REGION Network 4: OUT4
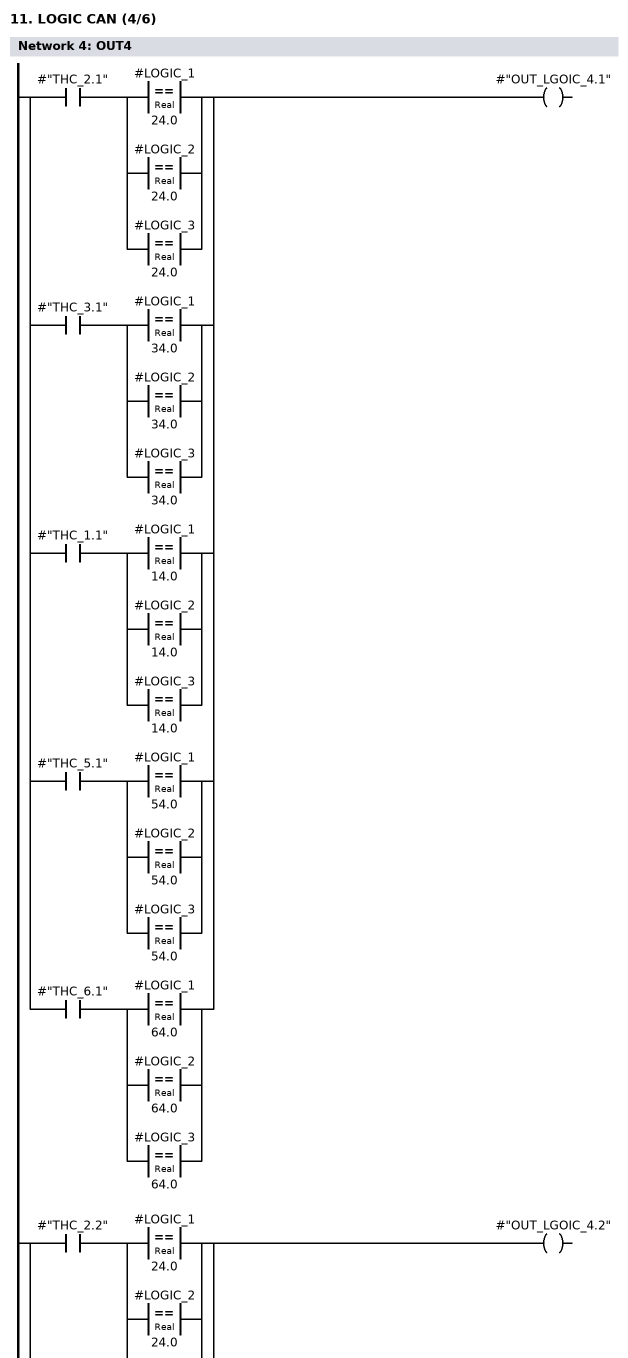
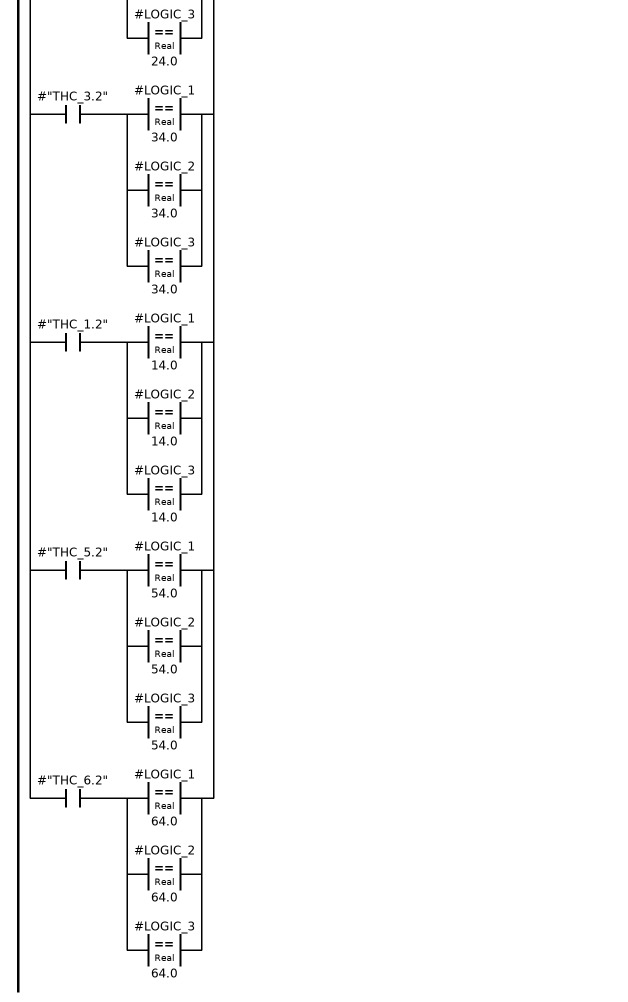
   RUNG wire#powerrail
      Contact( #"THC_2.1" )
      wire#w1
      { S7_Templates := "SrcType := Real" } EQ_Contact(in1 := #LOGIC_1, in2 := 24.0)
      wire#w2
      Coil( #"OUT_LGOIC_4.1" )
   END_RUNG
   RUNG wire#w1
      { S7_Templates := "SrcType := Real" } EQ_Contact(in1 := #LOGIC_2, in2 := 24.0)
   END_RUNG wire#w2
   RUNG wire#w1
      { S7_Templates := "SrcType := Real" } EQ_Contact(in1 := #LOGIC_3, in2 := 24.0)
   END_RUNG wire#w2
   RUNG wire#powerrail
      Contact( #"THC_3.1" )
      wire#w3
      { S7_Templates := "SrcType := Real" } EQ_Contact(in1 := #LOGIC_1, in2 := 34.0)
   END_RUNG wire#w2
   RUNG wire#w3
      { S7_Templates := "SrcType := Real" } EQ_Contact(in1 := #LOGIC_2, in2 := 34.0)
   END_RUNG wire#w2
   RUNG wire#w3
      { S7_Templates := "SrcType := Real" } EQ_Contact(in1 := #LOGIC_3, in2 := 34.0)
   END_RUNG wire#w2
   RUNG wire#powerrail
      Contact( #"THC_1.1" )
      wire#w4
      { S7_Templates := "SrcType := Real" } EQ_Contact(in1 := #LOGIC_1, in2 := 14.0)
   END_RUNG wire#w2
   RUNG wire#w4
      { S7_Templates := "SrcType := Real" } EQ_Contact(in1 := #LOGIC_2, in2 := 14.0)
   END_RUNG wire#w2
   RUNG wire#w4
      { S7_Templates := "SrcType := Real" } EQ_Contact(in1 := #LOGIC_3, in2 := 14.0)
   END_RUNG wire#w2
   RUNG wire#powerrail
      Contact( #"THC_5.1" )
      wire#w5
      { S7_Templates := "SrcType := Real" } EQ_Contact(in1 := #LOGIC_1, in2 := 54.0)
   END_RUNG wire#w2
   RUNG wire#w5
      { S7_Templates := "SrcType := Real" } EQ_Contact(in1 := #LOGIC_2, in2 := 54.0)
   END_RUNG wire#w2
   RUNG wire#w5
      { S7_Templates := "SrcType := Real" } EQ_Contact(in1 := #LOGIC_3, in2 := 54.0)
   END_RUNG wire#w2
   RUNG wire#powerrail
      Contact( #"THC_6.1" )
      wire#w6
      { S7_Templates := "SrcType := Real" } EQ_Contact(in1 := #LOGIC_1, in2 := 64.0)
   END_RUNG wire#w2
   RUNG wire#w6
      { S7_Templates := "SrcType := Real" } EQ_Contact(in1 := #LOGIC_2, in2 := 64.0)
   END_RUNG wire#w2
   RUNG wire#w6
      { S7_Templates := "SrcType := Real" } EQ_Contact(in1 := #LOGIC_3, in2 := 64.0)
   END_RUNG wire#w2
   RUNG wire#powerrail
      Contact( #"THC_2.2" )
      wire#w7
      { S7_Templates := "SrcType := Real" } EQ_Contact(in1 := #LOGIC_1, in2 := 24.0)
      wire#w8
      Coil( #"OUT_LGOIC_4.2" )
   END_RUNG
   RUNG wire#w7
      { S7_Templates := "SrcType := Real" } EQ_Contact(in1 := #LOGIC_2, in2 := 24.0)
   END_RUNG wire#w8
   RUNG wire#w7
      { S7_Templates := "SrcType := Real" } EQ_Contact(in1 := #LOGIC_3, in2 := 24.0)
   END_RUNG wire#w8
   RUNG wire#powerrail
      Contact( #"THC_3.2" )
      wire#w9
      { S7_Templates := "SrcType := Real" } EQ_Contact(in1 := #LOGIC_1, in2 := 34.0)
   END_RUNG wire#w8
   RUNG wire#w9
      { S7_Templates := "SrcType := Real" } EQ_Contact(in1 := #LOGIC_2, in2 := 34.0)
   END_RUNG wire#w8
   RUNG wire#w9
      { S7_Templates := "SrcType := Real" } EQ_Contact(in1 := #LOGIC_3, in2 := 34.0)
   END_RUNG wire#w8
   RUNG wire#powerrail
      Contact( #"THC_1.2" )
      wire#w10
      { S7_Templates := "SrcType := Real" } EQ_Contact(in1 := #LOGIC_1, in2 := 14.0)
   END_RUNG wire#w8
   RUNG wire#w10
      { S7_Templates := "SrcType := Real" } EQ_Contact(in1 := #LOGIC_2, in2 := 14.0)
   END_RUNG wire#w8
   RUNG wire#w10
      { S7_Templates := "SrcType := Real" } EQ_Contact(in1 := #LOGIC_3, in2 := 14.0)
   END_RUNG wire#w8
   RUNG wire#powerrail
      Contact( #"THC_5.2" )
      wire#w11
      { S7_Templates := "SrcType := Real" } EQ_Contact(in1 := #LOGIC_1, in2 := 54.0)
   END_RUNG wire#w8
   RUNG wire#w11
      { S7_Templates := "SrcType := Real" } EQ_Contact(in1 := #LOGIC_2, in2 := 54.0)
   END_RUNG wire#w8
   RUNG wire#w11
      { S7_Templates := "SrcType := Real" } EQ_Contact(in1 := #LOGIC_3, in2 := 54.0)
   END_RUNG wire#w8
   RUNG wire#powerrail
      Contact( #"THC_6.2" )
      wire#w12
      { S7_Templates := "SrcType := Real" } EQ_Contact(in1 := #LOGIC_1, in2 := 64.0)
   END_RUNG wire#w8
   RUNG wire#w12
      { S7_Templates := "SrcType := Real" } EQ_Contact(in1 := #LOGIC_2, in2 := 64.0)
   END_RUNG wire#w8
   RUNG wire#w12
      { S7_Templates := "SrcType := Real" } EQ_Contact(in1 := #LOGIC_3, in2 := 64.0)
   END_RUNG wire#w8
   // the same network as SCL:
   #"OUT_LGOIC_4.1" := (#"THC_2.1" AND ((#LOGIC_1 = 24.0) OR (#LOGIC_2 = 24.0) OR (#LOGIC_3 = 24.0))) OR (#"THC_3.1" AND ((#LOGIC_1 = 34.0) OR (#LOGIC_2 = 34.0) OR (#LOGIC_3 = 34.0))) OR (#"THC_1.1" AND ((#LOGIC_1 = 14.0) OR (#LOGIC_2 = 14.0) OR (#LOGIC_3 = 14.0))) OR (#"THC_5.1" AND ((#LOGIC_1 = 54.0) OR (#LOGIC_2 = 54.0) OR (#LOGIC_3 = 54.0))) OR (#"THC_6.1" AND ((#LOGIC_1 = 64.0) OR (#LOGIC_2 = 64.0) OR (#LOGIC_3 = 64.0)));
   #"OUT_LGOIC_4.2" := (#"THC_2.2" AND ((#LOGIC_1 = 24.0) OR (#LOGIC_2 = 24.0) OR (#LOGIC_3 = 24.0))) OR (#"THC_3.2" AND ((#LOGIC_1 = 34.0) OR (#LOGIC_2 = 34.0) OR (#LOGIC_3 = 34.0))) OR (#"THC_1.2" AND ((#LOGIC_1 = 14.0) OR (#LOGIC_2 = 14.0) OR (#LOGIC_3 = 14.0))) OR (#"THC_5.2" AND ((#LOGIC_1 = 54.0) OR (#LOGIC_2 = 54.0) OR (#LOGIC_3 = 54.0))) OR (#"THC_6.2" AND ((#LOGIC_1 = 64.0) OR (#LOGIC_2 = 64.0) OR (#LOGIC_3 = 64.0)));
END_REGION

REGION Network 5: OUT5
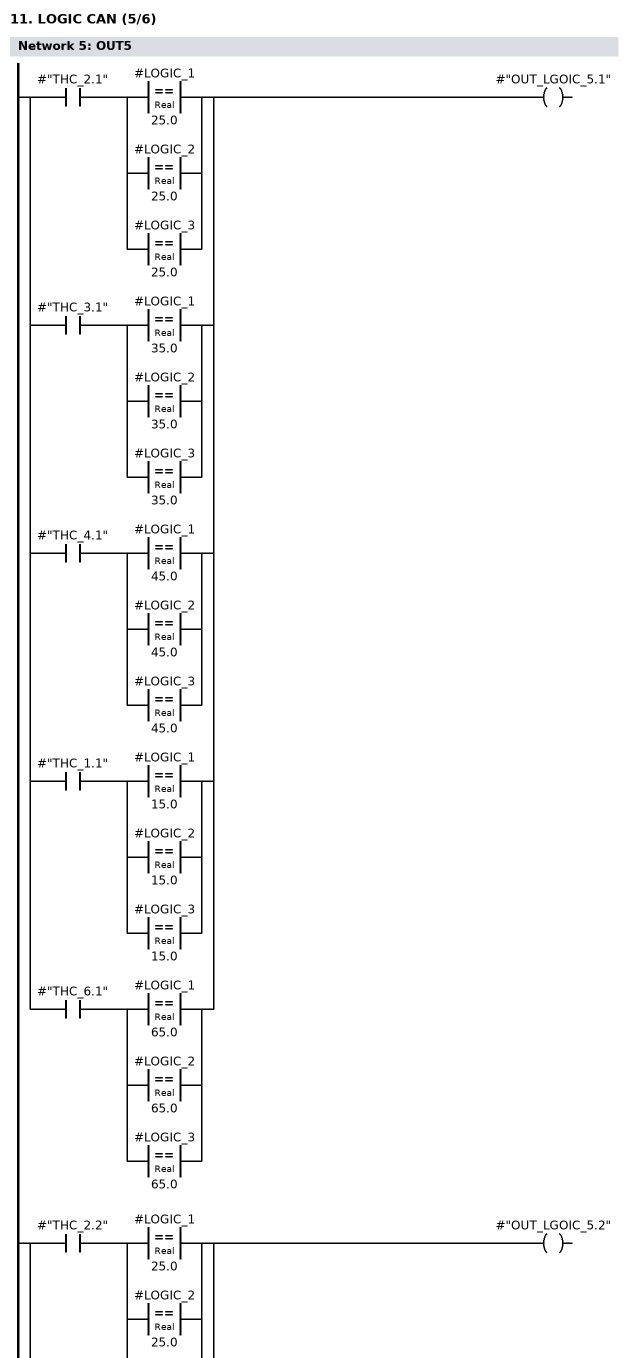
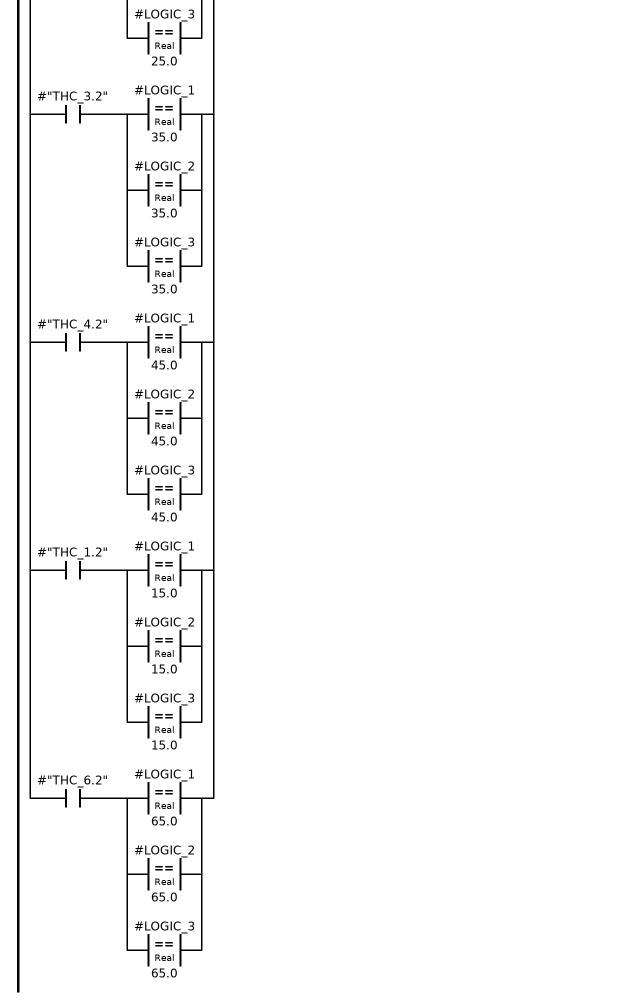
   RUNG wire#powerrail
      Contact( #"THC_2.1" )
      wire#w1
      { S7_Templates := "SrcType := Real" } EQ_Contact(in1 := #LOGIC_1, in2 := 25.0)
      wire#w2
      Coil( #"OUT_LGOIC_5.1" )
   END_RUNG
   RUNG wire#w1
      { S7_Templates := "SrcType := Real" } EQ_Contact(in1 := #LOGIC_2, in2 := 25.0)
   END_RUNG wire#w2
   RUNG wire#w1
      { S7_Templates := "SrcType := Real" } EQ_Contact(in1 := #LOGIC_3, in2 := 25.0)
   END_RUNG wire#w2
   RUNG wire#powerrail
      Contact( #"THC_3.1" )
      wire#w3
      { S7_Templates := "SrcType := Real" } EQ_Contact(in1 := #LOGIC_1, in2 := 35.0)
   END_RUNG wire#w2
   RUNG wire#w3
      { S7_Templates := "SrcType := Real" } EQ_Contact(in1 := #LOGIC_2, in2 := 35.0)
   END_RUNG wire#w2
   RUNG wire#w3
      { S7_Templates := "SrcType := Real" } EQ_Contact(in1 := #LOGIC_3, in2 := 35.0)
   END_RUNG wire#w2
   RUNG wire#powerrail
      Contact( #"THC_4.1" )
      wire#w4
      { S7_Templates := "SrcType := Real" } EQ_Contact(in1 := #LOGIC_1, in2 := 45.0)
   END_RUNG wire#w2
   RUNG wire#w4
      { S7_Templates := "SrcType := Real" } EQ_Contact(in1 := #LOGIC_2, in2 := 45.0)
   END_RUNG wire#w2
   RUNG wire#w4
      { S7_Templates := "SrcType := Real" } EQ_Contact(in1 := #LOGIC_3, in2 := 45.0)
   END_RUNG wire#w2
   RUNG wire#powerrail
      Contact( #"THC_1.1" )
      wire#w5
      { S7_Templates := "SrcType := Real" } EQ_Contact(in1 := #LOGIC_1, in2 := 15.0)
   END_RUNG wire#w2
   RUNG wire#w5
      { S7_Templates := "SrcType := Real" } EQ_Contact(in1 := #LOGIC_2, in2 := 15.0)
   END_RUNG wire#w2
   RUNG wire#w5
      { S7_Templates := "SrcType := Real" } EQ_Contact(in1 := #LOGIC_3, in2 := 15.0)
   END_RUNG wire#w2
   RUNG wire#powerrail
      Contact( #"THC_6.1" )
      wire#w6
      { S7_Templates := "SrcType := Real" } EQ_Contact(in1 := #LOGIC_1, in2 := 65.0)
   END_RUNG wire#w2
   RUNG wire#w6
      { S7_Templates := "SrcType := Real" } EQ_Contact(in1 := #LOGIC_2, in2 := 65.0)
   END_RUNG wire#w2
   RUNG wire#w6
      { S7_Templates := "SrcType := Real" } EQ_Contact(in1 := #LOGIC_3, in2 := 65.0)
   END_RUNG wire#w2
   RUNG wire#powerrail
      Contact( #"THC_2.2" )
      wire#w7
      { S7_Templates := "SrcType := Real" } EQ_Contact(in1 := #LOGIC_1, in2 := 25.0)
      wire#w8
      Coil( #"OUT_LGOIC_5.2" )
   END_RUNG
   RUNG wire#w7
      { S7_Templates := "SrcType := Real" } EQ_Contact(in1 := #LOGIC_2, in2 := 25.0)
   END_RUNG wire#w8
   RUNG wire#w7
      { S7_Templates := "SrcType := Real" } EQ_Contact(in1 := #LOGIC_3, in2 := 25.0)
   END_RUNG wire#w8
   RUNG wire#powerrail
      Contact( #"THC_3.2" )
      wire#w9
      { S7_Templates := "SrcType := Real" } EQ_Contact(in1 := #LOGIC_1, in2 := 35.0)
   END_RUNG wire#w8
   RUNG wire#w9
      { S7_Templates := "SrcType := Real" } EQ_Contact(in1 := #LOGIC_2, in2 := 35.0)
   END_RUNG wire#w8
   RUNG wire#w9
      { S7_Templates := "SrcType := Real" } EQ_Contact(in1 := #LOGIC_3, in2 := 35.0)
   END_RUNG wire#w8
   RUNG wire#powerrail
      Contact( #"THC_4.2" )
      wire#w10
      { S7_Templates := "SrcType := Real" } EQ_Contact(in1 := #LOGIC_1, in2 := 45.0)
   END_RUNG wire#w8
   RUNG wire#w10
      { S7_Templates := "SrcType := Real" } EQ_Contact(in1 := #LOGIC_2, in2 := 45.0)
   END_RUNG wire#w8
   RUNG wire#w10
      { S7_Templates := "SrcType := Real" } EQ_Contact(in1 := #LOGIC_3, in2 := 45.0)
   END_RUNG wire#w8
   RUNG wire#powerrail
      Contact( #"THC_1.2" )
      wire#w11
      { S7_Templates := "SrcType := Real" } EQ_Contact(in1 := #LOGIC_1, in2 := 15.0)
   END_RUNG wire#w8
   RUNG wire#w11
      { S7_Templates := "SrcType := Real" } EQ_Contact(in1 := #LOGIC_2, in2 := 15.0)
   END_RUNG wire#w8
   RUNG wire#w11
      { S7_Templates := "SrcType := Real" } EQ_Contact(in1 := #LOGIC_3, in2 := 15.0)
   END_RUNG wire#w8
   RUNG wire#powerrail
      Contact( #"THC_6.2" )
      wire#w12
      { S7_Templates := "SrcType := Real" } EQ_Contact(in1 := #LOGIC_1, in2 := 65.0)
   END_RUNG wire#w8
   RUNG wire#w12
      { S7_Templates := "SrcType := Real" } EQ_Contact(in1 := #LOGIC_2, in2 := 65.0)
   END_RUNG wire#w8
   RUNG wire#w12
      { S7_Templates := "SrcType := Real" } EQ_Contact(in1 := #LOGIC_3, in2 := 65.0)
   END_RUNG wire#w8
   // the same network as SCL:
   #"OUT_LGOIC_5.1" := (#"THC_2.1" AND ((#LOGIC_1 = 25.0) OR (#LOGIC_2 = 25.0) OR (#LOGIC_3 = 25.0))) OR (#"THC_3.1" AND ((#LOGIC_1 = 35.0) OR (#LOGIC_2 = 35.0) OR (#LOGIC_3 = 35.0))) OR (#"THC_4.1" AND ((#LOGIC_1 = 45.0) OR (#LOGIC_2 = 45.0) OR (#LOGIC_3 = 45.0))) OR (#"THC_1.1" AND ((#LOGIC_1 = 15.0) OR (#LOGIC_2 = 15.0) OR (#LOGIC_3 = 15.0))) OR (#"THC_6.1" AND ((#LOGIC_1 = 65.0) OR (#LOGIC_2 = 65.0) OR (#LOGIC_3 = 65.0)));
   #"OUT_LGOIC_5.2" := (#"THC_2.2" AND ((#LOGIC_1 = 25.0) OR (#LOGIC_2 = 25.0) OR (#LOGIC_3 = 25.0))) OR (#"THC_3.2" AND ((#LOGIC_1 = 35.0) OR (#LOGIC_2 = 35.0) OR (#LOGIC_3 = 35.0))) OR (#"THC_4.2" AND ((#LOGIC_1 = 45.0) OR (#LOGIC_2 = 45.0) OR (#LOGIC_3 = 45.0))) OR (#"THC_1.2" AND ((#LOGIC_1 = 15.0) OR (#LOGIC_2 = 15.0) OR (#LOGIC_3 = 15.0))) OR (#"THC_6.2" AND ((#LOGIC_1 = 65.0) OR (#LOGIC_2 = 65.0) OR (#LOGIC_3 = 65.0)));
END_REGION

REGION Network 6: OUT6
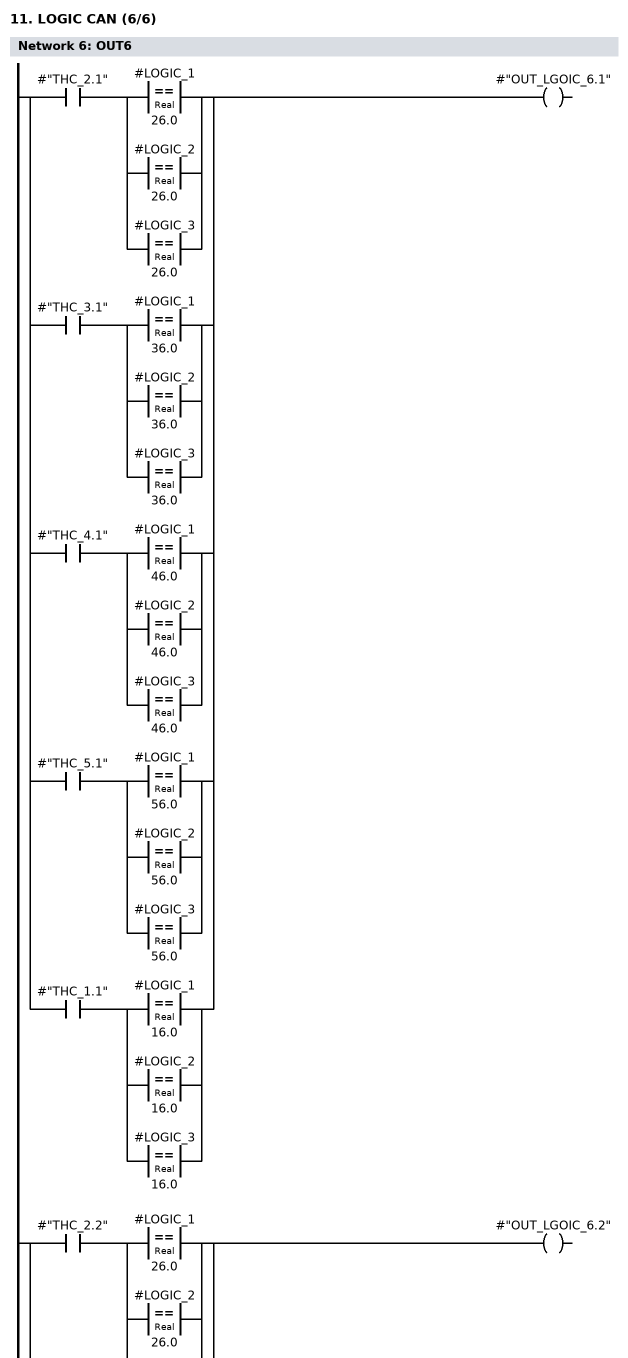
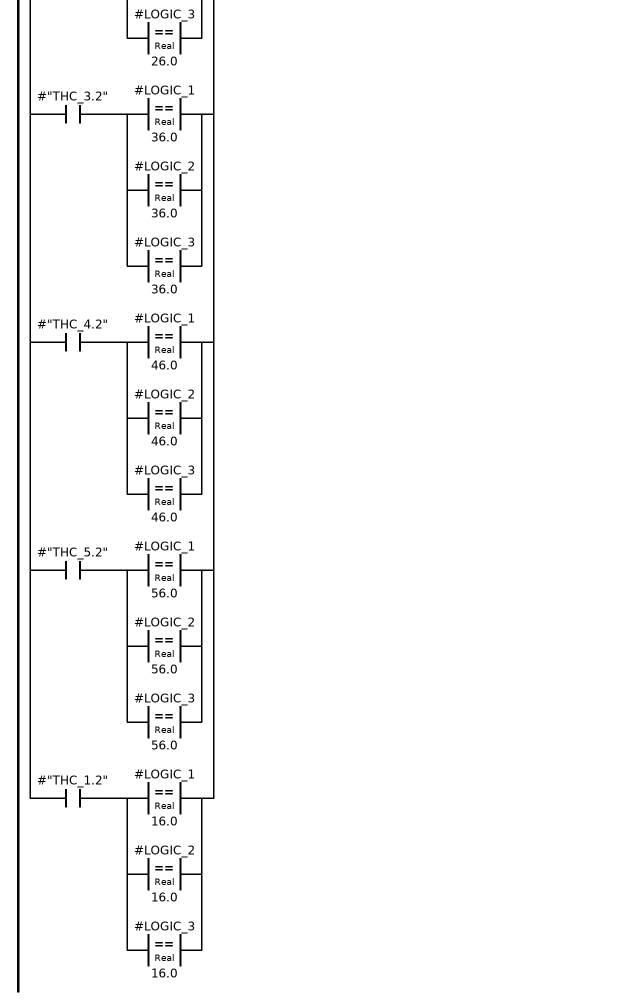
   RUNG wire#powerrail
      Contact( #"THC_2.1" )
      wire#w1
      { S7_Templates := "SrcType := Real" } EQ_Contact(in1 := #LOGIC_1, in2 := 26.0)
      wire#w2
      Coil( #"OUT_LGOIC_6.1" )
   END_RUNG
   RUNG wire#w1
      { S7_Templates := "SrcType := Real" } EQ_Contact(in1 := #LOGIC_2, in2 := 26.0)
   END_RUNG wire#w2
   RUNG wire#w1
      { S7_Templates := "SrcType := Real" } EQ_Contact(in1 := #LOGIC_3, in2 := 26.0)
   END_RUNG wire#w2
   RUNG wire#powerrail
      Contact( #"THC_3.1" )
      wire#w3
      { S7_Templates := "SrcType := Real" } EQ_Contact(in1 := #LOGIC_1, in2 := 36.0)
   END_RUNG wire#w2
   RUNG wire#w3
      { S7_Templates := "SrcType := Real" } EQ_Contact(in1 := #LOGIC_2, in2 := 36.0)
   END_RUNG wire#w2
   RUNG wire#w3
      { S7_Templates := "SrcType := Real" } EQ_Contact(in1 := #LOGIC_3, in2 := 36.0)
   END_RUNG wire#w2
   RUNG wire#powerrail
      Contact( #"THC_4.1" )
      wire#w4
      { S7_Templates := "SrcType := Real" } EQ_Contact(in1 := #LOGIC_1, in2 := 46.0)
   END_RUNG wire#w2
   RUNG wire#w4
      { S7_Templates := "SrcType := Real" } EQ_Contact(in1 := #LOGIC_2, in2 := 46.0)
   END_RUNG wire#w2
   RUNG wire#w4
      { S7_Templates := "SrcType := Real" } EQ_Contact(in1 := #LOGIC_3, in2 := 46.0)
   END_RUNG wire#w2
   RUNG wire#powerrail
      Contact( #"THC_5.1" )
      wire#w5
      { S7_Templates := "SrcType := Real" } EQ_Contact(in1 := #LOGIC_1, in2 := 56.0)
   END_RUNG wire#w2
   RUNG wire#w5
      { S7_Templates := "SrcType := Real" } EQ_Contact(in1 := #LOGIC_2, in2 := 56.0)
   END_RUNG wire#w2
   RUNG wire#w5
      { S7_Templates := "SrcType := Real" } EQ_Contact(in1 := #LOGIC_3, in2 := 56.0)
   END_RUNG wire#w2
   RUNG wire#powerrail
      Contact( #"THC_1.1" )
      wire#w6
      { S7_Templates := "SrcType := Real" } EQ_Contact(in1 := #LOGIC_1, in2 := 16.0)
   END_RUNG wire#w2
   RUNG wire#w6
      { S7_Templates := "SrcType := Real" } EQ_Contact(in1 := #LOGIC_2, in2 := 16.0)
   END_RUNG wire#w2
   RUNG wire#w6
      { S7_Templates := "SrcType := Real" } EQ_Contact(in1 := #LOGIC_3, in2 := 16.0)
   END_RUNG wire#w2
   RUNG wire#powerrail
      Contact( #"THC_2.2" )
      wire#w7
      { S7_Templates := "SrcType := Real" } EQ_Contact(in1 := #LOGIC_1, in2 := 26.0)
      wire#w8
      Coil( #"OUT_LGOIC_6.2" )
   END_RUNG
   RUNG wire#w7
      { S7_Templates := "SrcType := Real" } EQ_Contact(in1 := #LOGIC_2, in2 := 26.0)
   END_RUNG wire#w8
   RUNG wire#w7
      { S7_Templates := "SrcType := Real" } EQ_Contact(in1 := #LOGIC_3, in2 := 26.0)
   END_RUNG wire#w8
   RUNG wire#powerrail
      Contact( #"THC_3.2" )
      wire#w9
      { S7_Templates := "SrcType := Real" } EQ_Contact(in1 := #LOGIC_1, in2 := 36.0)
   END_RUNG wire#w8
   RUNG wire#w9
      { S7_Templates := "SrcType := Real" } EQ_Contact(in1 := #LOGIC_2, in2 := 36.0)
   END_RUNG wire#w8
   RUNG wire#w9
      { S7_Templates := "SrcType := Real" } EQ_Contact(in1 := #LOGIC_3, in2 := 36.0)
   END_RUNG wire#w8
   RUNG wire#powerrail
      Contact( #"THC_4.2" )
      wire#w10
      { S7_Templates := "SrcType := Real" } EQ_Contact(in1 := #LOGIC_1, in2 := 46.0)
   END_RUNG wire#w8
   RUNG wire#w10
      { S7_Templates := "SrcType := Real" } EQ_Contact(in1 := #LOGIC_2, in2 := 46.0)
   END_RUNG wire#w8
   RUNG wire#w10
      { S7_Templates := "SrcType := Real" } EQ_Contact(in1 := #LOGIC_3, in2 := 46.0)
   END_RUNG wire#w8
   RUNG wire#powerrail
      Contact( #"THC_5.2" )
      wire#w11
      { S7_Templates := "SrcType := Real" } EQ_Contact(in1 := #LOGIC_1, in2 := 56.0)
   END_RUNG wire#w8
   RUNG wire#w11
      { S7_Templates := "SrcType := Real" } EQ_Contact(in1 := #LOGIC_2, in2 := 56.0)
   END_RUNG wire#w8
   RUNG wire#w11
      { S7_Templates := "SrcType := Real" } EQ_Contact(in1 := #LOGIC_3, in2 := 56.0)
   END_RUNG wire#w8
   RUNG wire#powerrail
      Contact( #"THC_1.2" )
      wire#w12
      { S7_Templates := "SrcType := Real" } EQ_Contact(in1 := #LOGIC_1, in2 := 16.0)
   END_RUNG wire#w8
   RUNG wire#w12
      { S7_Templates := "SrcType := Real" } EQ_Contact(in1 := #LOGIC_2, in2 := 16.0)
   END_RUNG wire#w8
   RUNG wire#w12
      { S7_Templates := "SrcType := Real" } EQ_Contact(in1 := #LOGIC_3, in2 := 16.0)
   END_RUNG wire#w8
   // the same network as SCL:
   #"OUT_LGOIC_6.1" := (#"THC_2.1" AND ((#LOGIC_1 = 26.0) OR (#LOGIC_2 = 26.0) OR (#LOGIC_3 = 26.0))) OR (#"THC_3.1" AND ((#LOGIC_1 = 36.0) OR (#LOGIC_2 = 36.0) OR (#LOGIC_3 = 36.0))) OR (#"THC_4.1" AND ((#LOGIC_1 = 46.0) OR (#LOGIC_2 = 46.0) OR (#LOGIC_3 = 46.0))) OR (#"THC_5.1" AND ((#LOGIC_1 = 56.0) OR (#LOGIC_2 = 56.0) OR (#LOGIC_3 = 56.0))) OR (#"THC_1.1" AND ((#LOGIC_1 = 16.0) OR (#LOGIC_2 = 16.0) OR (#LOGIC_3 = 16.0)));
   #"OUT_LGOIC_6.2" := (#"THC_2.2" AND ((#LOGIC_1 = 26.0) OR (#LOGIC_2 = 26.0) OR (#LOGIC_3 = 26.0))) OR (#"THC_3.2" AND ((#LOGIC_1 = 36.0) OR (#LOGIC_2 = 36.0) OR (#LOGIC_3 = 36.0))) OR (#"THC_4.2" AND ((#LOGIC_1 = 46.0) OR (#LOGIC_2 = 46.0) OR (#LOGIC_3 = 46.0))) OR (#"THC_5.2" AND ((#LOGIC_1 = 56.0) OR (#LOGIC_2 = 56.0) OR (#LOGIC_3 = 56.0))) OR (#"THC_1.2" AND ((#LOGIC_1 = 16.0) OR (#LOGIC_2 = 16.0) OR (#LOGIC_3 = 16.0)));
END_REGION
END_FUNCTION_BLOCK

FUNCTION "3.OUTPUT_PLC" : Void   // FC3, LAD
{ S7_Optimized_Access := 'TRUE' }
VERSION : 0.1
// stored: AutoNumber false, CodeModifiedDate 2025-08-27T17:07:28.4518091Z, CompileDate 2025-08-30T17:40:35.2673041Z, CreationDate 2024-10-12T12:36:08.0193576Z, HandleErrorsWithinBlock false, InterfaceModifiedDate 2022-06-07T03:40:45.7898546Z, IsConsistent true, IsIECCheckEnabled false, IsKnowHowProtected false, IsWriteProtected false, LibraryConformanceStatus The object is library-conformant., ModifiedDate 2025-08-27T17:07:28.4518091Z, ParameterModified 2022-06-07T03:40:45.7898546Z, PLCSimAdvancedSupport false, SetENOAutomatically False, StructureModified 2022-06-07T03:40:45.7898546Z, UDAEnableTagReadback false
   VAR_INPUT
      A1 : Bool;
      M1 : Bool;
      A2 : Bool;
      M2 : Bool;
      A3 : Bool;
      M3 : Bool;
      A4 : Bool;
      M4 : Bool;
   END_VAR
   VAR_OUTPUT
      OUT1 : Bool;
      OUT2 : Bool;
      OUT3 : Bool;
      OUT4 : Bool;
   END_VAR
BEGIN

REGION Network 1
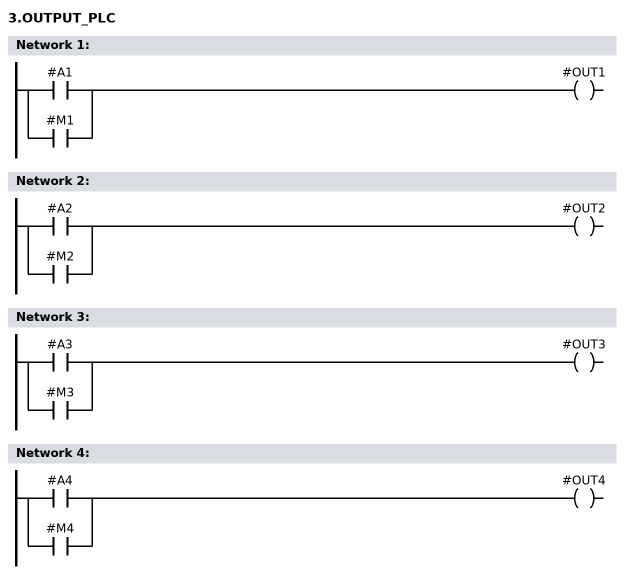
   RUNG wire#powerrail
      Contact( #A1 )
      wire#w1
      Coil( #OUT1 )
   END_RUNG
   RUNG wire#powerrail
      Contact( #M1 )
   END_RUNG wire#w1
   // the same network as SCL:
   #OUT1 := #A1 OR #M1;
END_REGION

REGION Network 2
   RUNG wire#powerrail
      Contact( #A2 )
      wire#w1
      Coil( #OUT2 )
   END_RUNG
   RUNG wire#powerrail
      Contact( #M2 )
   END_RUNG wire#w1
   // the same network as SCL:
   #OUT2 := #A2 OR #M2;
END_REGION

REGION Network 3
   RUNG wire#powerrail
      Contact( #A3 )
      wire#w1
      Coil( #OUT3 )
   END_RUNG
   RUNG wire#powerrail
      Contact( #M3 )
   END_RUNG wire#w1
   // the same network as SCL:
   #OUT3 := #A3 OR #M3;
END_REGION

REGION Network 4
   RUNG wire#powerrail
      Contact( #A4 )
      wire#w1
      Coil( #OUT4 )
   END_RUNG
   RUNG wire#powerrail
      Contact( #M4 )
   END_RUNG wire#w1
   // the same network as SCL:
   #OUT4 := #A4 OR #M4;
END_REGION
END_FUNCTION

FUNCTION_BLOCK "3.RUN_MODE"   // FB3, LAD
{ S7_Optimized_Access := 'TRUE' }
VERSION : 0.1
// stored: AutoNumber false, CodeModifiedDate 2025-08-27T17:11:43.2955348Z, CompileDate 2025-08-30T17:40:35.1660868Z, CreationDate 2024-10-12T12:36:08.0193576Z, DownloadWithoutReinit false, HandleErrorsWithinBlock false, InterfaceModifiedDate 2023-07-24T14:42:19.3789304Z, IsConsistent true, IsIECCheckEnabled false, IsKnowHowProtected false, IsRetainMemResEnabled false, IsWriteProtected false, LibraryConformanceStatus The object is library-conformant., MemoryReserve 100, ModifiedDate 2025-08-27T17:11:43.2955348Z, ParameterModified 2023-07-24T14:41:56.9787559Z, PLCSimAdvancedSupport false, SetENOAutomatically False, StructureModified 2023-07-24T14:42:19.3789304Z, UDAEnableTagReadback false
   VAR_INPUT
      NN_RUN : Bool;
      NN_STOP : Bool;
      SW_SIM : Bool;
      SW_MAN : Bool;
      SW_AUT : Bool;
   END_VAR
   VAR_OUTPUT
      RUN : Bool;
      SIM : Bool;
      MAN : Bool;
      AUT : Bool;
   END_VAR
   VAR
      TEMP1 : Bool;
      TEMP2 : Bool;
   END_VAR
BEGIN

REGION Network 1
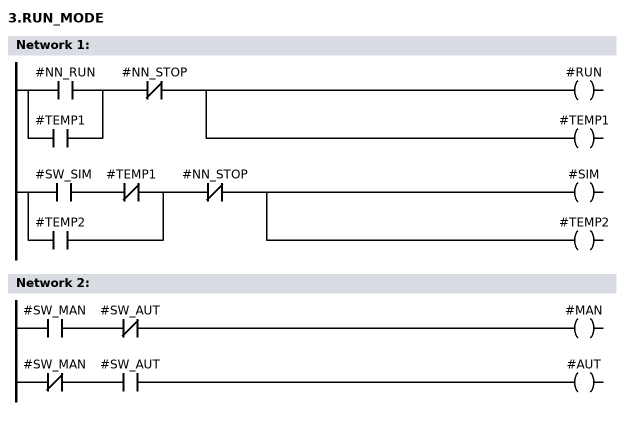
   RUNG wire#powerrail
      Contact( #NN_RUN )
      wire#w1
      I_Contact( #NN_STOP )
      wire#w2
      Coil( #RUN )
   END_RUNG
   RUNG wire#powerrail
      Contact( #TEMP1 )
   END_RUNG wire#w1
   RUNG wire#w2
      Coil( #TEMP1 )
   END_RUNG
   RUNG wire#powerrail
      Contact( #SW_SIM )
      I_Contact( #TEMP1 )
      wire#w3
      I_Contact( #NN_STOP )
      wire#w4
      Coil( #SIM )
   END_RUNG
   RUNG wire#powerrail
      Contact( #TEMP2 )
   END_RUNG wire#w3
   RUNG wire#w4
      Coil( #TEMP2 )
   END_RUNG
   // the same network as SCL:
   #RUN := (#NN_RUN OR #TEMP1) AND NOT #NN_STOP;
   #TEMP1 := #RUN;
   #SIM := ((#SW_SIM AND NOT #TEMP1) OR #TEMP2) AND NOT #NN_STOP;
   #TEMP2 := #SIM;
END_REGION

REGION Network 2
   RUNG wire#powerrail
      Contact( #SW_MAN )
      I_Contact( #SW_AUT )
      Coil( #MAN )
   END_RUNG
   RUNG wire#powerrail
      I_Contact( #SW_MAN )
      Contact( #SW_AUT )
      Coil( #AUT )
   END_RUNG
   // the same network as SCL:
   #MAN := #SW_MAN AND NOT #SW_AUT;
   #AUT := NOT #SW_MAN AND #SW_AUT;
END_REGION
END_FUNCTION_BLOCK

FUNCTION "4.CONVERT_VOLUME" : Void   // FC4, LAD
{ S7_Optimized_Access := 'TRUE' }
VERSION : 0.1
// stored: AutoNumber true, CodeModifiedDate 2025-08-27T17:08:03.467369Z, CompileDate 2025-08-30T17:40:35.2171394Z, CreationDate 2024-10-12T12:36:08.0193576Z, HandleErrorsWithinBlock false, InterfaceModifiedDate 2023-07-25T19:47:42.5745Z, IsConsistent true, IsIECCheckEnabled false, IsKnowHowProtected false, IsWriteProtected false, LibraryConformanceStatus The object is library-conformant., ModifiedDate 2025-08-27T17:08:03.467369Z, ParameterModified 2023-07-25T19:47:42.5745Z, PLCSimAdvancedSupport false, SetENOAutomatically False, StructureModified 2023-07-25T19:47:42.5745Z, UDAEnableTagReadback false
   VAR_INPUT
      SO_KHOI : Real;
      M3_MAX : Real;
   END_VAR
   VAR_OUTPUT
      SO_ME : Real;
      "M3/ME" : Real;
   END_VAR
   VAR_TEMP
      TEMP1 : Real;
      TEMP2 : Int;
      TEMP3 : Real;
   END_VAR
BEGIN

REGION Network 1
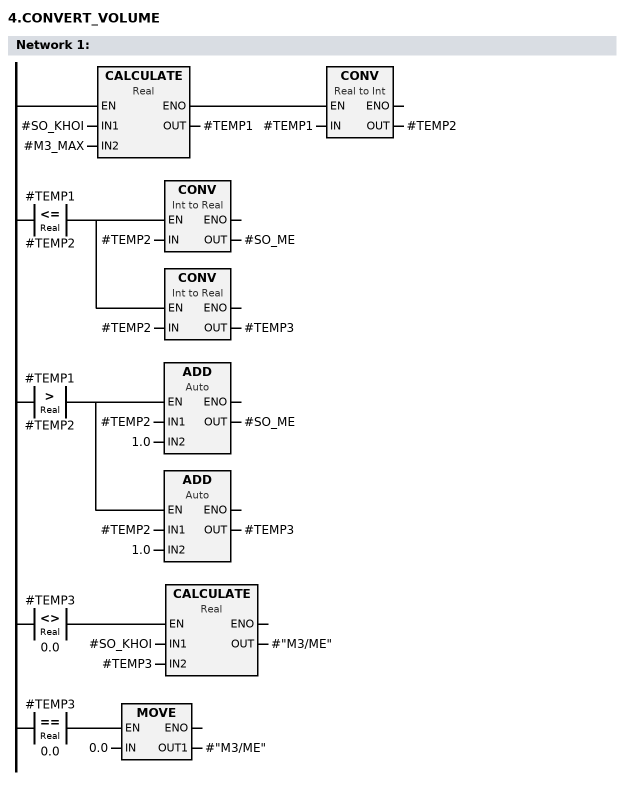
   RUNG wire#powerrail
      { S7_Templates := "SrcType := Real"; S7_Expression := "IN1/IN2" } Calculate(in1 := #SO_KHOI, in2 := #M3_MAX, out => #TEMP1)
      { S7_Templates := "[SrcType := Real, DestType := Int]" } Convert(in := #TEMP1, out => #TEMP2)
   END_RUNG
   RUNG wire#powerrail
      { S7_Templates := "SrcType := Real" } LE_Contact(in1 := #TEMP1, in2 := #TEMP2)
      wire#w1
      { S7_Templates := "[SrcType := Int, DestType := Real]" } Convert(in := #TEMP2, out => #SO_ME)
   END_RUNG
   RUNG wire#w1
      { S7_Templates := "[SrcType := Int, DestType := Real]" } Convert(in := #TEMP2, out => #TEMP3)
   END_RUNG
   RUNG wire#powerrail
      { S7_Templates := "SrcType := Real" } GT_Contact(in1 := #TEMP1, in2 := #TEMP2)
      wire#w2
      Add(in1 := #TEMP2, in2 := 1.0, out => #SO_ME)
   END_RUNG
   RUNG wire#w2
      Add(in1 := #TEMP2, in2 := 1.0, out => #TEMP3)
   END_RUNG
   RUNG wire#powerrail
      { S7_Templates := "SrcType := Real" } NE_Contact(in1 := #TEMP3, in2 := 0.0)
      { S7_Templates := "SrcType := Real"; S7_Expression := "IN1/IN2" } Calculate(in1 := #SO_KHOI, in2 := #TEMP3, out => #"M3/ME")
   END_RUNG
   RUNG wire#powerrail
      { S7_Templates := "SrcType := Real" } EQ_Contact(in1 := #TEMP3, in2 := 0.0)
      Move(in := 0.0, out1 => #"M3/ME")
   END_RUNG
   // the same network as SCL:
   #TEMP1 := #SO_KHOI/#M3_MAX;
   #TEMP2 := REAL_TO_INT(#TEMP1);
   IF #TEMP1 <= #TEMP2 THEN
       #SO_ME := INT_TO_REAL(#TEMP2);
       #TEMP3 := INT_TO_REAL(#TEMP2);
   END_IF;
   IF #TEMP1 > #TEMP2 THEN
       #SO_ME := #TEMP2 + 1.0;
       #TEMP3 := #TEMP2 + 1.0;
   END_IF;
   IF #TEMP3 <> 0.0 THEN #"M3/ME" := #SO_KHOI/#TEMP3; END_IF;
   IF #TEMP3 = 0.0 THEN #"M3/ME" := 0.0; END_IF;
END_REGION
END_FUNCTION

FUNCTION_BLOCK "5.ADDITIVES_PULE"   // FB5, LAD
{ S7_Optimized_Access := 'TRUE' }
VERSION : 0.1
// stored: AutoNumber false, CodeModifiedDate 2024-07-29T16:22:18.8856203Z, CompileDate 2025-08-30T17:40:35.1271729Z, CreationDate 2024-10-12T12:36:08.0193576Z, DownloadWithoutReinit false, HandleErrorsWithinBlock false, InterfaceModifiedDate 2024-07-29T16:20:48.5427985Z, IsConsistent true, IsIECCheckEnabled false, IsKnowHowProtected false, IsRetainMemResEnabled false, IsWriteProtected false, LibraryConformanceStatus The object is library-conformant., MemoryReserve 100, ModifiedDate 2024-07-29T16:22:18.8856203Z, ParameterModified 2024-07-29T16:20:48.5427985Z, PLCSimAdvancedSupport false, SetENOAutomatically False, StructureModified 2024-07-29T16:20:48.5427985Z, UDAEnableTagReadback false
   VAR_INPUT
      "Xung In" : DWord;
      Reset : Bool;
      "Set Tai" : Bool;
      "Khoi Luong Calib" : Real;
   END_VAR
   VAR_OUTPUT
      "Khoi Luong Out" : Real;
      "Xung Out" : Real;
   END_VAR
   VAR RETAIN
      "Xu In" : Real;
      "He So" : Real;
      "Xu Calib" : Real;
      "Kl Calib" : Real;
   END_VAR
   VAR
      M1 : Bool;
   END_VAR
   VAR_TEMP
      Conv : DInt;
   END_VAR
BEGIN

REGION Network 1
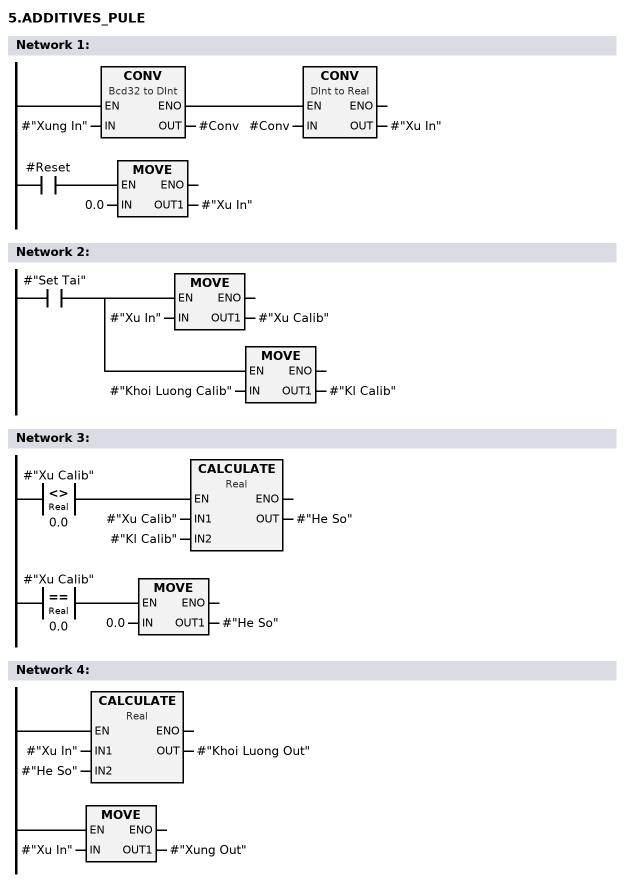
   RUNG wire#powerrail
      { S7_Templates := "[SrcType := Bcd32, DestType := DInt]" } Convert(in := #"Xung In", out => #Conv)
      { S7_Templates := "[SrcType := DInt, DestType := Real]" } Convert(in := #Conv, out => #"Xu In")
   END_RUNG
   RUNG wire#powerrail
      Contact( #Reset )
      Move(in := 0.0, out1 => #"Xu In")
   END_RUNG
   // the same network as SCL:
   #Conv := BCD32_TO_DINT(#"Xung In");
   #"Xu In" := DINT_TO_REAL(#Conv);
   IF #Reset THEN #"Xu In" := 0.0; END_IF;
END_REGION

REGION Network 2
   RUNG wire#powerrail
      Contact( #"Set Tai" )
      wire#w1
      Move(in := #"Xu In", out1 => #"Xu Calib")
   END_RUNG
   RUNG wire#w1
      Move(in := #"Khoi Luong Calib", out1 => #"Kl Calib")
   END_RUNG
   // the same network as SCL:
   IF #"Set Tai" THEN
       #"Xu Calib" := #"Xu In";
       #"Kl Calib" := #"Khoi Luong Calib";
   END_IF;
END_REGION

REGION Network 3
   RUNG wire#powerrail
      { S7_Templates := "SrcType := Real" } NE_Contact(in1 := #"Xu Calib", in2 := 0.0)
      { S7_Templates := "SrcType := Real"; S7_Expression := "IN2/IN1" } Calculate(in1 := #"Xu Calib", in2 := #"Kl Calib", out => #"He So")
   END_RUNG
   RUNG wire#powerrail
      { S7_Templates := "SrcType := Real" } EQ_Contact(in1 := #"Xu Calib", in2 := 0.0)
      Move(in := 0.0, out1 => #"He So")
   END_RUNG
   // the same network as SCL:
   IF #"Xu Calib" <> 0.0 THEN #"He So" := #"Kl Calib"/#"Xu Calib"; END_IF;
   IF #"Xu Calib" = 0.0 THEN #"He So" := 0.0; END_IF;
END_REGION

REGION Network 4
   RUNG wire#powerrail
      { S7_Templates := "SrcType := Real"; S7_Expression := "IN1*IN2" } Calculate(in1 := #"Xu In", in2 := #"He So", out => #"Khoi Luong Out")
   END_RUNG
   RUNG wire#powerrail
      Move(in := #"Xu In", out1 => #"Xung Out")
   END_RUNG
   // the same network as SCL:
   #"Khoi Luong Out" := #"Xu In"*#"He So";
   #"Xung Out" := #"Xu In";
END_REGION
END_FUNCTION_BLOCK

FUNCTION "FCCA_IND_AGG12345" : Void   // FC21, LAD
{ S7_Optimized_Access := 'TRUE' }
VERSION : 0.1
// stored: AutoNumber false, CodeModifiedDate 2026-01-09T13:44:33.0674527Z, CompileDate 2026-01-09T13:44:34.3725446Z, CreationDate 2026-01-06T17:40:48.6758963Z, HandleErrorsWithinBlock false, InterfaceModifiedDate 2026-01-06T17:40:48.6758963Z, IsConsistent true, IsIECCheckEnabled false, IsKnowHowProtected false, IsWriteProtected false, LibraryConformanceStatus Error: The block contains calls of single instances. Warning: The object contains access to global data blocks. Warning: The block contains direct access to inputs, outputs, bit memories, indirect access to the registry or indirect access to external memory areas that are unknown at the time of compilation., ModifiedDate 2026-01-09T13:44:33.0674527Z, ParameterModified 2026-01-06T17:40:48.6758963Z, PLCSimAdvancedSupport false, SetENOAutomatically False, StructureModified 2026-01-06T17:40:48.6758963Z, UDAEnableTagReadback false
   VAR_TEMP   // added for the SCL form of the ladder/FBD networks
      _w1 : Bool;
      _w2 : Bool;
   END_VAR
BEGIN

REGION Network 1: CAN COT LIEU AGG1
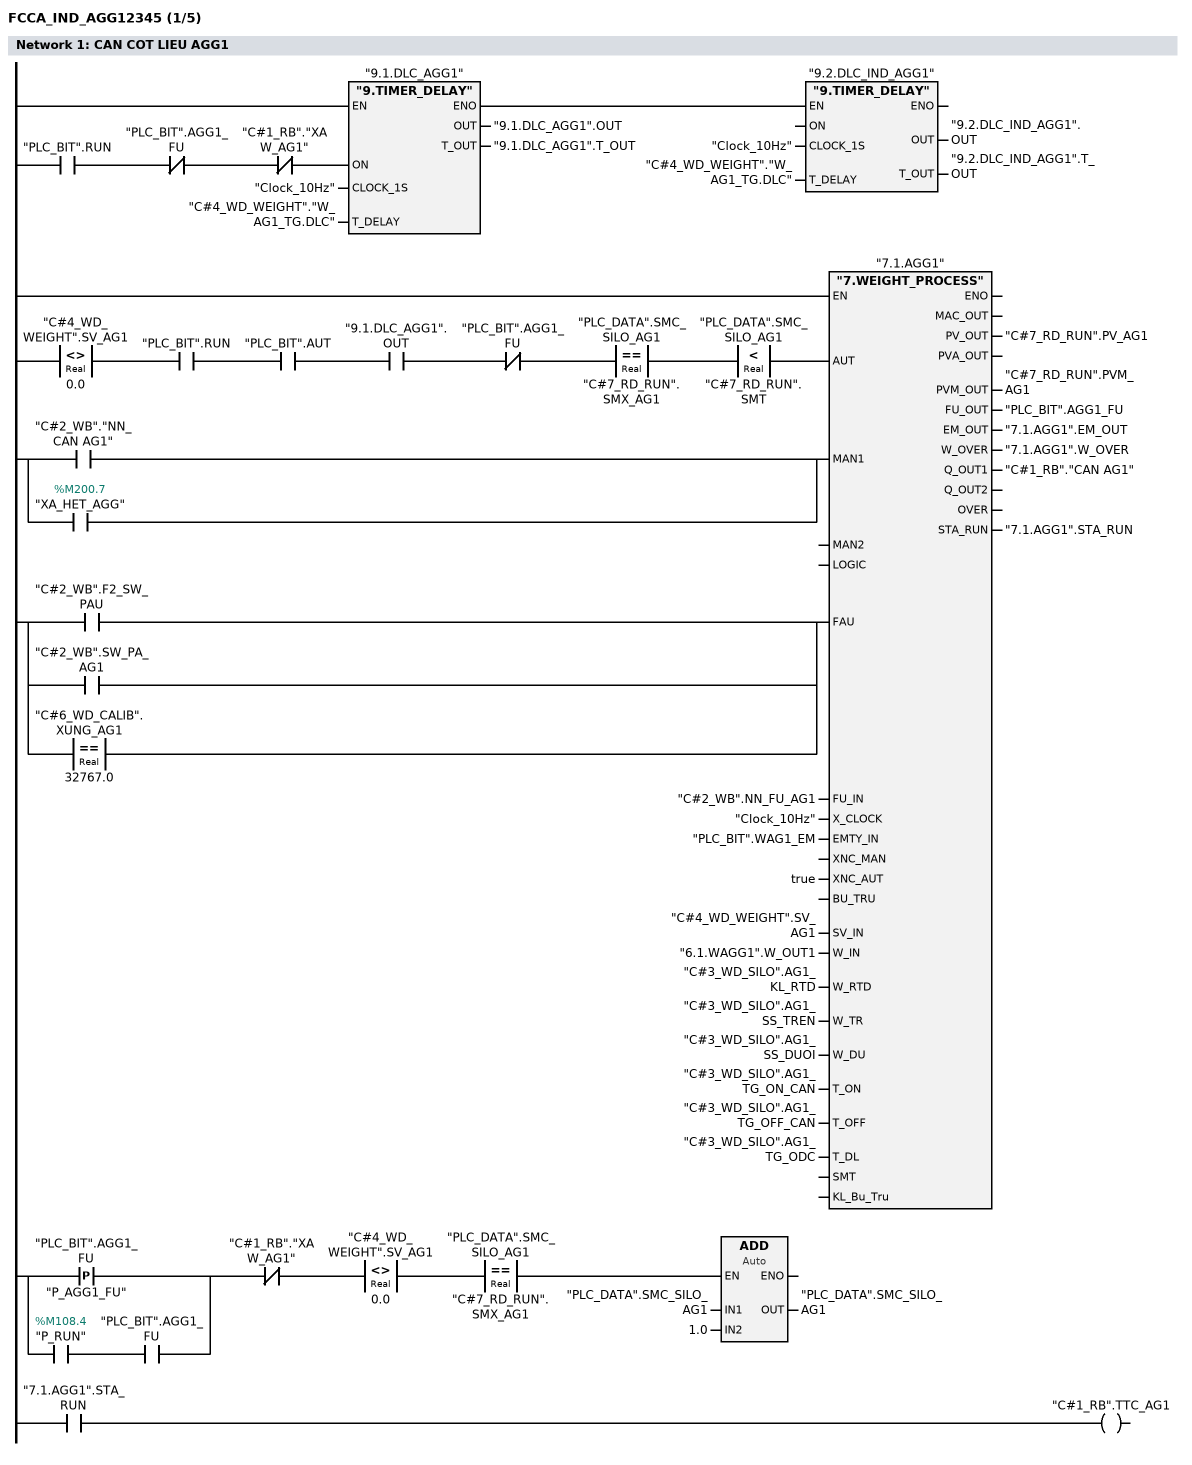
   RUNG wire#powerrail
      "9.1.DLC_AGG1"(ON := wire#w1, CLOCK_1S := "Clock_10Hz", T_DELAY := "C#4_WD_WEIGHT"."W_AG1_TG.DLC", OUT => "9.1.DLC_AGG1".OUT, T_OUT => "9.1.DLC_AGG1".T_OUT)
      "9.2.DLC_IND_AGG1"(ON :=, CLOCK_1S := "Clock_10Hz", T_DELAY := "C#4_WD_WEIGHT"."W_AG1_TG.DLC", OUT => "9.2.DLC_IND_AGG1".OUT, T_OUT => "9.2.DLC_IND_AGG1".T_OUT)
   END_RUNG
   RUNG wire#powerrail
      Contact( "PLC_BIT".RUN )
      I_Contact( "PLC_BIT".AGG1_FU )
      I_Contact( "C#1_RB"."XA W_AG1" )
   END_RUNG wire#w1
   RUNG wire#powerrail
      "7.1.AGG1"(AUT := wire#w2, MAN1 := wire#w3, FAU := wire#w4, MAN2 :=, LOGIC :=, FU_IN := "C#2_WB".NN_FU_AG1, X_CLOCK := "Clock_10Hz", EMTY_IN := "PLC_BIT".WAG1_EM, XNC_MAN :=, XNC_AUT := true, BU_TRU :=, SV_IN := "C#4_WD_WEIGHT".SV_AG1, W_IN := "6.1.WAGG1".W_OUT1, W_RTD := "C#3_WD_SILO".AG1_KL_RTD, W_TR := "C#3_WD_SILO".AG1_SS_TREN, W_DU := "C#3_WD_SILO".AG1_SS_DUOI, T_ON := "C#3_WD_SILO".AG1_TG_ON_CAN, T_OFF := "C#3_WD_SILO".AG1_TG_OFF_CAN, T_DL := "C#3_WD_SILO".AG1_TG_ODC, SMT :=, KL_Bu_Tru :=, MAC_OUT =>, PV_OUT => "C#7_RD_RUN".PV_AG1, PVA_OUT =>, PVM_OUT => "C#7_RD_RUN".PVM_AG1, FU_OUT => "PLC_BIT".AGG1_FU, EM_OUT => "7.1.AGG1".EM_OUT, W_OVER => "7.1.AGG1".W_OVER, Q_OUT1 => "C#1_RB"."CAN AG1", Q_OUT2 =>, OVER =>, STA_RUN => "7.1.AGG1".STA_RUN)
   END_RUNG
   RUNG wire#powerrail
      { S7_Templates := "SrcType := Real" } NE_Contact(in1 := "C#4_WD_WEIGHT".SV_AG1, in2 := 0.0)
      Contact( "PLC_BIT".RUN )
      Contact( "PLC_BIT".AUT )
      Contact( "9.1.DLC_AGG1".OUT )
      I_Contact( "PLC_BIT".AGG1_FU )
      { S7_Templates := "SrcType := Real" } EQ_Contact(in1 := "PLC_DATA".SMC_SILO_AG1, in2 := "C#7_RD_RUN".SMX_AG1)
      { S7_Templates := "SrcType := Real" } LT_Contact(in1 := "PLC_DATA".SMC_SILO_AG1, in2 := "C#7_RD_RUN".SMT)
   END_RUNG wire#w2
   RUNG wire#powerrail
      Contact( "C#2_WB"."NN_CAN AG1" )
   END_RUNG wire#w3
   RUNG wire#powerrail
      Contact( "XA_HET_AGG" )
   END_RUNG wire#w3
   RUNG wire#powerrail
      Contact( "C#2_WB".F2_SW_PAU )
   END_RUNG wire#w4
   RUNG wire#powerrail
      Contact( "C#2_WB".SW_PA_AG1 )
   END_RUNG wire#w4
   RUNG wire#powerrail
      { S7_Templates := "SrcType := Real" } EQ_Contact(in1 := "C#6_WD_CALIB".XUNG_AG1, in2 := 32767.0)
   END_RUNG wire#w4
   RUNG wire#powerrail
      P_Contact(operand := "PLC_BIT".AGG1_FU, bit := "P_AGG1_FU")
      wire#w5
      I_Contact( "C#1_RB"."XA W_AG1" )
      { S7_Templates := "SrcType := Real" } NE_Contact(in1 := "C#4_WD_WEIGHT".SV_AG1, in2 := 0.0)
      { S7_Templates := "SrcType := Real" } EQ_Contact(in1 := "PLC_DATA".SMC_SILO_AG1, in2 := "C#7_RD_RUN".SMX_AG1)
      Add(in1 := "PLC_DATA".SMC_SILO_AG1, in2 := 1.0, out => "PLC_DATA".SMC_SILO_AG1)
   END_RUNG
   RUNG wire#powerrail
      Contact( "P_RUN" )
      Contact( "PLC_BIT".AGG1_FU )
   END_RUNG wire#w5
   RUNG wire#powerrail
      Contact( "7.1.AGG1".STA_RUN )
      Coil( "C#1_RB".TTC_AG1 )
   END_RUNG
   // the same network as SCL:
   "9.1.DLC_AGG1"(ON := "PLC_BIT".RUN AND NOT "PLC_BIT".AGG1_FU AND NOT "C#1_RB"."XA W_AG1",   // "9.TIMER_DELAY"
                  CLOCK_1S := "Clock_10Hz",
                  T_DELAY := "C#4_WD_WEIGHT"."W_AG1_TG.DLC",
                  OUT => "9.1.DLC_AGG1".OUT,
                  T_OUT => "9.1.DLC_AGG1".T_OUT,
                  ENO => #_w1);
   IF #_w1 THEN
       "9.2.DLC_IND_AGG1"(CLOCK_1S := "Clock_10Hz",   // "9.TIMER_DELAY"
                          T_DELAY := "C#4_WD_WEIGHT"."W_AG1_TG.DLC",
                          OUT => "9.2.DLC_IND_AGG1".OUT,
                          T_OUT => "9.2.DLC_IND_AGG1".T_OUT);
   END_IF;
   "7.1.AGG1"(AUT := ("C#4_WD_WEIGHT".SV_AG1 <> 0.0) AND "PLC_BIT".RUN AND "PLC_BIT".AUT AND "9.1.DLC_AGG1".OUT AND NOT "PLC_BIT".AGG1_FU AND ("PLC_DATA".SMC_SILO_AG1 = "C#7_RD_RUN".SMX_AG1) AND ("PLC_DATA".SMC_SILO_AG1 < "C#7_RD_RUN".SMT),   // "7.WEIGHT_PROCESS"
              MAN1 := "C#2_WB"."NN_CAN AG1" OR "XA_HET_AGG",
              FAU := "C#2_WB".F2_SW_PAU OR "C#2_WB".SW_PA_AG1 OR ("C#6_WD_CALIB".XUNG_AG1 = 32767.0),
              FU_IN := "C#2_WB".NN_FU_AG1,
              X_CLOCK := "Clock_10Hz",
              EMTY_IN := "PLC_BIT".WAG1_EM,
              XNC_AUT := true,
              SV_IN := "C#4_WD_WEIGHT".SV_AG1,
              W_IN := "6.1.WAGG1".W_OUT1,
              W_RTD := "C#3_WD_SILO".AG1_KL_RTD,
              W_TR := "C#3_WD_SILO".AG1_SS_TREN,
              W_DU := "C#3_WD_SILO".AG1_SS_DUOI,
              T_ON := "C#3_WD_SILO".AG1_TG_ON_CAN,
              T_OFF := "C#3_WD_SILO".AG1_TG_OFF_CAN,
              T_DL := "C#3_WD_SILO".AG1_TG_ODC,
              PV_OUT => "C#7_RD_RUN".PV_AG1,
              PVM_OUT => "C#7_RD_RUN".PVM_AG1,
              FU_OUT => "PLC_BIT".AGG1_FU,
              EM_OUT => "7.1.AGG1".EM_OUT,
              W_OVER => "7.1.AGG1".W_OVER,
              Q_OUT1 => "C#1_RB"."CAN AG1",
              STA_RUN => "7.1.AGG1".STA_RUN);
   #_w2 := "PLC_BIT".AGG1_FU AND NOT "P_AGG1_FU";   // rising edge of "PLC_BIT".AGG1_FU
   "P_AGG1_FU" := "PLC_BIT".AGG1_FU;
   IF (#_w2 OR ("P_RUN" AND "PLC_BIT".AGG1_FU)) AND NOT "C#1_RB"."XA W_AG1" AND ("C#4_WD_WEIGHT".SV_AG1 <> 0.0) AND ("PLC_DATA".SMC_SILO_AG1 = "C#7_RD_RUN".SMX_AG1) THEN
       "PLC_DATA".SMC_SILO_AG1 := "PLC_DATA".SMC_SILO_AG1 + 1.0;
   END_IF;
   "C#1_RB".TTC_AG1 := "7.1.AGG1".STA_RUN;
END_REGION

REGION Network 2: CAN COT LIEU AGG2
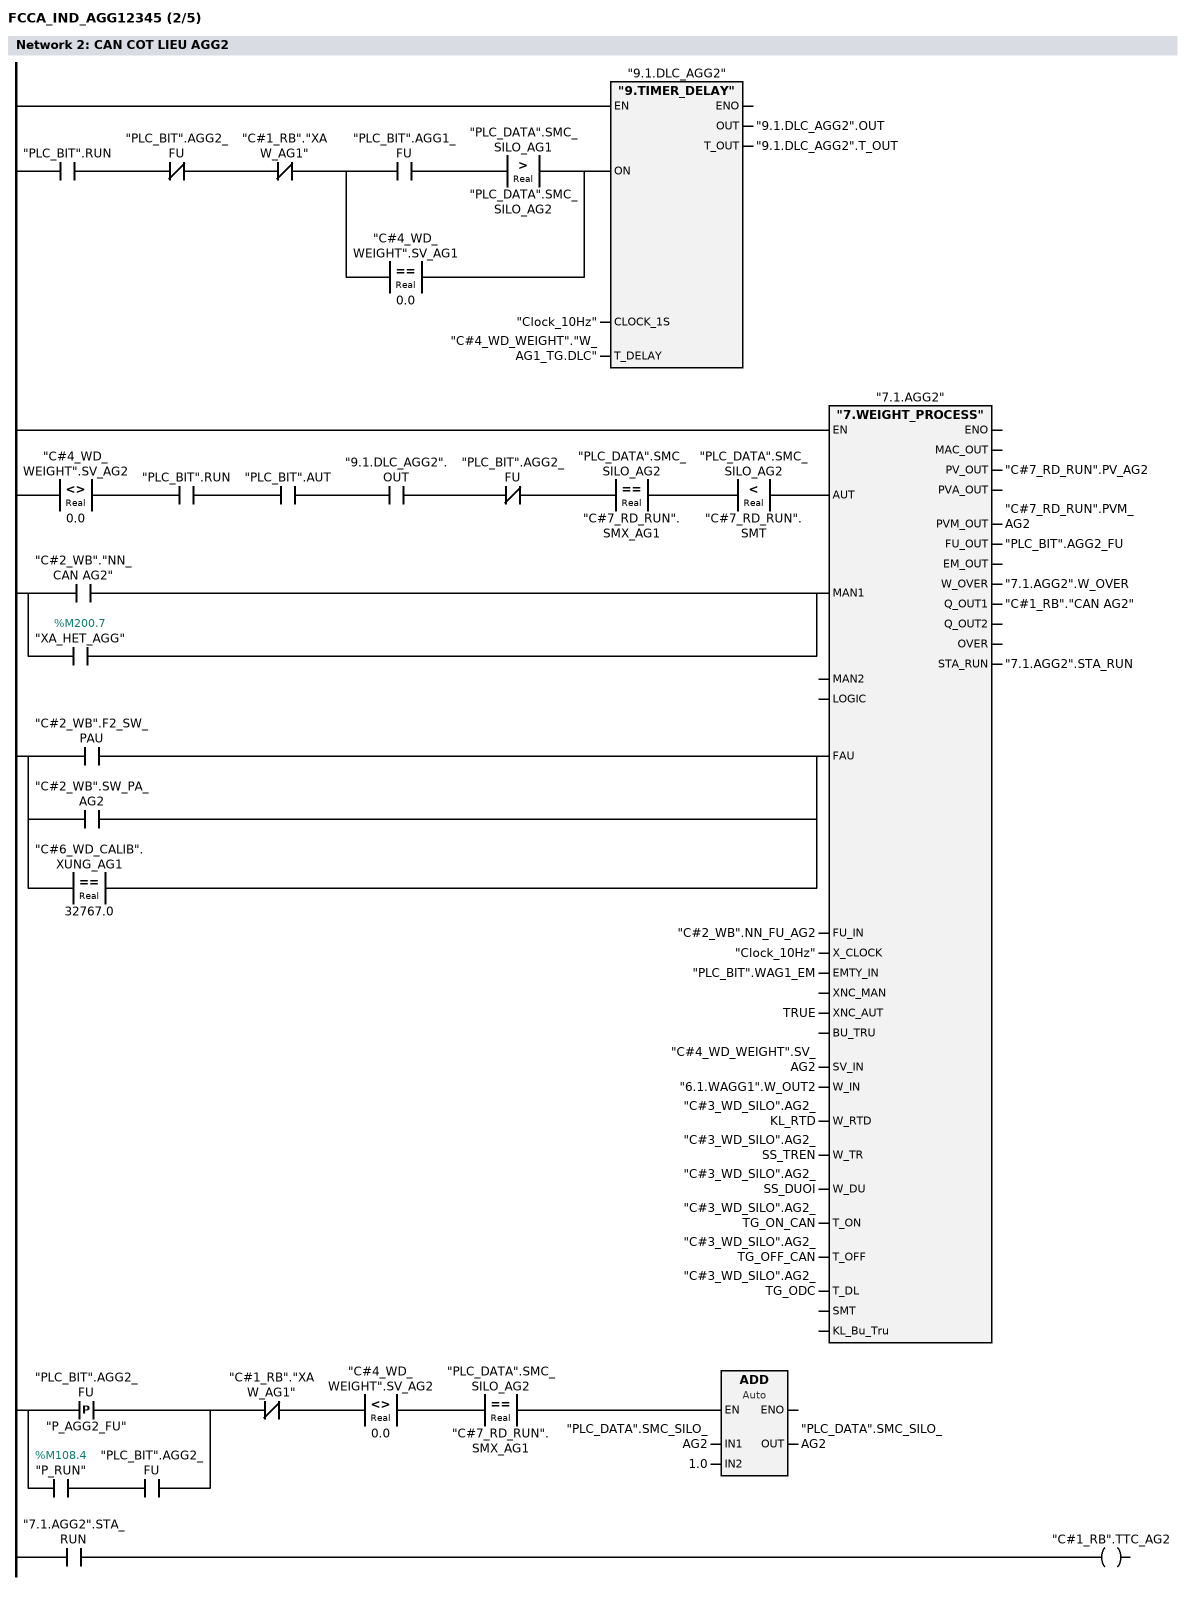
   RUNG wire#powerrail
      "9.1.DLC_AGG2"(ON := wire#w2, CLOCK_1S := "Clock_10Hz", T_DELAY := "C#4_WD_WEIGHT"."W_AG1_TG.DLC", OUT => "9.1.DLC_AGG2".OUT, T_OUT => "9.1.DLC_AGG2".T_OUT)
   END_RUNG
   RUNG wire#powerrail
      Contact( "PLC_BIT".RUN )
      I_Contact( "PLC_BIT".AGG2_FU )
      I_Contact( "C#1_RB"."XA W_AG1" )
      wire#w1
      Contact( "PLC_BIT".AGG1_FU )
      { S7_Templates := "SrcType := Real" } GT_Contact(in1 := "PLC_DATA".SMC_SILO_AG1, in2 := "PLC_DATA".SMC_SILO_AG2)
   END_RUNG wire#w2
   RUNG wire#w1
      { S7_Templates := "SrcType := Real" } EQ_Contact(in1 := "C#4_WD_WEIGHT".SV_AG1, in2 := 0.0)
   END_RUNG wire#w2
   RUNG wire#powerrail
      "7.1.AGG2"(AUT := wire#w3, MAN1 := wire#w4, FAU := wire#w5, MAN2 :=, LOGIC :=, FU_IN := "C#2_WB".NN_FU_AG2, X_CLOCK := "Clock_10Hz", EMTY_IN := "PLC_BIT".WAG1_EM, XNC_MAN :=, XNC_AUT := TRUE, BU_TRU :=, SV_IN := "C#4_WD_WEIGHT".SV_AG2, W_IN := "6.1.WAGG1".W_OUT2, W_RTD := "C#3_WD_SILO".AG2_KL_RTD, W_TR := "C#3_WD_SILO".AG2_SS_TREN, W_DU := "C#3_WD_SILO".AG2_SS_DUOI, T_ON := "C#3_WD_SILO".AG2_TG_ON_CAN, T_OFF := "C#3_WD_SILO".AG2_TG_OFF_CAN, T_DL := "C#3_WD_SILO".AG2_TG_ODC, SMT :=, KL_Bu_Tru :=, MAC_OUT =>, PV_OUT => "C#7_RD_RUN".PV_AG2, PVA_OUT =>, PVM_OUT => "C#7_RD_RUN".PVM_AG2, FU_OUT => "PLC_BIT".AGG2_FU, EM_OUT =>, W_OVER => "7.1.AGG2".W_OVER, Q_OUT1 => "C#1_RB"."CAN AG2", Q_OUT2 =>, OVER =>, STA_RUN => "7.1.AGG2".STA_RUN)
   END_RUNG
   RUNG wire#powerrail
      { S7_Templates := "SrcType := Real" } NE_Contact(in1 := "C#4_WD_WEIGHT".SV_AG2, in2 := 0.0)
      Contact( "PLC_BIT".RUN )
      Contact( "PLC_BIT".AUT )
      Contact( "9.1.DLC_AGG2".OUT )
      I_Contact( "PLC_BIT".AGG2_FU )
      { S7_Templates := "SrcType := Real" } EQ_Contact(in1 := "PLC_DATA".SMC_SILO_AG2, in2 := "C#7_RD_RUN".SMX_AG1)
      { S7_Templates := "SrcType := Real" } LT_Contact(in1 := "PLC_DATA".SMC_SILO_AG2, in2 := "C#7_RD_RUN".SMT)
   END_RUNG wire#w3
   RUNG wire#powerrail
      Contact( "C#2_WB"."NN_CAN AG2" )
   END_RUNG wire#w4
   RUNG wire#powerrail
      Contact( "XA_HET_AGG" )
   END_RUNG wire#w4
   RUNG wire#powerrail
      Contact( "C#2_WB".F2_SW_PAU )
   END_RUNG wire#w5
   RUNG wire#powerrail
      Contact( "C#2_WB".SW_PA_AG2 )
   END_RUNG wire#w5
   RUNG wire#powerrail
      { S7_Templates := "SrcType := Real" } EQ_Contact(in1 := "C#6_WD_CALIB".XUNG_AG1, in2 := 32767.0)
   END_RUNG wire#w5
   RUNG wire#powerrail
      P_Contact(operand := "PLC_BIT".AGG2_FU, bit := "P_AGG2_FU")
      wire#w6
      I_Contact( "C#1_RB"."XA W_AG1" )
      { S7_Templates := "SrcType := Real" } NE_Contact(in1 := "C#4_WD_WEIGHT".SV_AG2, in2 := 0.0)
      { S7_Templates := "SrcType := Real" } EQ_Contact(in1 := "PLC_DATA".SMC_SILO_AG2, in2 := "C#7_RD_RUN".SMX_AG1)
      Add(in1 := "PLC_DATA".SMC_SILO_AG2, in2 := 1.0, out => "PLC_DATA".SMC_SILO_AG2)
   END_RUNG
   RUNG wire#powerrail
      Contact( "P_RUN" )
      Contact( "PLC_BIT".AGG2_FU )
   END_RUNG wire#w6
   RUNG wire#powerrail
      Contact( "7.1.AGG2".STA_RUN )
      Coil( "C#1_RB".TTC_AG2 )
   END_RUNG
   // the same network as SCL:
   "9.1.DLC_AGG2"(ON := "PLC_BIT".RUN AND NOT "PLC_BIT".AGG2_FU AND NOT "C#1_RB"."XA W_AG1" AND (("PLC_BIT".AGG1_FU AND ("PLC_DATA".SMC_SILO_AG1 > "PLC_DATA".SMC_SILO_AG2)) OR ("C#4_WD_WEIGHT".SV_AG1 = 0.0)),   // "9.TIMER_DELAY"
                  CLOCK_1S := "Clock_10Hz",
                  T_DELAY := "C#4_WD_WEIGHT"."W_AG1_TG.DLC",
                  OUT => "9.1.DLC_AGG2".OUT,
                  T_OUT => "9.1.DLC_AGG2".T_OUT);
   "7.1.AGG2"(AUT := ("C#4_WD_WEIGHT".SV_AG2 <> 0.0) AND "PLC_BIT".RUN AND "PLC_BIT".AUT AND "9.1.DLC_AGG2".OUT AND NOT "PLC_BIT".AGG2_FU AND ("PLC_DATA".SMC_SILO_AG2 = "C#7_RD_RUN".SMX_AG1) AND ("PLC_DATA".SMC_SILO_AG2 < "C#7_RD_RUN".SMT),   // "7.WEIGHT_PROCESS"
              MAN1 := "C#2_WB"."NN_CAN AG2" OR "XA_HET_AGG",
              FAU := "C#2_WB".F2_SW_PAU OR "C#2_WB".SW_PA_AG2 OR ("C#6_WD_CALIB".XUNG_AG1 = 32767.0),
              FU_IN := "C#2_WB".NN_FU_AG2,
              X_CLOCK := "Clock_10Hz",
              EMTY_IN := "PLC_BIT".WAG1_EM,
              XNC_AUT := TRUE,
              SV_IN := "C#4_WD_WEIGHT".SV_AG2,
              W_IN := "6.1.WAGG1".W_OUT2,
              W_RTD := "C#3_WD_SILO".AG2_KL_RTD,
              W_TR := "C#3_WD_SILO".AG2_SS_TREN,
              W_DU := "C#3_WD_SILO".AG2_SS_DUOI,
              T_ON := "C#3_WD_SILO".AG2_TG_ON_CAN,
              T_OFF := "C#3_WD_SILO".AG2_TG_OFF_CAN,
              T_DL := "C#3_WD_SILO".AG2_TG_ODC,
              PV_OUT => "C#7_RD_RUN".PV_AG2,
              PVM_OUT => "C#7_RD_RUN".PVM_AG2,
              FU_OUT => "PLC_BIT".AGG2_FU,
              W_OVER => "7.1.AGG2".W_OVER,
              Q_OUT1 => "C#1_RB"."CAN AG2",
              STA_RUN => "7.1.AGG2".STA_RUN);
   #_w1 := "PLC_BIT".AGG2_FU AND NOT "P_AGG2_FU";   // rising edge of "PLC_BIT".AGG2_FU
   "P_AGG2_FU" := "PLC_BIT".AGG2_FU;
   IF (#_w1 OR ("P_RUN" AND "PLC_BIT".AGG2_FU)) AND NOT "C#1_RB"."XA W_AG1" AND ("C#4_WD_WEIGHT".SV_AG2 <> 0.0) AND ("PLC_DATA".SMC_SILO_AG2 = "C#7_RD_RUN".SMX_AG1) THEN
       "PLC_DATA".SMC_SILO_AG2 := "PLC_DATA".SMC_SILO_AG2 + 1.0;
   END_IF;
   "C#1_RB".TTC_AG2 := "7.1.AGG2".STA_RUN;
END_REGION

REGION Network 3: CAN COT LIEU AGG3
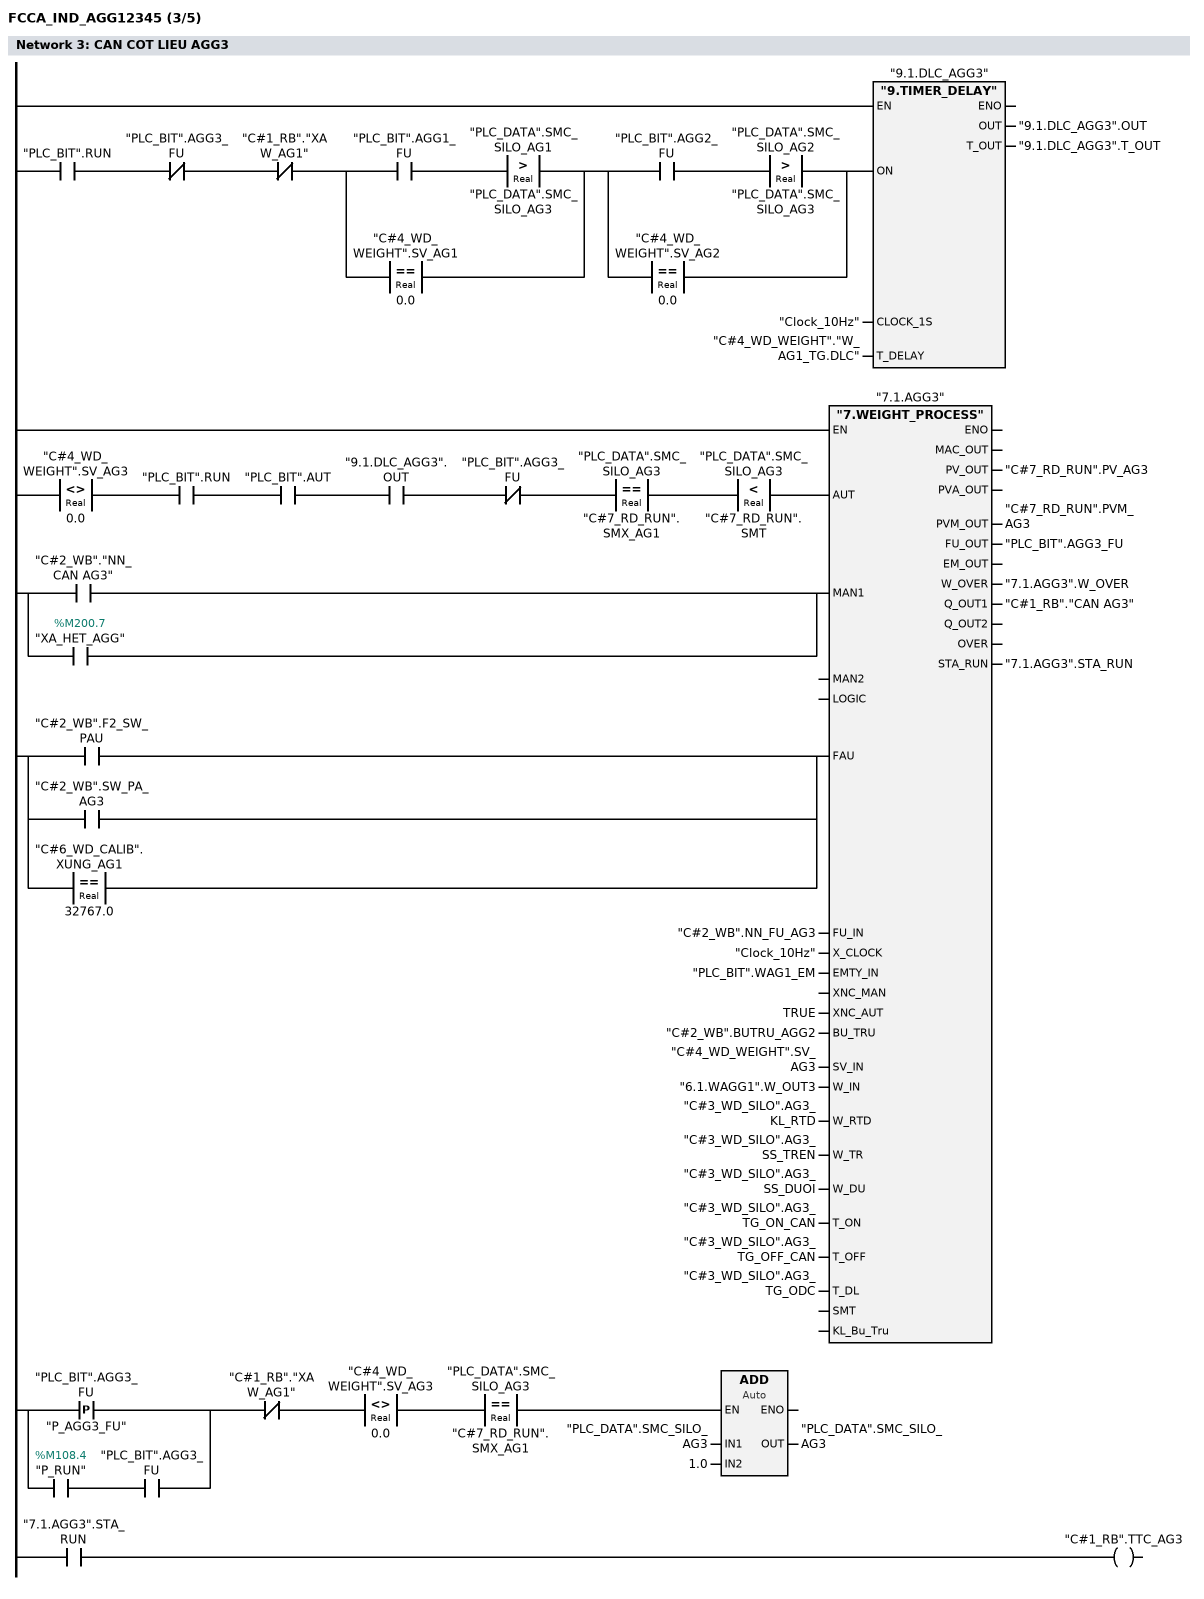
   RUNG wire#powerrail
      "9.1.DLC_AGG3"(ON := wire#w3, CLOCK_1S := "Clock_10Hz", T_DELAY := "C#4_WD_WEIGHT"."W_AG1_TG.DLC", OUT => "9.1.DLC_AGG3".OUT, T_OUT => "9.1.DLC_AGG3".T_OUT)
   END_RUNG
   RUNG wire#powerrail
      Contact( "PLC_BIT".RUN )
      I_Contact( "PLC_BIT".AGG3_FU )
      I_Contact( "C#1_RB"."XA W_AG1" )
      wire#w1
      Contact( "PLC_BIT".AGG1_FU )
      { S7_Templates := "SrcType := Real" } GT_Contact(in1 := "PLC_DATA".SMC_SILO_AG1, in2 := "PLC_DATA".SMC_SILO_AG3)
      wire#w2
      Contact( "PLC_BIT".AGG2_FU )
      { S7_Templates := "SrcType := Real" } GT_Contact(in1 := "PLC_DATA".SMC_SILO_AG2, in2 := "PLC_DATA".SMC_SILO_AG3)
   END_RUNG wire#w3
   RUNG wire#w1
      { S7_Templates := "SrcType := Real" } EQ_Contact(in1 := "C#4_WD_WEIGHT".SV_AG1, in2 := 0.0)
   END_RUNG wire#w2
   RUNG wire#w2
      { S7_Templates := "SrcType := Real" } EQ_Contact(in1 := "C#4_WD_WEIGHT".SV_AG2, in2 := 0.0)
   END_RUNG wire#w3
   RUNG wire#powerrail
      "7.1.AGG3"(AUT := wire#w4, MAN1 := wire#w5, FAU := wire#w6, MAN2 :=, LOGIC :=, FU_IN := "C#2_WB".NN_FU_AG3, X_CLOCK := "Clock_10Hz", EMTY_IN := "PLC_BIT".WAG1_EM, XNC_MAN :=, XNC_AUT := TRUE, BU_TRU := "C#2_WB".BUTRU_AGG2, SV_IN := "C#4_WD_WEIGHT".SV_AG3, W_IN := "6.1.WAGG1".W_OUT3, W_RTD := "C#3_WD_SILO".AG3_KL_RTD, W_TR := "C#3_WD_SILO".AG3_SS_TREN, W_DU := "C#3_WD_SILO".AG3_SS_DUOI, T_ON := "C#3_WD_SILO".AG3_TG_ON_CAN, T_OFF := "C#3_WD_SILO".AG3_TG_OFF_CAN, T_DL := "C#3_WD_SILO".AG3_TG_ODC, SMT :=, KL_Bu_Tru :=, MAC_OUT =>, PV_OUT => "C#7_RD_RUN".PV_AG3, PVA_OUT =>, PVM_OUT => "C#7_RD_RUN".PVM_AG3, FU_OUT => "PLC_BIT".AGG3_FU, EM_OUT =>, W_OVER => "7.1.AGG3".W_OVER, Q_OUT1 => "C#1_RB"."CAN AG3", Q_OUT2 =>, OVER =>, STA_RUN => "7.1.AGG3".STA_RUN)
   END_RUNG
   RUNG wire#powerrail
      { S7_Templates := "SrcType := Real" } NE_Contact(in1 := "C#4_WD_WEIGHT".SV_AG3, in2 := 0.0)
      Contact( "PLC_BIT".RUN )
      Contact( "PLC_BIT".AUT )
      Contact( "9.1.DLC_AGG3".OUT )
      I_Contact( "PLC_BIT".AGG3_FU )
      { S7_Templates := "SrcType := Real" } EQ_Contact(in1 := "PLC_DATA".SMC_SILO_AG3, in2 := "C#7_RD_RUN".SMX_AG1)
      { S7_Templates := "SrcType := Real" } LT_Contact(in1 := "PLC_DATA".SMC_SILO_AG3, in2 := "C#7_RD_RUN".SMT)
   END_RUNG wire#w4
   RUNG wire#powerrail
      Contact( "C#2_WB"."NN_CAN AG3" )
   END_RUNG wire#w5
   RUNG wire#powerrail
      Contact( "XA_HET_AGG" )
   END_RUNG wire#w5
   RUNG wire#powerrail
      Contact( "C#2_WB".F2_SW_PAU )
   END_RUNG wire#w6
   RUNG wire#powerrail
      Contact( "C#2_WB".SW_PA_AG3 )
   END_RUNG wire#w6
   RUNG wire#powerrail
      { S7_Templates := "SrcType := Real" } EQ_Contact(in1 := "C#6_WD_CALIB".XUNG_AG1, in2 := 32767.0)
   END_RUNG wire#w6
   RUNG wire#powerrail
      P_Contact(operand := "PLC_BIT".AGG3_FU, bit := "P_AGG3_FU")
      wire#w7
      I_Contact( "C#1_RB"."XA W_AG1" )
      { S7_Templates := "SrcType := Real" } NE_Contact(in1 := "C#4_WD_WEIGHT".SV_AG3, in2 := 0.0)
      { S7_Templates := "SrcType := Real" } EQ_Contact(in1 := "PLC_DATA".SMC_SILO_AG3, in2 := "C#7_RD_RUN".SMX_AG1)
      Add(in1 := "PLC_DATA".SMC_SILO_AG3, in2 := 1.0, out => "PLC_DATA".SMC_SILO_AG3)
   END_RUNG
   RUNG wire#powerrail
      Contact( "P_RUN" )
      Contact( "PLC_BIT".AGG3_FU )
   END_RUNG wire#w7
   RUNG wire#powerrail
      Contact( "7.1.AGG3".STA_RUN )
      Coil( "C#1_RB".TTC_AG3 )
   END_RUNG
   // the same network as SCL:
   "9.1.DLC_AGG3"(ON := "PLC_BIT".RUN AND NOT "PLC_BIT".AGG3_FU AND NOT "C#1_RB"."XA W_AG1" AND (("PLC_BIT".AGG1_FU AND ("PLC_DATA".SMC_SILO_AG1 > "PLC_DATA".SMC_SILO_AG3)) OR ("C#4_WD_WEIGHT".SV_AG1 = 0.0)) AND (("PLC_BIT".AGG2_FU AND ("PLC_DATA".SMC_SILO_AG2 > "PLC_DATA".SMC_SILO_AG3)) OR ("C#4_WD_WEIGHT".SV_AG2 = 0.0)),   // "9.TIMER_DELAY"
                  CLOCK_1S := "Clock_10Hz",
                  T_DELAY := "C#4_WD_WEIGHT"."W_AG1_TG.DLC",
                  OUT => "9.1.DLC_AGG3".OUT,
                  T_OUT => "9.1.DLC_AGG3".T_OUT);
   "7.1.AGG3"(AUT := ("C#4_WD_WEIGHT".SV_AG3 <> 0.0) AND "PLC_BIT".RUN AND "PLC_BIT".AUT AND "9.1.DLC_AGG3".OUT AND NOT "PLC_BIT".AGG3_FU AND ("PLC_DATA".SMC_SILO_AG3 = "C#7_RD_RUN".SMX_AG1) AND ("PLC_DATA".SMC_SILO_AG3 < "C#7_RD_RUN".SMT),   // "7.WEIGHT_PROCESS"
              MAN1 := "C#2_WB"."NN_CAN AG3" OR "XA_HET_AGG",
              FAU := "C#2_WB".F2_SW_PAU OR "C#2_WB".SW_PA_AG3 OR ("C#6_WD_CALIB".XUNG_AG1 = 32767.0),
              FU_IN := "C#2_WB".NN_FU_AG3,
              X_CLOCK := "Clock_10Hz",
              EMTY_IN := "PLC_BIT".WAG1_EM,
              XNC_AUT := TRUE,
              BU_TRU := "C#2_WB".BUTRU_AGG2,
              SV_IN := "C#4_WD_WEIGHT".SV_AG3,
              W_IN := "6.1.WAGG1".W_OUT3,
              W_RTD := "C#3_WD_SILO".AG3_KL_RTD,
              W_TR := "C#3_WD_SILO".AG3_SS_TREN,
              W_DU := "C#3_WD_SILO".AG3_SS_DUOI,
              T_ON := "C#3_WD_SILO".AG3_TG_ON_CAN,
              T_OFF := "C#3_WD_SILO".AG3_TG_OFF_CAN,
              T_DL := "C#3_WD_SILO".AG3_TG_ODC,
              PV_OUT => "C#7_RD_RUN".PV_AG3,
              PVM_OUT => "C#7_RD_RUN".PVM_AG3,
              FU_OUT => "PLC_BIT".AGG3_FU,
              W_OVER => "7.1.AGG3".W_OVER,
              Q_OUT1 => "C#1_RB"."CAN AG3",
              STA_RUN => "7.1.AGG3".STA_RUN);
   #_w1 := "PLC_BIT".AGG3_FU AND NOT "P_AGG3_FU";   // rising edge of "PLC_BIT".AGG3_FU
   "P_AGG3_FU" := "PLC_BIT".AGG3_FU;
   IF (#_w1 OR ("P_RUN" AND "PLC_BIT".AGG3_FU)) AND NOT "C#1_RB"."XA W_AG1" AND ("C#4_WD_WEIGHT".SV_AG3 <> 0.0) AND ("PLC_DATA".SMC_SILO_AG3 = "C#7_RD_RUN".SMX_AG1) THEN
       "PLC_DATA".SMC_SILO_AG3 := "PLC_DATA".SMC_SILO_AG3 + 1.0;
   END_IF;
   "C#1_RB".TTC_AG3 := "7.1.AGG3".STA_RUN;
END_REGION

REGION Network 4: CAN COT LIEU AGG4
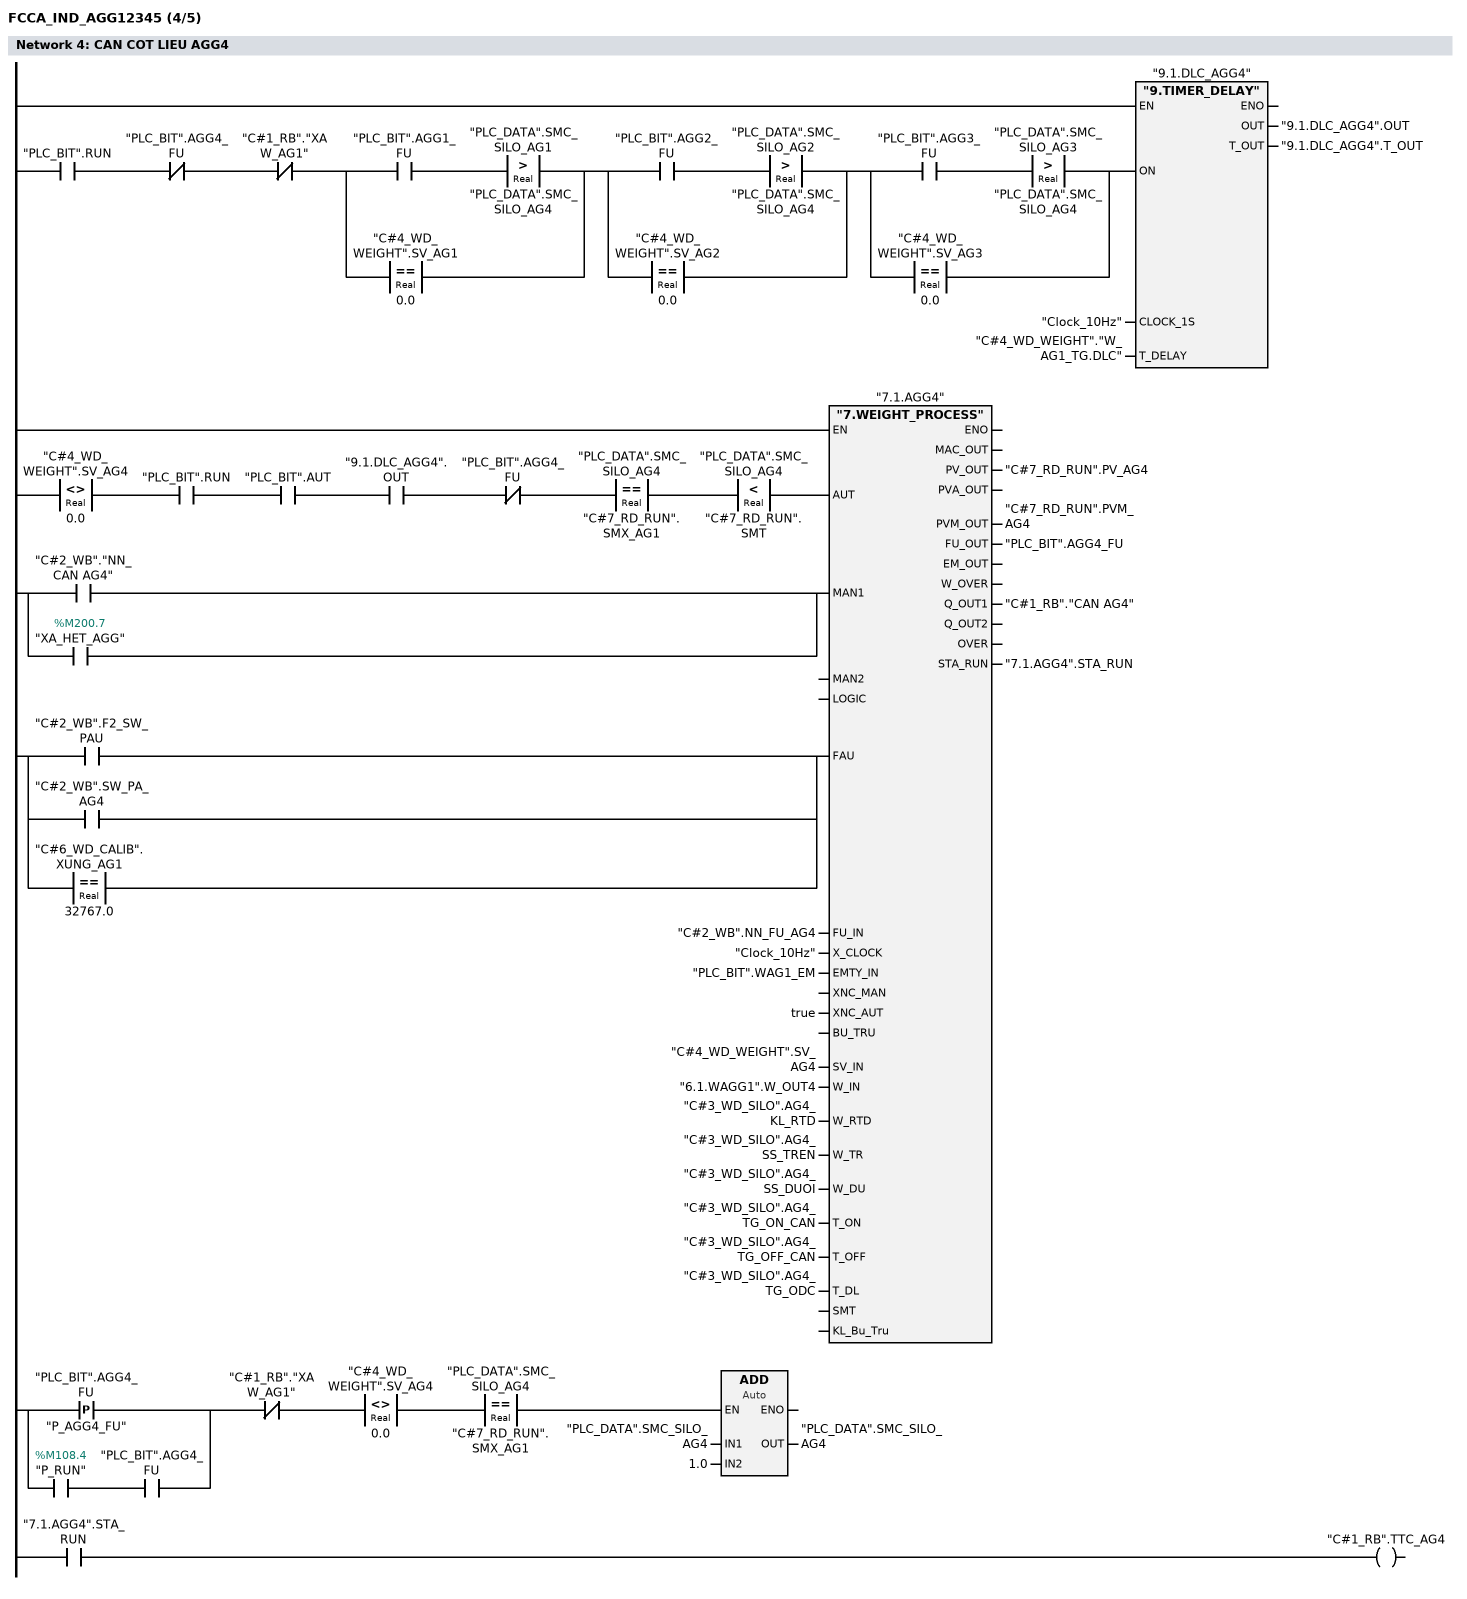
   RUNG wire#powerrail
      "9.1.DLC_AGG4"(ON := wire#w4, CLOCK_1S := "Clock_10Hz", T_DELAY := "C#4_WD_WEIGHT"."W_AG1_TG.DLC", OUT => "9.1.DLC_AGG4".OUT, T_OUT => "9.1.DLC_AGG4".T_OUT)
   END_RUNG
   RUNG wire#powerrail
      Contact( "PLC_BIT".RUN )
      I_Contact( "PLC_BIT".AGG4_FU )
      I_Contact( "C#1_RB"."XA W_AG1" )
      wire#w1
      Contact( "PLC_BIT".AGG1_FU )
      { S7_Templates := "SrcType := Real" } GT_Contact(in1 := "PLC_DATA".SMC_SILO_AG1, in2 := "PLC_DATA".SMC_SILO_AG4)
      wire#w2
      Contact( "PLC_BIT".AGG2_FU )
      { S7_Templates := "SrcType := Real" } GT_Contact(in1 := "PLC_DATA".SMC_SILO_AG2, in2 := "PLC_DATA".SMC_SILO_AG4)
      wire#w3
      Contact( "PLC_BIT".AGG3_FU )
      { S7_Templates := "SrcType := Real" } GT_Contact(in1 := "PLC_DATA".SMC_SILO_AG3, in2 := "PLC_DATA".SMC_SILO_AG4)
   END_RUNG wire#w4
   RUNG wire#w1
      { S7_Templates := "SrcType := Real" } EQ_Contact(in1 := "C#4_WD_WEIGHT".SV_AG1, in2 := 0.0)
   END_RUNG wire#w2
   RUNG wire#w2
      { S7_Templates := "SrcType := Real" } EQ_Contact(in1 := "C#4_WD_WEIGHT".SV_AG2, in2 := 0.0)
   END_RUNG wire#w3
   RUNG wire#w3
      { S7_Templates := "SrcType := Real" } EQ_Contact(in1 := "C#4_WD_WEIGHT".SV_AG3, in2 := 0.0)
   END_RUNG wire#w4
   RUNG wire#powerrail
      "7.1.AGG4"(AUT := wire#w5, MAN1 := wire#w6, FAU := wire#w7, MAN2 :=, LOGIC :=, FU_IN := "C#2_WB".NN_FU_AG4, X_CLOCK := "Clock_10Hz", EMTY_IN := "PLC_BIT".WAG1_EM, XNC_MAN :=, XNC_AUT := true, BU_TRU :=, SV_IN := "C#4_WD_WEIGHT".SV_AG4, W_IN := "6.1.WAGG1".W_OUT4, W_RTD := "C#3_WD_SILO".AG4_KL_RTD, W_TR := "C#3_WD_SILO".AG4_SS_TREN, W_DU := "C#3_WD_SILO".AG4_SS_DUOI, T_ON := "C#3_WD_SILO".AG4_TG_ON_CAN, T_OFF := "C#3_WD_SILO".AG4_TG_OFF_CAN, T_DL := "C#3_WD_SILO".AG4_TG_ODC, SMT :=, KL_Bu_Tru :=, MAC_OUT =>, PV_OUT => "C#7_RD_RUN".PV_AG4, PVA_OUT =>, PVM_OUT => "C#7_RD_RUN".PVM_AG4, FU_OUT => "PLC_BIT".AGG4_FU, EM_OUT =>, W_OVER =>, Q_OUT1 => "C#1_RB"."CAN AG4", Q_OUT2 =>, OVER =>, STA_RUN => "7.1.AGG4".STA_RUN)
   END_RUNG
   RUNG wire#powerrail
      { S7_Templates := "SrcType := Real" } NE_Contact(in1 := "C#4_WD_WEIGHT".SV_AG4, in2 := 0.0)
      Contact( "PLC_BIT".RUN )
      Contact( "PLC_BIT".AUT )
      Contact( "9.1.DLC_AGG4".OUT )
      I_Contact( "PLC_BIT".AGG4_FU )
      { S7_Templates := "SrcType := Real" } EQ_Contact(in1 := "PLC_DATA".SMC_SILO_AG4, in2 := "C#7_RD_RUN".SMX_AG1)
      { S7_Templates := "SrcType := Real" } LT_Contact(in1 := "PLC_DATA".SMC_SILO_AG4, in2 := "C#7_RD_RUN".SMT)
   END_RUNG wire#w5
   RUNG wire#powerrail
      Contact( "C#2_WB"."NN_CAN AG4" )
   END_RUNG wire#w6
   RUNG wire#powerrail
      Contact( "XA_HET_AGG" )
   END_RUNG wire#w6
   RUNG wire#powerrail
      Contact( "C#2_WB".F2_SW_PAU )
   END_RUNG wire#w7
   RUNG wire#powerrail
      Contact( "C#2_WB".SW_PA_AG4 )
   END_RUNG wire#w7
   RUNG wire#powerrail
      { S7_Templates := "SrcType := Real" } EQ_Contact(in1 := "C#6_WD_CALIB".XUNG_AG1, in2 := 32767.0)
   END_RUNG wire#w7
   RUNG wire#powerrail
      P_Contact(operand := "PLC_BIT".AGG4_FU, bit := "P_AGG4_FU")
      wire#w8
      I_Contact( "C#1_RB"."XA W_AG1" )
      { S7_Templates := "SrcType := Real" } NE_Contact(in1 := "C#4_WD_WEIGHT".SV_AG4, in2 := 0.0)
      { S7_Templates := "SrcType := Real" } EQ_Contact(in1 := "PLC_DATA".SMC_SILO_AG4, in2 := "C#7_RD_RUN".SMX_AG1)
      Add(in1 := "PLC_DATA".SMC_SILO_AG4, in2 := 1.0, out => "PLC_DATA".SMC_SILO_AG4)
   END_RUNG
   RUNG wire#powerrail
      Contact( "P_RUN" )
      Contact( "PLC_BIT".AGG4_FU )
   END_RUNG wire#w8
   RUNG wire#powerrail
      Contact( "7.1.AGG4".STA_RUN )
      Coil( "C#1_RB".TTC_AG4 )
   END_RUNG
   // the same network as SCL:
   "9.1.DLC_AGG4"(ON := "PLC_BIT".RUN AND NOT "PLC_BIT".AGG4_FU AND NOT "C#1_RB"."XA W_AG1" AND (("PLC_BIT".AGG1_FU AND ("PLC_DATA".SMC_SILO_AG1 > "PLC_DATA".SMC_SILO_AG4)) OR ("C#4_WD_WEIGHT".SV_AG1 = 0.0)) AND (("PLC_BIT".AGG2_FU AND ("PLC_DATA".SMC_SILO_AG2 > "PLC_DATA".SMC_SILO_AG4)) OR ("C#4_WD_WEIGHT".SV_AG2 = 0.0)) AND (("PLC_BIT".AGG3_FU AND ("PLC_DATA".SMC_SILO_AG3 > "PLC_DATA".SMC_SILO_AG4)) OR ("C#4_WD_WEIGHT".SV_AG3 = 0.0)),   // "9.TIMER_DELAY"
                  CLOCK_1S := "Clock_10Hz",
                  T_DELAY := "C#4_WD_WEIGHT"."W_AG1_TG.DLC",
                  OUT => "9.1.DLC_AGG4".OUT,
                  T_OUT => "9.1.DLC_AGG4".T_OUT);
   "7.1.AGG4"(AUT := ("C#4_WD_WEIGHT".SV_AG4 <> 0.0) AND "PLC_BIT".RUN AND "PLC_BIT".AUT AND "9.1.DLC_AGG4".OUT AND NOT "PLC_BIT".AGG4_FU AND ("PLC_DATA".SMC_SILO_AG4 = "C#7_RD_RUN".SMX_AG1) AND ("PLC_DATA".SMC_SILO_AG4 < "C#7_RD_RUN".SMT),   // "7.WEIGHT_PROCESS"
              MAN1 := "C#2_WB"."NN_CAN AG4" OR "XA_HET_AGG",
              FAU := "C#2_WB".F2_SW_PAU OR "C#2_WB".SW_PA_AG4 OR ("C#6_WD_CALIB".XUNG_AG1 = 32767.0),
              FU_IN := "C#2_WB".NN_FU_AG4,
              X_CLOCK := "Clock_10Hz",
              EMTY_IN := "PLC_BIT".WAG1_EM,
              XNC_AUT := true,
              SV_IN := "C#4_WD_WEIGHT".SV_AG4,
              W_IN := "6.1.WAGG1".W_OUT4,
              W_RTD := "C#3_WD_SILO".AG4_KL_RTD,
              W_TR := "C#3_WD_SILO".AG4_SS_TREN,
              W_DU := "C#3_WD_SILO".AG4_SS_DUOI,
              T_ON := "C#3_WD_SILO".AG4_TG_ON_CAN,
              T_OFF := "C#3_WD_SILO".AG4_TG_OFF_CAN,
              T_DL := "C#3_WD_SILO".AG4_TG_ODC,
              PV_OUT => "C#7_RD_RUN".PV_AG4,
              PVM_OUT => "C#7_RD_RUN".PVM_AG4,
              FU_OUT => "PLC_BIT".AGG4_FU,
              Q_OUT1 => "C#1_RB"."CAN AG4",
              STA_RUN => "7.1.AGG4".STA_RUN);
   #_w1 := "PLC_BIT".AGG4_FU AND NOT "P_AGG4_FU";   // rising edge of "PLC_BIT".AGG4_FU
   "P_AGG4_FU" := "PLC_BIT".AGG4_FU;
   IF (#_w1 OR ("P_RUN" AND "PLC_BIT".AGG4_FU)) AND NOT "C#1_RB"."XA W_AG1" AND ("C#4_WD_WEIGHT".SV_AG4 <> 0.0) AND ("PLC_DATA".SMC_SILO_AG4 = "C#7_RD_RUN".SMX_AG1) THEN
       "PLC_DATA".SMC_SILO_AG4 := "PLC_DATA".SMC_SILO_AG4 + 1.0;
   END_IF;
   "C#1_RB".TTC_AG4 := "7.1.AGG4".STA_RUN;
END_REGION

REGION Network 5: Trạng thái cân Ag4
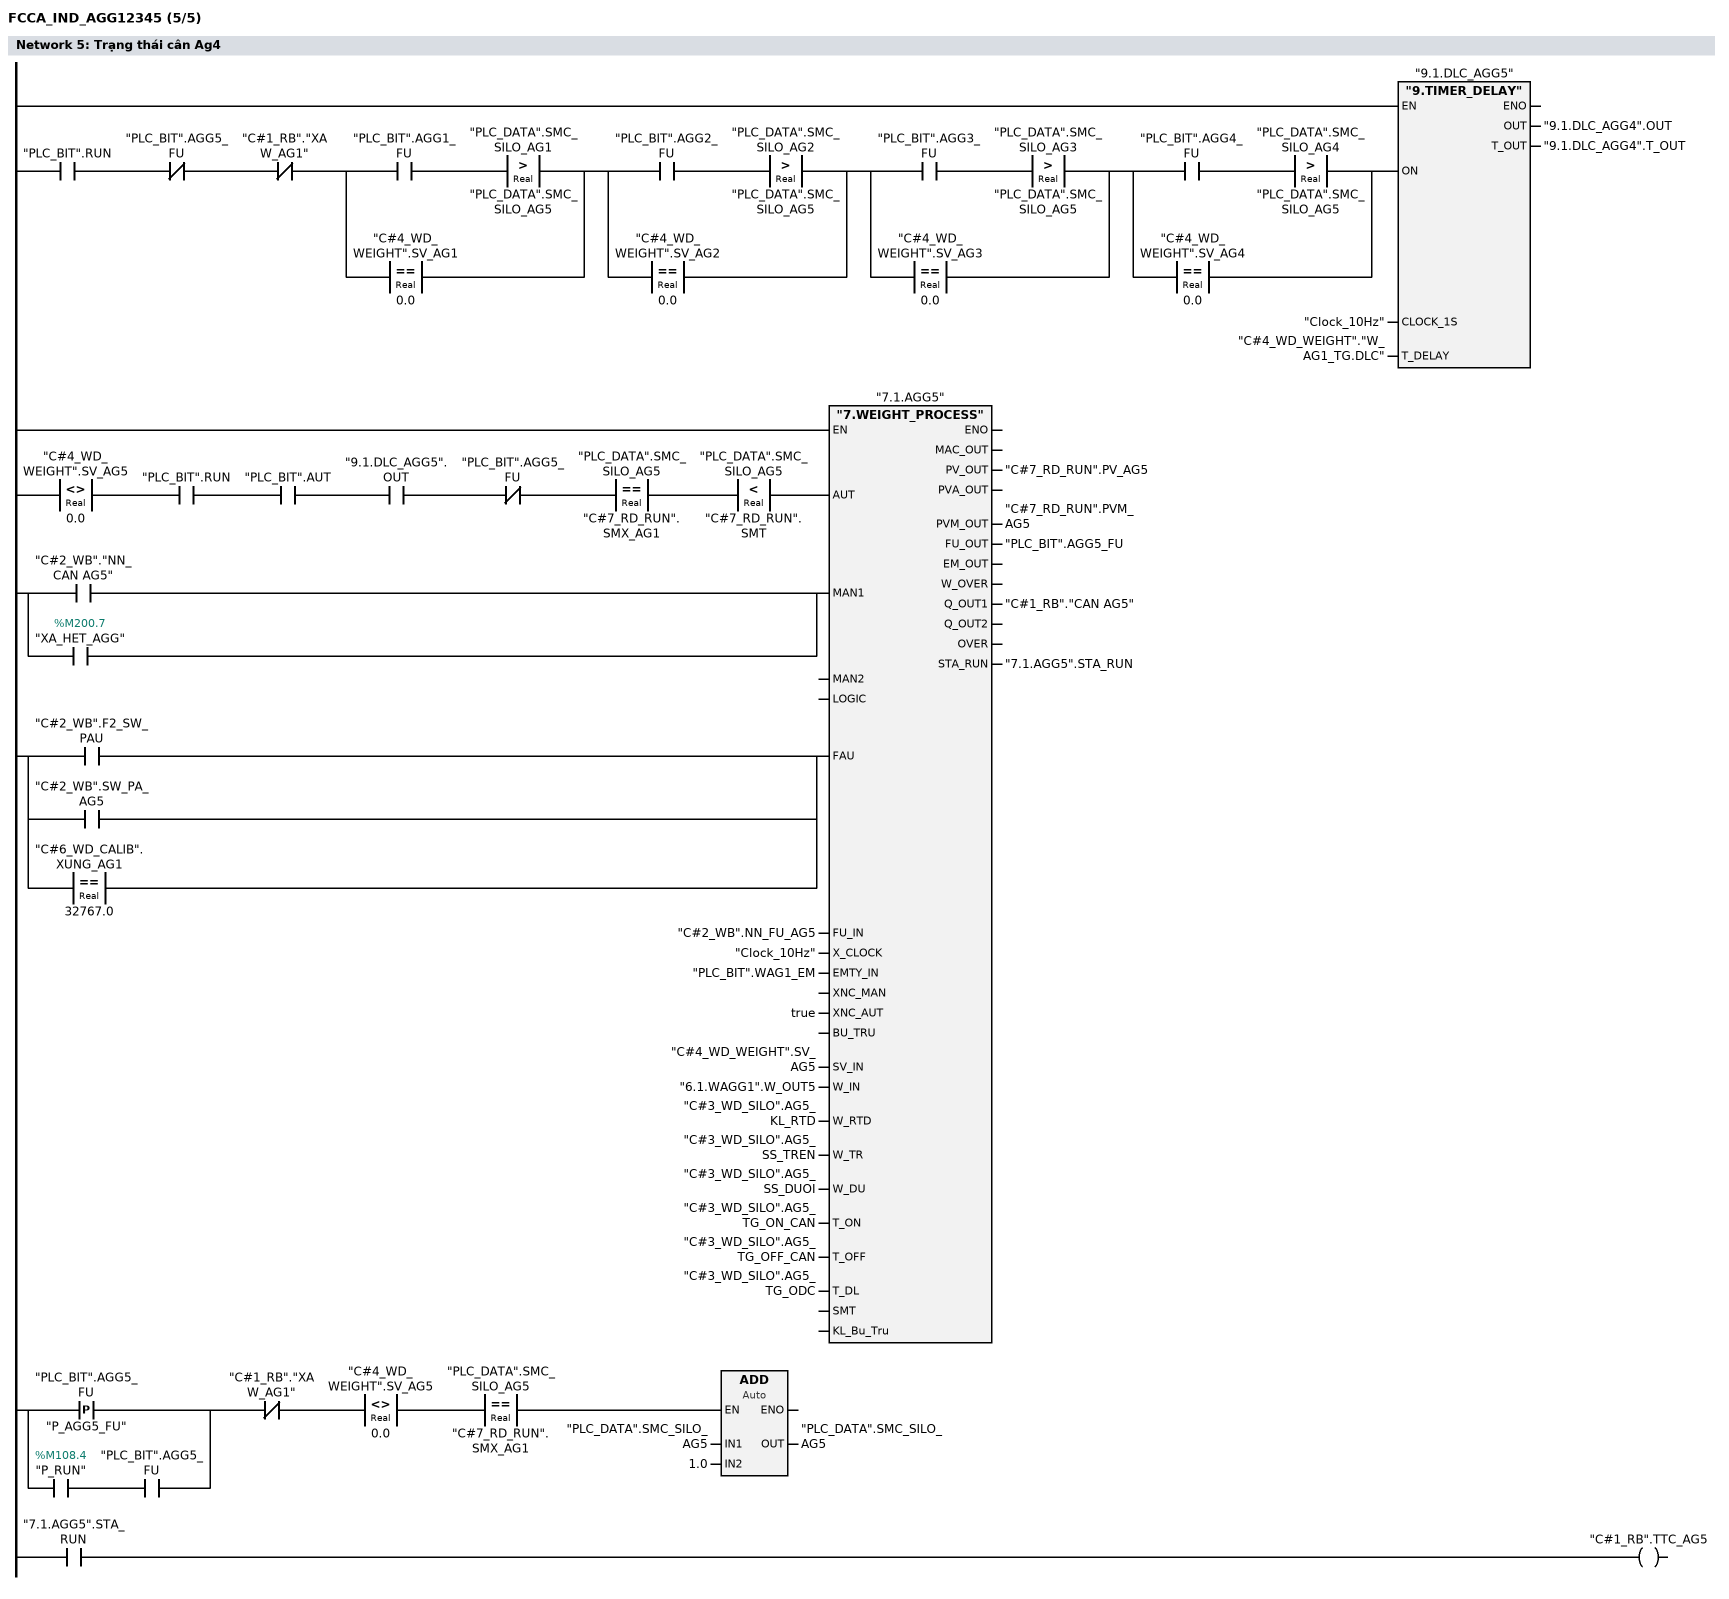
   RUNG wire#powerrail
      "9.1.DLC_AGG5"(ON := wire#w5, CLOCK_1S := "Clock_10Hz", T_DELAY := "C#4_WD_WEIGHT"."W_AG1_TG.DLC", OUT => "9.1.DLC_AGG4".OUT, T_OUT => "9.1.DLC_AGG4".T_OUT)
   END_RUNG
   RUNG wire#powerrail
      Contact( "PLC_BIT".RUN )
      I_Contact( "PLC_BIT".AGG5_FU )
      I_Contact( "C#1_RB"."XA W_AG1" )
      wire#w1
      Contact( "PLC_BIT".AGG1_FU )
      { S7_Templates := "SrcType := Real" } GT_Contact(in1 := "PLC_DATA".SMC_SILO_AG1, in2 := "PLC_DATA".SMC_SILO_AG5)
      wire#w2
      Contact( "PLC_BIT".AGG2_FU )
      { S7_Templates := "SrcType := Real" } GT_Contact(in1 := "PLC_DATA".SMC_SILO_AG2, in2 := "PLC_DATA".SMC_SILO_AG5)
      wire#w3
      Contact( "PLC_BIT".AGG3_FU )
      { S7_Templates := "SrcType := Real" } GT_Contact(in1 := "PLC_DATA".SMC_SILO_AG3, in2 := "PLC_DATA".SMC_SILO_AG5)
      wire#w4
      Contact( "PLC_BIT".AGG4_FU )
      { S7_Templates := "SrcType := Real" } GT_Contact(in1 := "PLC_DATA".SMC_SILO_AG4, in2 := "PLC_DATA".SMC_SILO_AG5)
   END_RUNG wire#w5
   RUNG wire#w1
      { S7_Templates := "SrcType := Real" } EQ_Contact(in1 := "C#4_WD_WEIGHT".SV_AG1, in2 := 0.0)
   END_RUNG wire#w2
   RUNG wire#w2
      { S7_Templates := "SrcType := Real" } EQ_Contact(in1 := "C#4_WD_WEIGHT".SV_AG2, in2 := 0.0)
   END_RUNG wire#w3
   RUNG wire#w3
      { S7_Templates := "SrcType := Real" } EQ_Contact(in1 := "C#4_WD_WEIGHT".SV_AG3, in2 := 0.0)
   END_RUNG wire#w4
   RUNG wire#w4
      { S7_Templates := "SrcType := Real" } EQ_Contact(in1 := "C#4_WD_WEIGHT".SV_AG4, in2 := 0.0)
   END_RUNG wire#w5
   RUNG wire#powerrail
      "7.1.AGG5"(AUT := wire#w6, MAN1 := wire#w7, FAU := wire#w8, MAN2 :=, LOGIC :=, FU_IN := "C#2_WB".NN_FU_AG5, X_CLOCK := "Clock_10Hz", EMTY_IN := "PLC_BIT".WAG1_EM, XNC_MAN :=, XNC_AUT := true, BU_TRU :=, SV_IN := "C#4_WD_WEIGHT".SV_AG5, W_IN := "6.1.WAGG1".W_OUT5, W_RTD := "C#3_WD_SILO".AG5_KL_RTD, W_TR := "C#3_WD_SILO".AG5_SS_TREN, W_DU := "C#3_WD_SILO".AG5_SS_DUOI, T_ON := "C#3_WD_SILO".AG5_TG_ON_CAN, T_OFF := "C#3_WD_SILO".AG5_TG_OFF_CAN, T_DL := "C#3_WD_SILO".AG5_TG_ODC, SMT :=, KL_Bu_Tru :=, MAC_OUT =>, PV_OUT => "C#7_RD_RUN".PV_AG5, PVA_OUT =>, PVM_OUT => "C#7_RD_RUN".PVM_AG5, FU_OUT => "PLC_BIT".AGG5_FU, EM_OUT =>, W_OVER =>, Q_OUT1 => "C#1_RB"."CAN AG5", Q_OUT2 =>, OVER =>, STA_RUN => "7.1.AGG5".STA_RUN)
   END_RUNG
   RUNG wire#powerrail
      { S7_Templates := "SrcType := Real" } NE_Contact(in1 := "C#4_WD_WEIGHT".SV_AG5, in2 := 0.0)
      Contact( "PLC_BIT".RUN )
      Contact( "PLC_BIT".AUT )
      Contact( "9.1.DLC_AGG5".OUT )
      I_Contact( "PLC_BIT".AGG5_FU )
      { S7_Templates := "SrcType := Real" } EQ_Contact(in1 := "PLC_DATA".SMC_SILO_AG5, in2 := "C#7_RD_RUN".SMX_AG1)
      { S7_Templates := "SrcType := Real" } LT_Contact(in1 := "PLC_DATA".SMC_SILO_AG5, in2 := "C#7_RD_RUN".SMT)
   END_RUNG wire#w6
   RUNG wire#powerrail
      Contact( "C#2_WB"."NN_CAN AG5" )
   END_RUNG wire#w7
   RUNG wire#powerrail
      Contact( "XA_HET_AGG" )
   END_RUNG wire#w7
   RUNG wire#powerrail
      Contact( "C#2_WB".F2_SW_PAU )
   END_RUNG wire#w8
   RUNG wire#powerrail
      Contact( "C#2_WB".SW_PA_AG5 )
   END_RUNG wire#w8
   RUNG wire#powerrail
      { S7_Templates := "SrcType := Real" } EQ_Contact(in1 := "C#6_WD_CALIB".XUNG_AG1, in2 := 32767.0)
   END_RUNG wire#w8
   RUNG wire#powerrail
      P_Contact(operand := "PLC_BIT".AGG5_FU, bit := "P_AGG5_FU")
      wire#w9
      I_Contact( "C#1_RB"."XA W_AG1" )
      { S7_Templates := "SrcType := Real" } NE_Contact(in1 := "C#4_WD_WEIGHT".SV_AG5, in2 := 0.0)
      { S7_Templates := "SrcType := Real" } EQ_Contact(in1 := "PLC_DATA".SMC_SILO_AG5, in2 := "C#7_RD_RUN".SMX_AG1)
      Add(in1 := "PLC_DATA".SMC_SILO_AG5, in2 := 1.0, out => "PLC_DATA".SMC_SILO_AG5)
   END_RUNG
   RUNG wire#powerrail
      Contact( "P_RUN" )
      Contact( "PLC_BIT".AGG5_FU )
   END_RUNG wire#w9
   RUNG wire#powerrail
      Contact( "7.1.AGG5".STA_RUN )
      Coil( "C#1_RB".TTC_AG5 )
   END_RUNG
   // the same network as SCL:
   "9.1.DLC_AGG5"(ON := "PLC_BIT".RUN AND NOT "PLC_BIT".AGG5_FU AND NOT "C#1_RB"."XA W_AG1" AND (("PLC_BIT".AGG1_FU AND ("PLC_DATA".SMC_SILO_AG1 > "PLC_DATA".SMC_SILO_AG5)) OR ("C#4_WD_WEIGHT".SV_AG1 = 0.0)) AND (("PLC_BIT".AGG2_FU AND ("PLC_DATA".SMC_SILO_AG2 > "PLC_DATA".SMC_SILO_AG5)) OR ("C#4_WD_WEIGHT".SV_AG2 = 0.0)) AND (("PLC_BIT".AGG3_FU AND ("PLC_DATA".SMC_SILO_AG3 > "PLC_DATA".SMC_SILO_AG5)) OR ("C#4_WD_WEIGHT".SV_AG3 = 0.0)) AND (("PLC_BIT".AGG4_FU AND ("PLC_DATA".SMC_SILO_AG4 > "PLC_DATA".SMC_SILO_AG5)) OR ("C#4_WD_WEIGHT".SV_AG4 = 0.0)),   // "9.TIMER_DELAY"
                  CLOCK_1S := "Clock_10Hz",
                  T_DELAY := "C#4_WD_WEIGHT"."W_AG1_TG.DLC",
                  OUT => "9.1.DLC_AGG4".OUT,
                  T_OUT => "9.1.DLC_AGG4".T_OUT);
   "7.1.AGG5"(AUT := ("C#4_WD_WEIGHT".SV_AG5 <> 0.0) AND "PLC_BIT".RUN AND "PLC_BIT".AUT AND "9.1.DLC_AGG5".OUT AND NOT "PLC_BIT".AGG5_FU AND ("PLC_DATA".SMC_SILO_AG5 = "C#7_RD_RUN".SMX_AG1) AND ("PLC_DATA".SMC_SILO_AG5 < "C#7_RD_RUN".SMT),   // "7.WEIGHT_PROCESS"
              MAN1 := "C#2_WB"."NN_CAN AG5" OR "XA_HET_AGG",
              FAU := "C#2_WB".F2_SW_PAU OR "C#2_WB".SW_PA_AG5 OR ("C#6_WD_CALIB".XUNG_AG1 = 32767.0),
              FU_IN := "C#2_WB".NN_FU_AG5,
              X_CLOCK := "Clock_10Hz",
              EMTY_IN := "PLC_BIT".WAG1_EM,
              XNC_AUT := true,
              SV_IN := "C#4_WD_WEIGHT".SV_AG5,
              W_IN := "6.1.WAGG1".W_OUT5,
              W_RTD := "C#3_WD_SILO".AG5_KL_RTD,
              W_TR := "C#3_WD_SILO".AG5_SS_TREN,
              W_DU := "C#3_WD_SILO".AG5_SS_DUOI,
              T_ON := "C#3_WD_SILO".AG5_TG_ON_CAN,
              T_OFF := "C#3_WD_SILO".AG5_TG_OFF_CAN,
              T_DL := "C#3_WD_SILO".AG5_TG_ODC,
              PV_OUT => "C#7_RD_RUN".PV_AG5,
              PVM_OUT => "C#7_RD_RUN".PVM_AG5,
              FU_OUT => "PLC_BIT".AGG5_FU,
              Q_OUT1 => "C#1_RB"."CAN AG5",
              STA_RUN => "7.1.AGG5".STA_RUN);
   #_w1 := "PLC_BIT".AGG5_FU AND NOT "P_AGG5_FU";   // rising edge of "PLC_BIT".AGG5_FU
   "P_AGG5_FU" := "PLC_BIT".AGG5_FU;
   IF (#_w1 OR ("P_RUN" AND "PLC_BIT".AGG5_FU)) AND NOT "C#1_RB"."XA W_AG1" AND ("C#4_WD_WEIGHT".SV_AG5 <> 0.0) AND ("PLC_DATA".SMC_SILO_AG5 = "C#7_RD_RUN".SMX_AG1) THEN
       "PLC_DATA".SMC_SILO_AG5 := "PLC_DATA".SMC_SILO_AG5 + 1.0;
   END_IF;
   "C#1_RB".TTC_AG5 := "7.1.AGG5".STA_RUN;
END_REGION
END_FUNCTION

FUNCTION "FCCA_IND_AGG1" : Void   // FC20, LAD
{ S7_Optimized_Access := 'TRUE' }
VERSION : 0.1
// stored: AutoNumber false, CodeModifiedDate 2026-01-15T16:25:53.7815162Z, CompileDate 2026-01-15T16:25:53.8212538Z, CreationDate 2026-01-15T16:24:02.4619467Z, HandleErrorsWithinBlock false, InterfaceModifiedDate 2026-01-10T08:55:50.3009267Z, IsConsistent true, IsIECCheckEnabled false, IsKnowHowProtected false, IsWriteProtected false, LibraryConformanceStatus Error: The block contains calls of single instances. Warning: The object contains access to global data blocks. Warning: The block contains direct access to inputs, outputs, bit memories, indirect access to the registry or indirect access to external memory areas that are unknown at the time of compilation., ModifiedDate 2026-01-15T16:25:53.7815162Z, ParameterModified 2026-01-10T08:55:50.3009267Z, PLCSimAdvancedSupport false, SetENOAutomatically False, StructureModified 2026-01-10T08:55:50.3009267Z, UDAEnableTagReadback false
BEGIN

REGION Network 1: Trạng thái cân AGG1
   // Đầu tiên nó sẽ đợi một khoảng thời gian gọi là Thời gian trễ cân, sau đó nó mới đủ điều kiện để cân
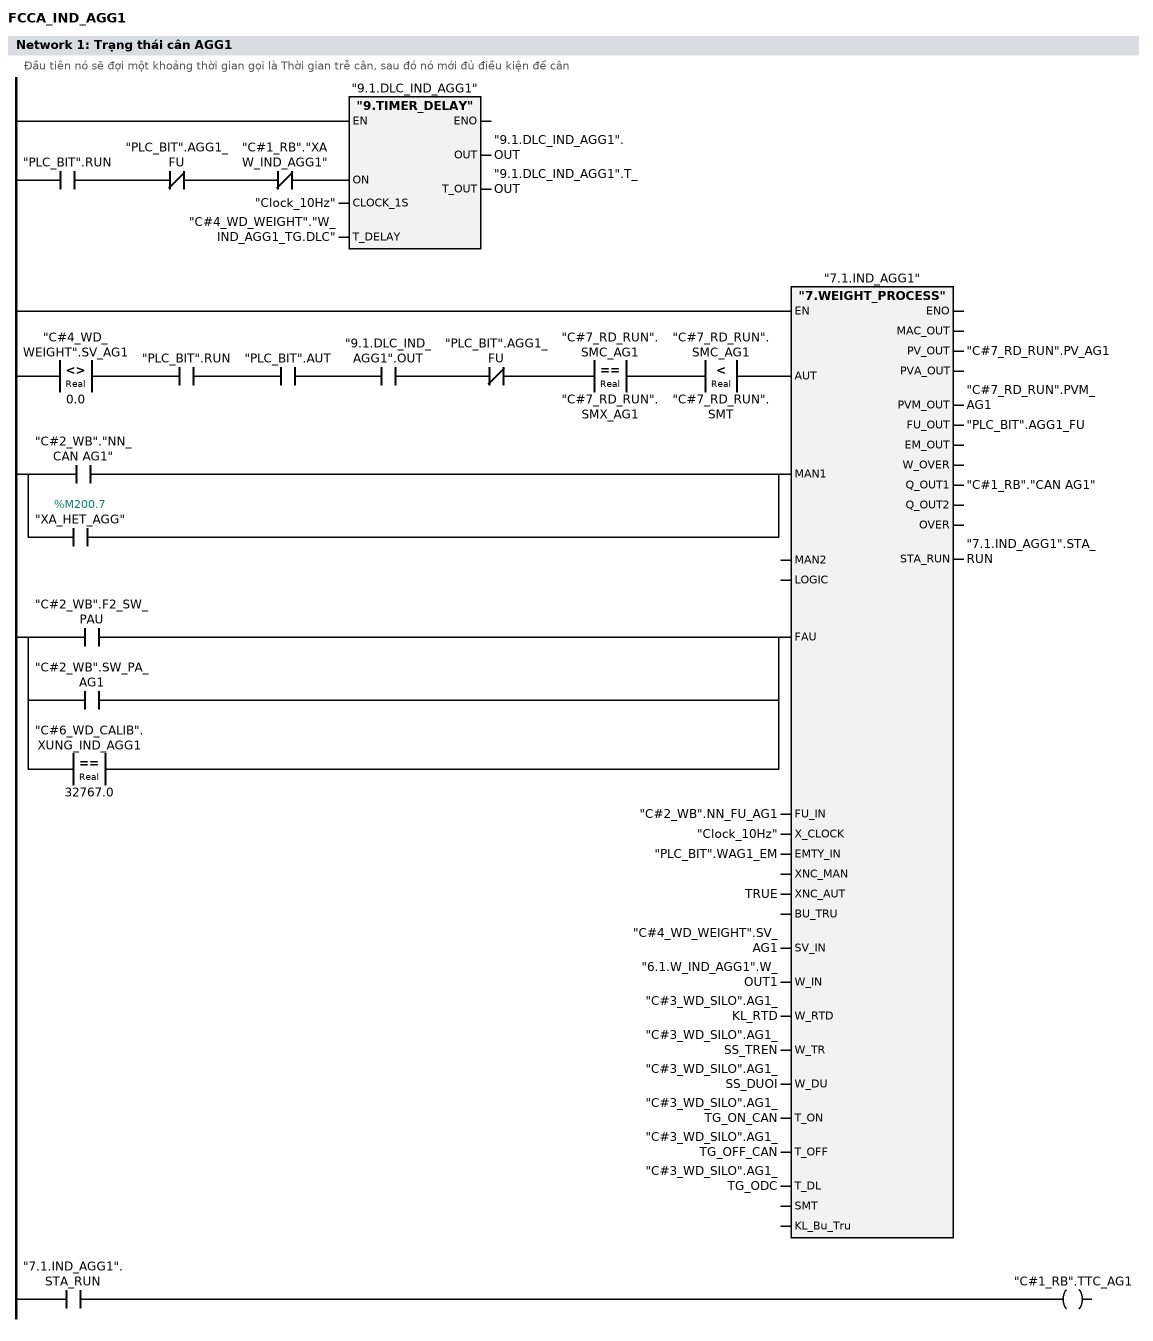
   RUNG wire#powerrail
      "9.1.DLC_IND_AGG1"(ON := wire#w1, CLOCK_1S := "Clock_10Hz", T_DELAY := "C#4_WD_WEIGHT"."W_IND_AGG1_TG.DLC", OUT => "9.1.DLC_IND_AGG1".OUT, T_OUT => "9.1.DLC_IND_AGG1".T_OUT)
   END_RUNG
   RUNG wire#powerrail
      Contact( "PLC_BIT".RUN )
      I_Contact( "PLC_BIT".AGG1_FU )
      I_Contact( "C#1_RB"."XA W_IND_AGG1" )
   END_RUNG wire#w1
   RUNG wire#powerrail
      "7.1.IND_AGG1"(AUT := wire#w2, MAN1 := wire#w3, FAU := wire#w4, MAN2 :=, LOGIC :=, FU_IN := "C#2_WB".NN_FU_AG1, X_CLOCK := "Clock_10Hz", EMTY_IN := "PLC_BIT".WAG1_EM, XNC_MAN :=, XNC_AUT := TRUE, BU_TRU :=, SV_IN := "C#4_WD_WEIGHT".SV_AG1, W_IN := "6.1.W_IND_AGG1".W_OUT1, W_RTD := "C#3_WD_SILO".AG1_KL_RTD, W_TR := "C#3_WD_SILO".AG1_SS_TREN, W_DU := "C#3_WD_SILO".AG1_SS_DUOI, T_ON := "C#3_WD_SILO".AG1_TG_ON_CAN, T_OFF := "C#3_WD_SILO".AG1_TG_OFF_CAN, T_DL := "C#3_WD_SILO".AG1_TG_ODC, SMT :=, KL_Bu_Tru :=, MAC_OUT =>, PV_OUT => "C#7_RD_RUN".PV_AG1, PVA_OUT =>, PVM_OUT => "C#7_RD_RUN".PVM_AG1, FU_OUT => "PLC_BIT".AGG1_FU, EM_OUT =>, W_OVER =>, Q_OUT1 => "C#1_RB"."CAN AG1", Q_OUT2 =>, OVER =>, STA_RUN => "7.1.IND_AGG1".STA_RUN)
   END_RUNG
   RUNG wire#powerrail
      { S7_Templates := "SrcType := Real" } NE_Contact(in1 := "C#4_WD_WEIGHT".SV_AG1, in2 := 0.0)
      Contact( "PLC_BIT".RUN )
      Contact( "PLC_BIT".AUT )
      Contact( "9.1.DLC_IND_AGG1".OUT )
      I_Contact( "PLC_BIT".AGG1_FU )
      { S7_Templates := "SrcType := Real" } EQ_Contact(in1 := "C#7_RD_RUN".SMC_AG1, in2 := "C#7_RD_RUN".SMX_AG1)
      { S7_Templates := "SrcType := Real" } LT_Contact(in1 := "C#7_RD_RUN".SMC_AG1, in2 := "C#7_RD_RUN".SMT)
   END_RUNG wire#w2
   RUNG wire#powerrail
      Contact( "C#2_WB"."NN_CAN AG1" )
   END_RUNG wire#w3
   RUNG wire#powerrail
      Contact( "XA_HET_AGG" )
   END_RUNG wire#w3
   RUNG wire#powerrail
      Contact( "C#2_WB".F2_SW_PAU )
   END_RUNG wire#w4
   RUNG wire#powerrail
      Contact( "C#2_WB".SW_PA_AG1 )
   END_RUNG wire#w4
   RUNG wire#powerrail
      { S7_Templates := "SrcType := Real" } EQ_Contact(in1 := "C#6_WD_CALIB".XUNG_IND_AGG1, in2 := 32767.0)
   END_RUNG wire#w4
   RUNG wire#powerrail
      Contact( "7.1.IND_AGG1".STA_RUN )
      Coil( "C#1_RB".TTC_AG1 )
   END_RUNG
   // the same network as SCL:
   "9.1.DLC_IND_AGG1"(ON := "PLC_BIT".RUN AND NOT "PLC_BIT".AGG1_FU AND NOT "C#1_RB"."XA W_IND_AGG1",   // "9.TIMER_DELAY"
                      CLOCK_1S := "Clock_10Hz",
                      T_DELAY := "C#4_WD_WEIGHT"."W_IND_AGG1_TG.DLC",
                      OUT => "9.1.DLC_IND_AGG1".OUT,
                      T_OUT => "9.1.DLC_IND_AGG1".T_OUT);
   "7.1.IND_AGG1"(AUT := ("C#4_WD_WEIGHT".SV_AG1 <> 0.0) AND "PLC_BIT".RUN AND "PLC_BIT".AUT AND "9.1.DLC_IND_AGG1".OUT AND NOT "PLC_BIT".AGG1_FU AND ("C#7_RD_RUN".SMC_AG1 = "C#7_RD_RUN".SMX_AG1) AND ("C#7_RD_RUN".SMC_AG1 < "C#7_RD_RUN".SMT),   // "7.WEIGHT_PROCESS"
                  MAN1 := "C#2_WB"."NN_CAN AG1" OR "XA_HET_AGG",
                  FAU := "C#2_WB".F2_SW_PAU OR "C#2_WB".SW_PA_AG1 OR ("C#6_WD_CALIB".XUNG_IND_AGG1 = 32767.0),
                  FU_IN := "C#2_WB".NN_FU_AG1,
                  X_CLOCK := "Clock_10Hz",
                  EMTY_IN := "PLC_BIT".WAG1_EM,
                  XNC_AUT := TRUE,
                  SV_IN := "C#4_WD_WEIGHT".SV_AG1,
                  W_IN := "6.1.W_IND_AGG1".W_OUT1,
                  W_RTD := "C#3_WD_SILO".AG1_KL_RTD,
                  W_TR := "C#3_WD_SILO".AG1_SS_TREN,
                  W_DU := "C#3_WD_SILO".AG1_SS_DUOI,
                  T_ON := "C#3_WD_SILO".AG1_TG_ON_CAN,
                  T_OFF := "C#3_WD_SILO".AG1_TG_OFF_CAN,
                  T_DL := "C#3_WD_SILO".AG1_TG_ODC,
                  PV_OUT => "C#7_RD_RUN".PV_AG1,
                  PVM_OUT => "C#7_RD_RUN".PVM_AG1,
                  FU_OUT => "PLC_BIT".AGG1_FU,
                  Q_OUT1 => "C#1_RB"."CAN AG1",
                  STA_RUN => "7.1.IND_AGG1".STA_RUN);
   "C#1_RB".TTC_AG1 := "7.1.IND_AGG1".STA_RUN;
END_REGION
END_FUNCTION

FUNCTION "FCCA_IND_AGG2" : Void   // FC8, LAD
{ S7_Optimized_Access := 'TRUE' }
VERSION : 0.1
// stored: AutoNumber true, CodeModifiedDate 2026-01-15T16:25:55.0920194Z, CompileDate 2026-01-15T16:25:55.1307959Z, CreationDate 2026-01-15T16:24:02.4619467Z, HandleErrorsWithinBlock false, InterfaceModifiedDate 2026-01-11T04:46:28.8679318Z, IsConsistent true, IsIECCheckEnabled false, IsKnowHowProtected false, IsWriteProtected false, LibraryConformanceStatus Error: The block contains calls of single instances. Warning: The object contains access to global data blocks. Warning: The block contains direct access to inputs, outputs, bit memories, indirect access to the registry or indirect access to external memory areas that are unknown at the time of compilation., ModifiedDate 2026-01-15T16:25:55.0920194Z, ParameterModified 2026-01-11T04:46:28.8679318Z, PLCSimAdvancedSupport false, SetENOAutomatically False, StructureModified 2026-01-11T04:46:28.8679318Z, UDAEnableTagReadback false
BEGIN

REGION Network 1: Trạng thái cân AGG2
   // Đầu tiên nó sẽ đợi một khoảng thời gian gọi là Thời gian trễ cân, sau đó nó mới đủ điều kiện để cân
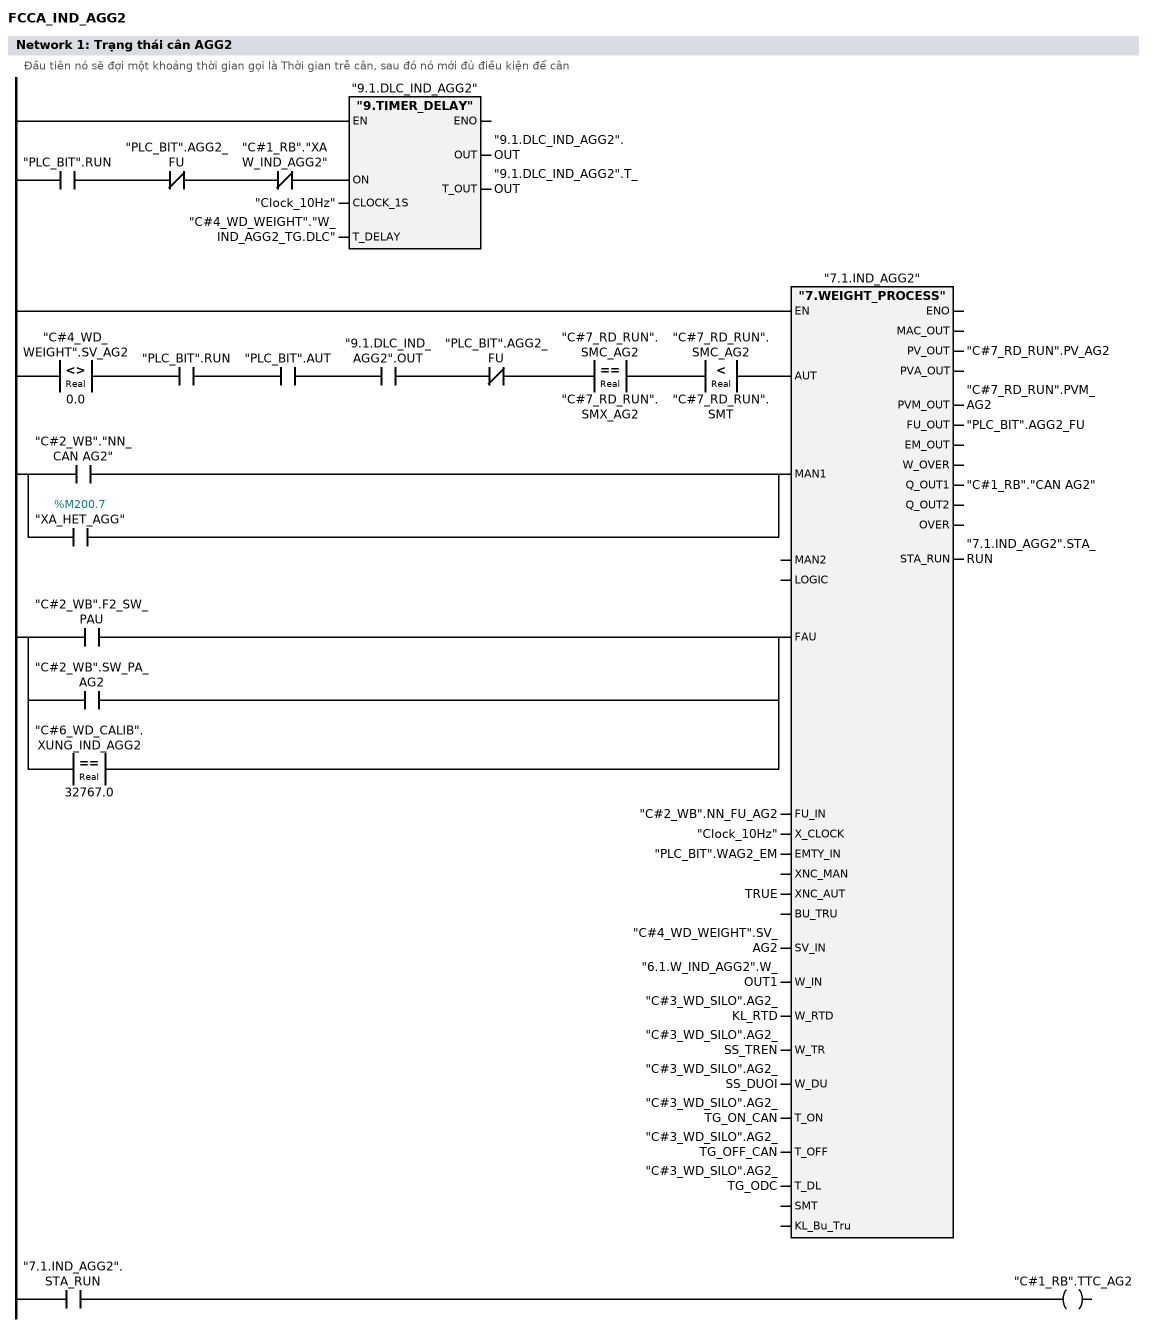
   RUNG wire#powerrail
      "9.1.DLC_IND_AGG2"(ON := wire#w1, CLOCK_1S := "Clock_10Hz", T_DELAY := "C#4_WD_WEIGHT"."W_IND_AGG2_TG.DLC", OUT => "9.1.DLC_IND_AGG2".OUT, T_OUT => "9.1.DLC_IND_AGG2".T_OUT)
   END_RUNG
   RUNG wire#powerrail
      Contact( "PLC_BIT".RUN )
      I_Contact( "PLC_BIT".AGG2_FU )
      I_Contact( "C#1_RB"."XA W_IND_AGG2" )
   END_RUNG wire#w1
   RUNG wire#powerrail
      "7.1.IND_AGG2"(AUT := wire#w2, MAN1 := wire#w3, FAU := wire#w4, MAN2 :=, LOGIC :=, FU_IN := "C#2_WB".NN_FU_AG2, X_CLOCK := "Clock_10Hz", EMTY_IN := "PLC_BIT".WAG2_EM, XNC_MAN :=, XNC_AUT := TRUE, BU_TRU :=, SV_IN := "C#4_WD_WEIGHT".SV_AG2, W_IN := "6.1.W_IND_AGG2".W_OUT1, W_RTD := "C#3_WD_SILO".AG2_KL_RTD, W_TR := "C#3_WD_SILO".AG2_SS_TREN, W_DU := "C#3_WD_SILO".AG2_SS_DUOI, T_ON := "C#3_WD_SILO".AG2_TG_ON_CAN, T_OFF := "C#3_WD_SILO".AG2_TG_OFF_CAN, T_DL := "C#3_WD_SILO".AG2_TG_ODC, SMT :=, KL_Bu_Tru :=, MAC_OUT =>, PV_OUT => "C#7_RD_RUN".PV_AG2, PVA_OUT =>, PVM_OUT => "C#7_RD_RUN".PVM_AG2, FU_OUT => "PLC_BIT".AGG2_FU, EM_OUT =>, W_OVER =>, Q_OUT1 => "C#1_RB"."CAN AG2", Q_OUT2 =>, OVER =>, STA_RUN => "7.1.IND_AGG2".STA_RUN)
   END_RUNG
   RUNG wire#powerrail
      { S7_Templates := "SrcType := Real" } NE_Contact(in1 := "C#4_WD_WEIGHT".SV_AG2, in2 := 0.0)
      Contact( "PLC_BIT".RUN )
      Contact( "PLC_BIT".AUT )
      Contact( "9.1.DLC_IND_AGG2".OUT )
      I_Contact( "PLC_BIT".AGG2_FU )
      { S7_Templates := "SrcType := Real" } EQ_Contact(in1 := "C#7_RD_RUN".SMC_AG2, in2 := "C#7_RD_RUN".SMX_AG2)
      { S7_Templates := "SrcType := Real" } LT_Contact(in1 := "C#7_RD_RUN".SMC_AG2, in2 := "C#7_RD_RUN".SMT)
   END_RUNG wire#w2
   RUNG wire#powerrail
      Contact( "C#2_WB"."NN_CAN AG2" )
   END_RUNG wire#w3
   RUNG wire#powerrail
      Contact( "XA_HET_AGG" )
   END_RUNG wire#w3
   RUNG wire#powerrail
      Contact( "C#2_WB".F2_SW_PAU )
   END_RUNG wire#w4
   RUNG wire#powerrail
      Contact( "C#2_WB".SW_PA_AG2 )
   END_RUNG wire#w4
   RUNG wire#powerrail
      { S7_Templates := "SrcType := Real" } EQ_Contact(in1 := "C#6_WD_CALIB".XUNG_IND_AGG2, in2 := 32767.0)
   END_RUNG wire#w4
   RUNG wire#powerrail
      Contact( "7.1.IND_AGG2".STA_RUN )
      Coil( "C#1_RB".TTC_AG2 )
   END_RUNG
   // the same network as SCL:
   "9.1.DLC_IND_AGG2"(ON := "PLC_BIT".RUN AND NOT "PLC_BIT".AGG2_FU AND NOT "C#1_RB"."XA W_IND_AGG2",   // "9.TIMER_DELAY"
                      CLOCK_1S := "Clock_10Hz",
                      T_DELAY := "C#4_WD_WEIGHT"."W_IND_AGG2_TG.DLC",
                      OUT => "9.1.DLC_IND_AGG2".OUT,
                      T_OUT => "9.1.DLC_IND_AGG2".T_OUT);
   "7.1.IND_AGG2"(AUT := ("C#4_WD_WEIGHT".SV_AG2 <> 0.0) AND "PLC_BIT".RUN AND "PLC_BIT".AUT AND "9.1.DLC_IND_AGG2".OUT AND NOT "PLC_BIT".AGG2_FU AND ("C#7_RD_RUN".SMC_AG2 = "C#7_RD_RUN".SMX_AG2) AND ("C#7_RD_RUN".SMC_AG2 < "C#7_RD_RUN".SMT),   // "7.WEIGHT_PROCESS"
                  MAN1 := "C#2_WB"."NN_CAN AG2" OR "XA_HET_AGG",
                  FAU := "C#2_WB".F2_SW_PAU OR "C#2_WB".SW_PA_AG2 OR ("C#6_WD_CALIB".XUNG_IND_AGG2 = 32767.0),
                  FU_IN := "C#2_WB".NN_FU_AG2,
                  X_CLOCK := "Clock_10Hz",
                  EMTY_IN := "PLC_BIT".WAG2_EM,
                  XNC_AUT := TRUE,
                  SV_IN := "C#4_WD_WEIGHT".SV_AG2,
                  W_IN := "6.1.W_IND_AGG2".W_OUT1,
                  W_RTD := "C#3_WD_SILO".AG2_KL_RTD,
                  W_TR := "C#3_WD_SILO".AG2_SS_TREN,
                  W_DU := "C#3_WD_SILO".AG2_SS_DUOI,
                  T_ON := "C#3_WD_SILO".AG2_TG_ON_CAN,
                  T_OFF := "C#3_WD_SILO".AG2_TG_OFF_CAN,
                  T_DL := "C#3_WD_SILO".AG2_TG_ODC,
                  PV_OUT => "C#7_RD_RUN".PV_AG2,
                  PVM_OUT => "C#7_RD_RUN".PVM_AG2,
                  FU_OUT => "PLC_BIT".AGG2_FU,
                  Q_OUT1 => "C#1_RB"."CAN AG2",
                  STA_RUN => "7.1.IND_AGG2".STA_RUN);
   "C#1_RB".TTC_AG2 := "7.1.IND_AGG2".STA_RUN;
END_REGION
END_FUNCTION

FUNCTION "FCCA_IND_AGG3" : Void   // FC11, LAD
{ S7_Optimized_Access := 'TRUE' }
VERSION : 0.1
// stored: AutoNumber true, CodeModifiedDate 2026-01-15T16:25:54.8129712Z, CompileDate 2026-01-15T16:25:54.8463711Z, CreationDate 2026-01-15T16:24:02.4619467Z, HandleErrorsWithinBlock false, InterfaceModifiedDate 2026-01-11T04:46:44.6799525Z, IsConsistent true, IsIECCheckEnabled false, IsKnowHowProtected false, IsWriteProtected false, LibraryConformanceStatus Error: The block contains calls of single instances. Warning: The object contains access to global data blocks. Warning: The block contains direct access to inputs, outputs, bit memories, indirect access to the registry or indirect access to external memory areas that are unknown at the time of compilation., ModifiedDate 2026-01-15T16:25:54.8129712Z, ParameterModified 2026-01-11T04:46:44.6799525Z, PLCSimAdvancedSupport false, SetENOAutomatically False, StructureModified 2026-01-11T04:46:44.6799525Z, UDAEnableTagReadback false
BEGIN

REGION Network 1: Trạng thái cân AGG3
   // Đầu tiên nó sẽ đợi một khoảng thời gian gọi là Thời gian trễ cân, sau đó nó mới đủ điều kiện để cân
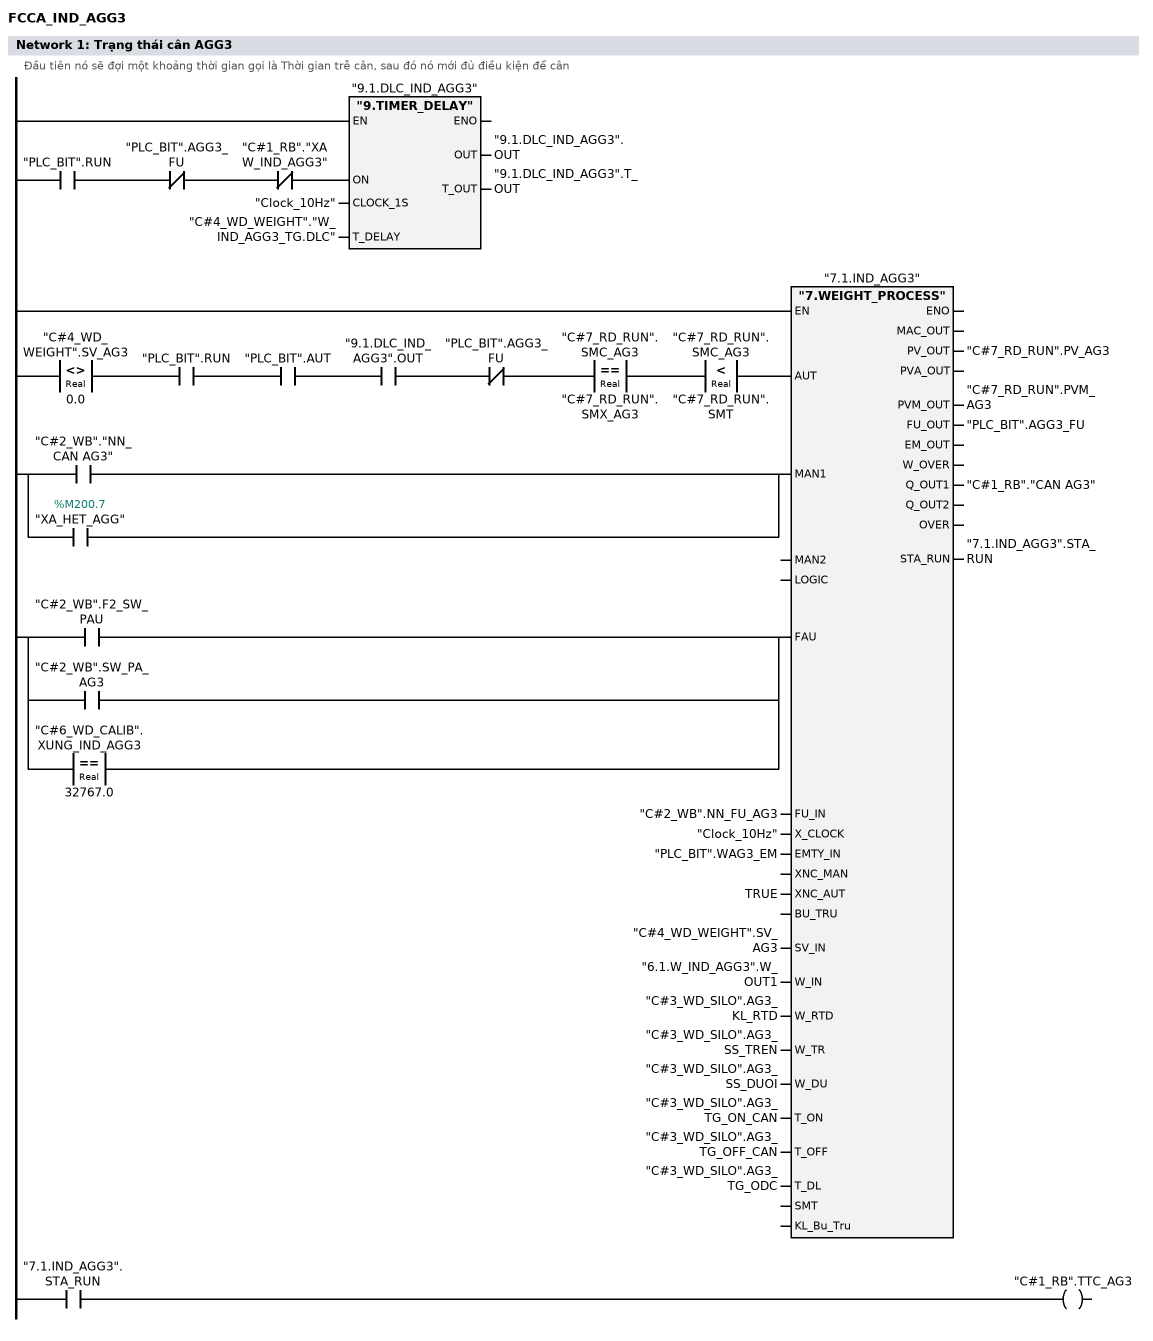
   RUNG wire#powerrail
      "9.1.DLC_IND_AGG3"(ON := wire#w1, CLOCK_1S := "Clock_10Hz", T_DELAY := "C#4_WD_WEIGHT"."W_IND_AGG3_TG.DLC", OUT => "9.1.DLC_IND_AGG3".OUT, T_OUT => "9.1.DLC_IND_AGG3".T_OUT)
   END_RUNG
   RUNG wire#powerrail
      Contact( "PLC_BIT".RUN )
      I_Contact( "PLC_BIT".AGG3_FU )
      I_Contact( "C#1_RB"."XA W_IND_AGG3" )
   END_RUNG wire#w1
   RUNG wire#powerrail
      "7.1.IND_AGG3"(AUT := wire#w2, MAN1 := wire#w3, FAU := wire#w4, MAN2 :=, LOGIC :=, FU_IN := "C#2_WB".NN_FU_AG3, X_CLOCK := "Clock_10Hz", EMTY_IN := "PLC_BIT".WAG3_EM, XNC_MAN :=, XNC_AUT := TRUE, BU_TRU :=, SV_IN := "C#4_WD_WEIGHT".SV_AG3, W_IN := "6.1.W_IND_AGG3".W_OUT1, W_RTD := "C#3_WD_SILO".AG3_KL_RTD, W_TR := "C#3_WD_SILO".AG3_SS_TREN, W_DU := "C#3_WD_SILO".AG3_SS_DUOI, T_ON := "C#3_WD_SILO".AG3_TG_ON_CAN, T_OFF := "C#3_WD_SILO".AG3_TG_OFF_CAN, T_DL := "C#3_WD_SILO".AG3_TG_ODC, SMT :=, KL_Bu_Tru :=, MAC_OUT =>, PV_OUT => "C#7_RD_RUN".PV_AG3, PVA_OUT =>, PVM_OUT => "C#7_RD_RUN".PVM_AG3, FU_OUT => "PLC_BIT".AGG3_FU, EM_OUT =>, W_OVER =>, Q_OUT1 => "C#1_RB"."CAN AG3", Q_OUT2 =>, OVER =>, STA_RUN => "7.1.IND_AGG3".STA_RUN)
   END_RUNG
   RUNG wire#powerrail
      { S7_Templates := "SrcType := Real" } NE_Contact(in1 := "C#4_WD_WEIGHT".SV_AG3, in2 := 0.0)
      Contact( "PLC_BIT".RUN )
      Contact( "PLC_BIT".AUT )
      Contact( "9.1.DLC_IND_AGG3".OUT )
      I_Contact( "PLC_BIT".AGG3_FU )
      { S7_Templates := "SrcType := Real" } EQ_Contact(in1 := "C#7_RD_RUN".SMC_AG3, in2 := "C#7_RD_RUN".SMX_AG3)
      { S7_Templates := "SrcType := Real" } LT_Contact(in1 := "C#7_RD_RUN".SMC_AG3, in2 := "C#7_RD_RUN".SMT)
   END_RUNG wire#w2
   RUNG wire#powerrail
      Contact( "C#2_WB"."NN_CAN AG3" )
   END_RUNG wire#w3
   RUNG wire#powerrail
      Contact( "XA_HET_AGG" )
   END_RUNG wire#w3
   RUNG wire#powerrail
      Contact( "C#2_WB".F2_SW_PAU )
   END_RUNG wire#w4
   RUNG wire#powerrail
      Contact( "C#2_WB".SW_PA_AG3 )
   END_RUNG wire#w4
   RUNG wire#powerrail
      { S7_Templates := "SrcType := Real" } EQ_Contact(in1 := "C#6_WD_CALIB".XUNG_IND_AGG3, in2 := 32767.0)
   END_RUNG wire#w4
   RUNG wire#powerrail
      Contact( "7.1.IND_AGG3".STA_RUN )
      Coil( "C#1_RB".TTC_AG3 )
   END_RUNG
   // the same network as SCL:
   "9.1.DLC_IND_AGG3"(ON := "PLC_BIT".RUN AND NOT "PLC_BIT".AGG3_FU AND NOT "C#1_RB"."XA W_IND_AGG3",   // "9.TIMER_DELAY"
                      CLOCK_1S := "Clock_10Hz",
                      T_DELAY := "C#4_WD_WEIGHT"."W_IND_AGG3_TG.DLC",
                      OUT => "9.1.DLC_IND_AGG3".OUT,
                      T_OUT => "9.1.DLC_IND_AGG3".T_OUT);
   "7.1.IND_AGG3"(AUT := ("C#4_WD_WEIGHT".SV_AG3 <> 0.0) AND "PLC_BIT".RUN AND "PLC_BIT".AUT AND "9.1.DLC_IND_AGG3".OUT AND NOT "PLC_BIT".AGG3_FU AND ("C#7_RD_RUN".SMC_AG3 = "C#7_RD_RUN".SMX_AG3) AND ("C#7_RD_RUN".SMC_AG3 < "C#7_RD_RUN".SMT),   // "7.WEIGHT_PROCESS"
                  MAN1 := "C#2_WB"."NN_CAN AG3" OR "XA_HET_AGG",
                  FAU := "C#2_WB".F2_SW_PAU OR "C#2_WB".SW_PA_AG3 OR ("C#6_WD_CALIB".XUNG_IND_AGG3 = 32767.0),
                  FU_IN := "C#2_WB".NN_FU_AG3,
                  X_CLOCK := "Clock_10Hz",
                  EMTY_IN := "PLC_BIT".WAG3_EM,
                  XNC_AUT := TRUE,
                  SV_IN := "C#4_WD_WEIGHT".SV_AG3,
                  W_IN := "6.1.W_IND_AGG3".W_OUT1,
                  W_RTD := "C#3_WD_SILO".AG3_KL_RTD,
                  W_TR := "C#3_WD_SILO".AG3_SS_TREN,
                  W_DU := "C#3_WD_SILO".AG3_SS_DUOI,
                  T_ON := "C#3_WD_SILO".AG3_TG_ON_CAN,
                  T_OFF := "C#3_WD_SILO".AG3_TG_OFF_CAN,
                  T_DL := "C#3_WD_SILO".AG3_TG_ODC,
                  PV_OUT => "C#7_RD_RUN".PV_AG3,
                  PVM_OUT => "C#7_RD_RUN".PVM_AG3,
                  FU_OUT => "PLC_BIT".AGG3_FU,
                  Q_OUT1 => "C#1_RB"."CAN AG3",
                  STA_RUN => "7.1.IND_AGG3".STA_RUN);
   "C#1_RB".TTC_AG3 := "7.1.IND_AGG3".STA_RUN;
END_REGION
END_FUNCTION

FUNCTION "FCCA_IND_AGG4" : Void   // FC13, LAD
{ S7_Optimized_Access := 'TRUE' }
VERSION : 0.1
// stored: AutoNumber true, CodeModifiedDate 2026-01-15T16:25:54.6221046Z, CompileDate 2026-01-15T16:25:54.6613801Z, CreationDate 2026-01-15T16:24:02.4619467Z, HandleErrorsWithinBlock false, InterfaceModifiedDate 2026-01-11T04:46:59.531034Z, IsConsistent true, IsIECCheckEnabled false, IsKnowHowProtected false, IsWriteProtected false, LibraryConformanceStatus Error: The block contains calls of single instances. Warning: The object contains access to global data blocks. Warning: The block contains direct access to inputs, outputs, bit memories, indirect access to the registry or indirect access to external memory areas that are unknown at the time of compilation., ModifiedDate 2026-01-15T16:25:54.6221046Z, ParameterModified 2026-01-11T04:46:59.531034Z, PLCSimAdvancedSupport false, SetENOAutomatically False, StructureModified 2026-01-11T04:46:59.531034Z, UDAEnableTagReadback false
BEGIN

REGION Network 1: Trạng thái cân AGG4
   // Đầu tiên nó sẽ đợi một khoảng thời gian gọi là Thời gian trễ cân, sau đó nó mới đủ điều kiện để cân
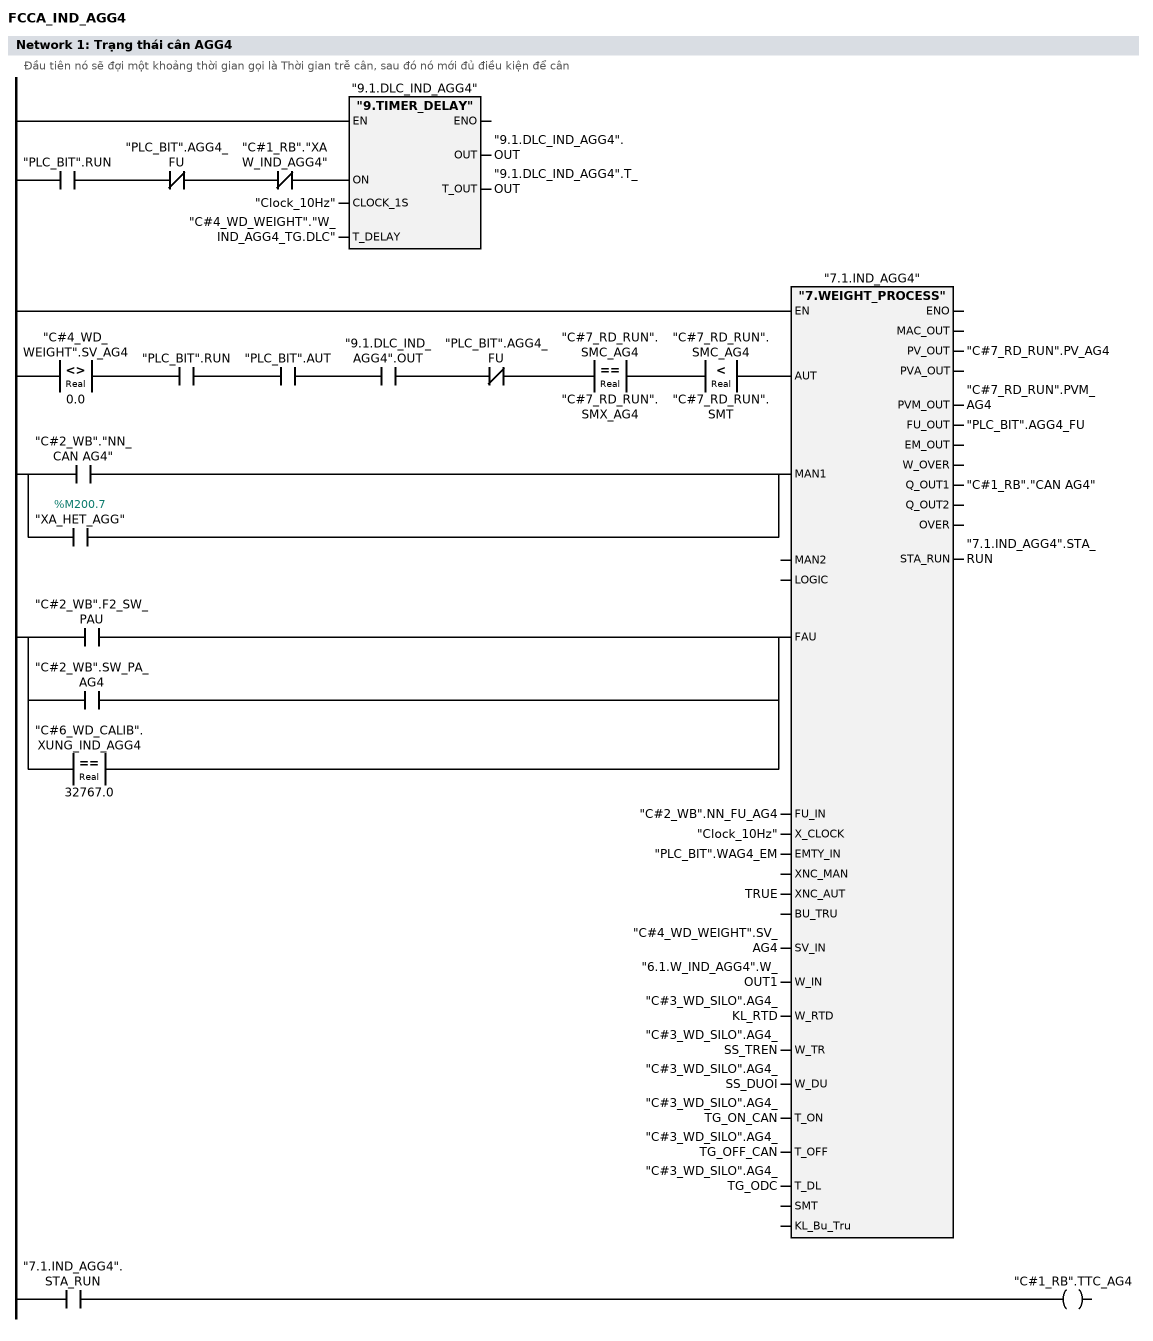
   RUNG wire#powerrail
      "9.1.DLC_IND_AGG4"(ON := wire#w1, CLOCK_1S := "Clock_10Hz", T_DELAY := "C#4_WD_WEIGHT"."W_IND_AGG4_TG.DLC", OUT => "9.1.DLC_IND_AGG4".OUT, T_OUT => "9.1.DLC_IND_AGG4".T_OUT)
   END_RUNG
   RUNG wire#powerrail
      Contact( "PLC_BIT".RUN )
      I_Contact( "PLC_BIT".AGG4_FU )
      I_Contact( "C#1_RB"."XA W_IND_AGG4" )
   END_RUNG wire#w1
   RUNG wire#powerrail
      "7.1.IND_AGG4"(AUT := wire#w2, MAN1 := wire#w3, FAU := wire#w4, MAN2 :=, LOGIC :=, FU_IN := "C#2_WB".NN_FU_AG4, X_CLOCK := "Clock_10Hz", EMTY_IN := "PLC_BIT".WAG4_EM, XNC_MAN :=, XNC_AUT := TRUE, BU_TRU :=, SV_IN := "C#4_WD_WEIGHT".SV_AG4, W_IN := "6.1.W_IND_AGG4".W_OUT1, W_RTD := "C#3_WD_SILO".AG4_KL_RTD, W_TR := "C#3_WD_SILO".AG4_SS_TREN, W_DU := "C#3_WD_SILO".AG4_SS_DUOI, T_ON := "C#3_WD_SILO".AG4_TG_ON_CAN, T_OFF := "C#3_WD_SILO".AG4_TG_OFF_CAN, T_DL := "C#3_WD_SILO".AG4_TG_ODC, SMT :=, KL_Bu_Tru :=, MAC_OUT =>, PV_OUT => "C#7_RD_RUN".PV_AG4, PVA_OUT =>, PVM_OUT => "C#7_RD_RUN".PVM_AG4, FU_OUT => "PLC_BIT".AGG4_FU, EM_OUT =>, W_OVER =>, Q_OUT1 => "C#1_RB"."CAN AG4", Q_OUT2 =>, OVER =>, STA_RUN => "7.1.IND_AGG4".STA_RUN)
   END_RUNG
   RUNG wire#powerrail
      { S7_Templates := "SrcType := Real" } NE_Contact(in1 := "C#4_WD_WEIGHT".SV_AG4, in2 := 0.0)
      Contact( "PLC_BIT".RUN )
      Contact( "PLC_BIT".AUT )
      Contact( "9.1.DLC_IND_AGG4".OUT )
      I_Contact( "PLC_BIT".AGG4_FU )
      { S7_Templates := "SrcType := Real" } EQ_Contact(in1 := "C#7_RD_RUN".SMC_AG4, in2 := "C#7_RD_RUN".SMX_AG4)
      { S7_Templates := "SrcType := Real" } LT_Contact(in1 := "C#7_RD_RUN".SMC_AG4, in2 := "C#7_RD_RUN".SMT)
   END_RUNG wire#w2
   RUNG wire#powerrail
      Contact( "C#2_WB"."NN_CAN AG4" )
   END_RUNG wire#w3
   RUNG wire#powerrail
      Contact( "XA_HET_AGG" )
   END_RUNG wire#w3
   RUNG wire#powerrail
      Contact( "C#2_WB".F2_SW_PAU )
   END_RUNG wire#w4
   RUNG wire#powerrail
      Contact( "C#2_WB".SW_PA_AG4 )
   END_RUNG wire#w4
   RUNG wire#powerrail
      { S7_Templates := "SrcType := Real" } EQ_Contact(in1 := "C#6_WD_CALIB".XUNG_IND_AGG4, in2 := 32767.0)
   END_RUNG wire#w4
   RUNG wire#powerrail
      Contact( "7.1.IND_AGG4".STA_RUN )
      Coil( "C#1_RB".TTC_AG4 )
   END_RUNG
   // the same network as SCL:
   "9.1.DLC_IND_AGG4"(ON := "PLC_BIT".RUN AND NOT "PLC_BIT".AGG4_FU AND NOT "C#1_RB"."XA W_IND_AGG4",   // "9.TIMER_DELAY"
                      CLOCK_1S := "Clock_10Hz",
                      T_DELAY := "C#4_WD_WEIGHT"."W_IND_AGG4_TG.DLC",
                      OUT => "9.1.DLC_IND_AGG4".OUT,
                      T_OUT => "9.1.DLC_IND_AGG4".T_OUT);
   "7.1.IND_AGG4"(AUT := ("C#4_WD_WEIGHT".SV_AG4 <> 0.0) AND "PLC_BIT".RUN AND "PLC_BIT".AUT AND "9.1.DLC_IND_AGG4".OUT AND NOT "PLC_BIT".AGG4_FU AND ("C#7_RD_RUN".SMC_AG4 = "C#7_RD_RUN".SMX_AG4) AND ("C#7_RD_RUN".SMC_AG4 < "C#7_RD_RUN".SMT),   // "7.WEIGHT_PROCESS"
                  MAN1 := "C#2_WB"."NN_CAN AG4" OR "XA_HET_AGG",
                  FAU := "C#2_WB".F2_SW_PAU OR "C#2_WB".SW_PA_AG4 OR ("C#6_WD_CALIB".XUNG_IND_AGG4 = 32767.0),
                  FU_IN := "C#2_WB".NN_FU_AG4,
                  X_CLOCK := "Clock_10Hz",
                  EMTY_IN := "PLC_BIT".WAG4_EM,
                  XNC_AUT := TRUE,
                  SV_IN := "C#4_WD_WEIGHT".SV_AG4,
                  W_IN := "6.1.W_IND_AGG4".W_OUT1,
                  W_RTD := "C#3_WD_SILO".AG4_KL_RTD,
                  W_TR := "C#3_WD_SILO".AG4_SS_TREN,
                  W_DU := "C#3_WD_SILO".AG4_SS_DUOI,
                  T_ON := "C#3_WD_SILO".AG4_TG_ON_CAN,
                  T_OFF := "C#3_WD_SILO".AG4_TG_OFF_CAN,
                  T_DL := "C#3_WD_SILO".AG4_TG_ODC,
                  PV_OUT => "C#7_RD_RUN".PV_AG4,
                  PVM_OUT => "C#7_RD_RUN".PVM_AG4,
                  FU_OUT => "PLC_BIT".AGG4_FU,
                  Q_OUT1 => "C#1_RB"."CAN AG4",
                  STA_RUN => "7.1.IND_AGG4".STA_RUN);
   "C#1_RB".TTC_AG4 := "7.1.IND_AGG4".STA_RUN;
END_REGION
END_FUNCTION

FUNCTION "FCCA_IND_AGG5" : Void   // FC14, LAD
{ S7_Optimized_Access := 'TRUE' }
VERSION : 0.1
// stored: AutoNumber true, CodeModifiedDate 2026-01-15T16:25:54.5394757Z, CompileDate 2026-01-15T16:25:54.5786206Z, CreationDate 2026-01-15T16:24:02.4619467Z, HandleErrorsWithinBlock false, InterfaceModifiedDate 2026-01-11T04:47:10.3302964Z, IsConsistent true, IsIECCheckEnabled false, IsKnowHowProtected false, IsWriteProtected false, LibraryConformanceStatus Error: The block contains calls of single instances. Warning: The object contains access to global data blocks. Warning: The block contains direct access to inputs, outputs, bit memories, indirect access to the registry or indirect access to external memory areas that are unknown at the time of compilation., ModifiedDate 2026-01-15T16:25:54.5394757Z, ParameterModified 2026-01-11T04:47:10.3302964Z, PLCSimAdvancedSupport false, SetENOAutomatically False, StructureModified 2026-01-11T04:47:10.3302964Z, UDAEnableTagReadback false
BEGIN

REGION Network 1: Trạng thái cân AGG5
   // Đầu tiên nó sẽ đợi một khoảng thời gian gọi là Thời gian trễ cân, sau đó nó mới đủ điều kiện để cân
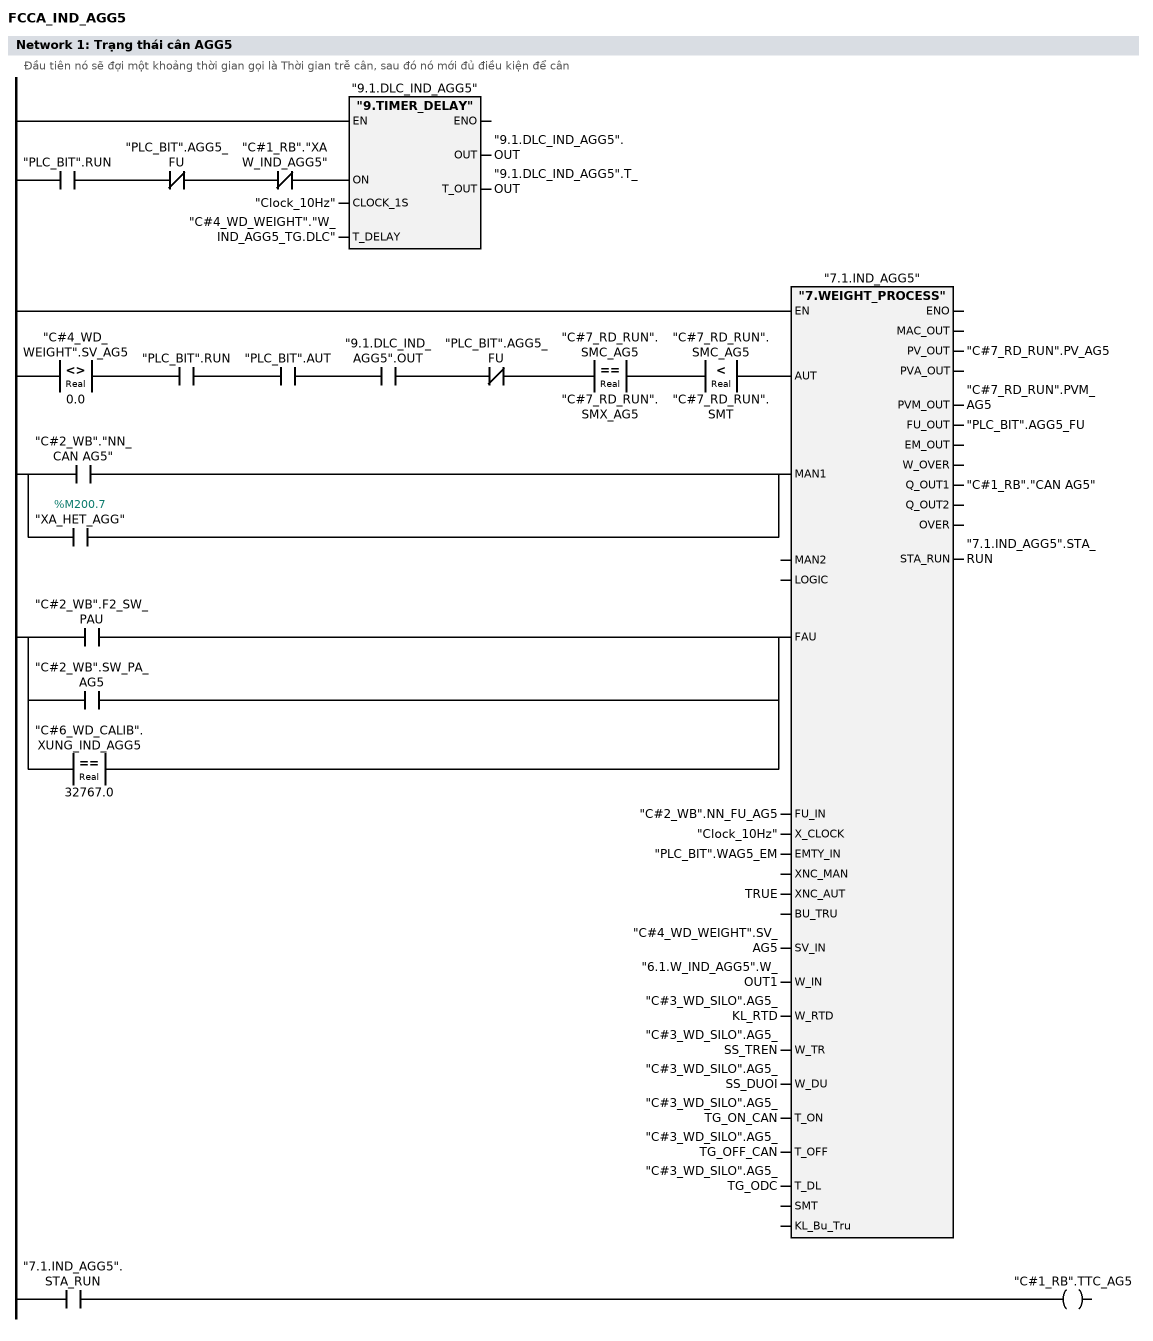
   RUNG wire#powerrail
      "9.1.DLC_IND_AGG5"(ON := wire#w1, CLOCK_1S := "Clock_10Hz", T_DELAY := "C#4_WD_WEIGHT"."W_IND_AGG5_TG.DLC", OUT => "9.1.DLC_IND_AGG5".OUT, T_OUT => "9.1.DLC_IND_AGG5".T_OUT)
   END_RUNG
   RUNG wire#powerrail
      Contact( "PLC_BIT".RUN )
      I_Contact( "PLC_BIT".AGG5_FU )
      I_Contact( "C#1_RB"."XA W_IND_AGG5" )
   END_RUNG wire#w1
   RUNG wire#powerrail
      "7.1.IND_AGG5"(AUT := wire#w2, MAN1 := wire#w3, FAU := wire#w4, MAN2 :=, LOGIC :=, FU_IN := "C#2_WB".NN_FU_AG5, X_CLOCK := "Clock_10Hz", EMTY_IN := "PLC_BIT".WAG5_EM, XNC_MAN :=, XNC_AUT := TRUE, BU_TRU :=, SV_IN := "C#4_WD_WEIGHT".SV_AG5, W_IN := "6.1.W_IND_AGG5".W_OUT1, W_RTD := "C#3_WD_SILO".AG5_KL_RTD, W_TR := "C#3_WD_SILO".AG5_SS_TREN, W_DU := "C#3_WD_SILO".AG5_SS_DUOI, T_ON := "C#3_WD_SILO".AG5_TG_ON_CAN, T_OFF := "C#3_WD_SILO".AG5_TG_OFF_CAN, T_DL := "C#3_WD_SILO".AG5_TG_ODC, SMT :=, KL_Bu_Tru :=, MAC_OUT =>, PV_OUT => "C#7_RD_RUN".PV_AG5, PVA_OUT =>, PVM_OUT => "C#7_RD_RUN".PVM_AG5, FU_OUT => "PLC_BIT".AGG5_FU, EM_OUT =>, W_OVER =>, Q_OUT1 => "C#1_RB"."CAN AG5", Q_OUT2 =>, OVER =>, STA_RUN => "7.1.IND_AGG5".STA_RUN)
   END_RUNG
   RUNG wire#powerrail
      { S7_Templates := "SrcType := Real" } NE_Contact(in1 := "C#4_WD_WEIGHT".SV_AG5, in2 := 0.0)
      Contact( "PLC_BIT".RUN )
      Contact( "PLC_BIT".AUT )
      Contact( "9.1.DLC_IND_AGG5".OUT )
      I_Contact( "PLC_BIT".AGG5_FU )
      { S7_Templates := "SrcType := Real" } EQ_Contact(in1 := "C#7_RD_RUN".SMC_AG5, in2 := "C#7_RD_RUN".SMX_AG5)
      { S7_Templates := "SrcType := Real" } LT_Contact(in1 := "C#7_RD_RUN".SMC_AG5, in2 := "C#7_RD_RUN".SMT)
   END_RUNG wire#w2
   RUNG wire#powerrail
      Contact( "C#2_WB"."NN_CAN AG5" )
   END_RUNG wire#w3
   RUNG wire#powerrail
      Contact( "XA_HET_AGG" )
   END_RUNG wire#w3
   RUNG wire#powerrail
      Contact( "C#2_WB".F2_SW_PAU )
   END_RUNG wire#w4
   RUNG wire#powerrail
      Contact( "C#2_WB".SW_PA_AG5 )
   END_RUNG wire#w4
   RUNG wire#powerrail
      { S7_Templates := "SrcType := Real" } EQ_Contact(in1 := "C#6_WD_CALIB".XUNG_IND_AGG5, in2 := 32767.0)
   END_RUNG wire#w4
   RUNG wire#powerrail
      Contact( "7.1.IND_AGG5".STA_RUN )
      Coil( "C#1_RB".TTC_AG5 )
   END_RUNG
   // the same network as SCL:
   "9.1.DLC_IND_AGG5"(ON := "PLC_BIT".RUN AND NOT "PLC_BIT".AGG5_FU AND NOT "C#1_RB"."XA W_IND_AGG5",   // "9.TIMER_DELAY"
                      CLOCK_1S := "Clock_10Hz",
                      T_DELAY := "C#4_WD_WEIGHT"."W_IND_AGG5_TG.DLC",
                      OUT => "9.1.DLC_IND_AGG5".OUT,
                      T_OUT => "9.1.DLC_IND_AGG5".T_OUT);
   "7.1.IND_AGG5"(AUT := ("C#4_WD_WEIGHT".SV_AG5 <> 0.0) AND "PLC_BIT".RUN AND "PLC_BIT".AUT AND "9.1.DLC_IND_AGG5".OUT AND NOT "PLC_BIT".AGG5_FU AND ("C#7_RD_RUN".SMC_AG5 = "C#7_RD_RUN".SMX_AG5) AND ("C#7_RD_RUN".SMC_AG5 < "C#7_RD_RUN".SMT),   // "7.WEIGHT_PROCESS"
                  MAN1 := "C#2_WB"."NN_CAN AG5" OR "XA_HET_AGG",
                  FAU := "C#2_WB".F2_SW_PAU OR "C#2_WB".SW_PA_AG5 OR ("C#6_WD_CALIB".XUNG_IND_AGG5 = 32767.0),
                  FU_IN := "C#2_WB".NN_FU_AG5,
                  X_CLOCK := "Clock_10Hz",
                  EMTY_IN := "PLC_BIT".WAG5_EM,
                  XNC_AUT := TRUE,
                  SV_IN := "C#4_WD_WEIGHT".SV_AG5,
                  W_IN := "6.1.W_IND_AGG5".W_OUT1,
                  W_RTD := "C#3_WD_SILO".AG5_KL_RTD,
                  W_TR := "C#3_WD_SILO".AG5_SS_TREN,
                  W_DU := "C#3_WD_SILO".AG5_SS_DUOI,
                  T_ON := "C#3_WD_SILO".AG5_TG_ON_CAN,
                  T_OFF := "C#3_WD_SILO".AG5_TG_OFF_CAN,
                  T_DL := "C#3_WD_SILO".AG5_TG_ODC,
                  PV_OUT => "C#7_RD_RUN".PV_AG5,
                  PVM_OUT => "C#7_RD_RUN".PVM_AG5,
                  FU_OUT => "PLC_BIT".AGG5_FU,
                  Q_OUT1 => "C#1_RB"."CAN AG5",
                  STA_RUN => "7.1.IND_AGG5".STA_RUN);
   "C#1_RB".TTC_AG5 := "7.1.IND_AGG5".STA_RUN;
END_REGION
END_FUNCTION

FUNCTION "FCXL_IND_AGG1" : Void   // FC6, LAD
{ S7_Optimized_Access := 'TRUE' }
VERSION : 0.1
// stored: AutoNumber true, CodeModifiedDate 2026-01-15T16:25:53.86748Z, CompileDate 2026-01-15T16:25:53.9093246Z, CreationDate 2026-01-15T16:24:02.4619467Z, HandleErrorsWithinBlock false, InterfaceModifiedDate 2026-01-10T11:03:05.6285532Z, IsConsistent true, IsIECCheckEnabled false, IsKnowHowProtected false, IsWriteProtected false, LibraryConformanceStatus Error: The block contains calls of single instances. Warning: The object contains access to global data blocks. Warning: The block contains direct access to inputs, outputs, bit memories, indirect access to the registry or indirect access to external memory areas that are unknown at the time of compilation., ModifiedDate 2026-01-15T16:25:53.86748Z, ParameterModified 2026-01-10T11:03:05.6285532Z, PLCSimAdvancedSupport false, SetENOAutomatically False, StructureModified 2026-01-10T11:03:05.6285532Z, UDAEnableTagReadback false
   VAR_TEMP   // added for the SCL form of the ladder/FBD networks
      _w1 : Bool;
      _w2 : Bool;
      _w3 : Bool;
   END_VAR
BEGIN

REGION Network 1: Cân độc lập AGG1 Full
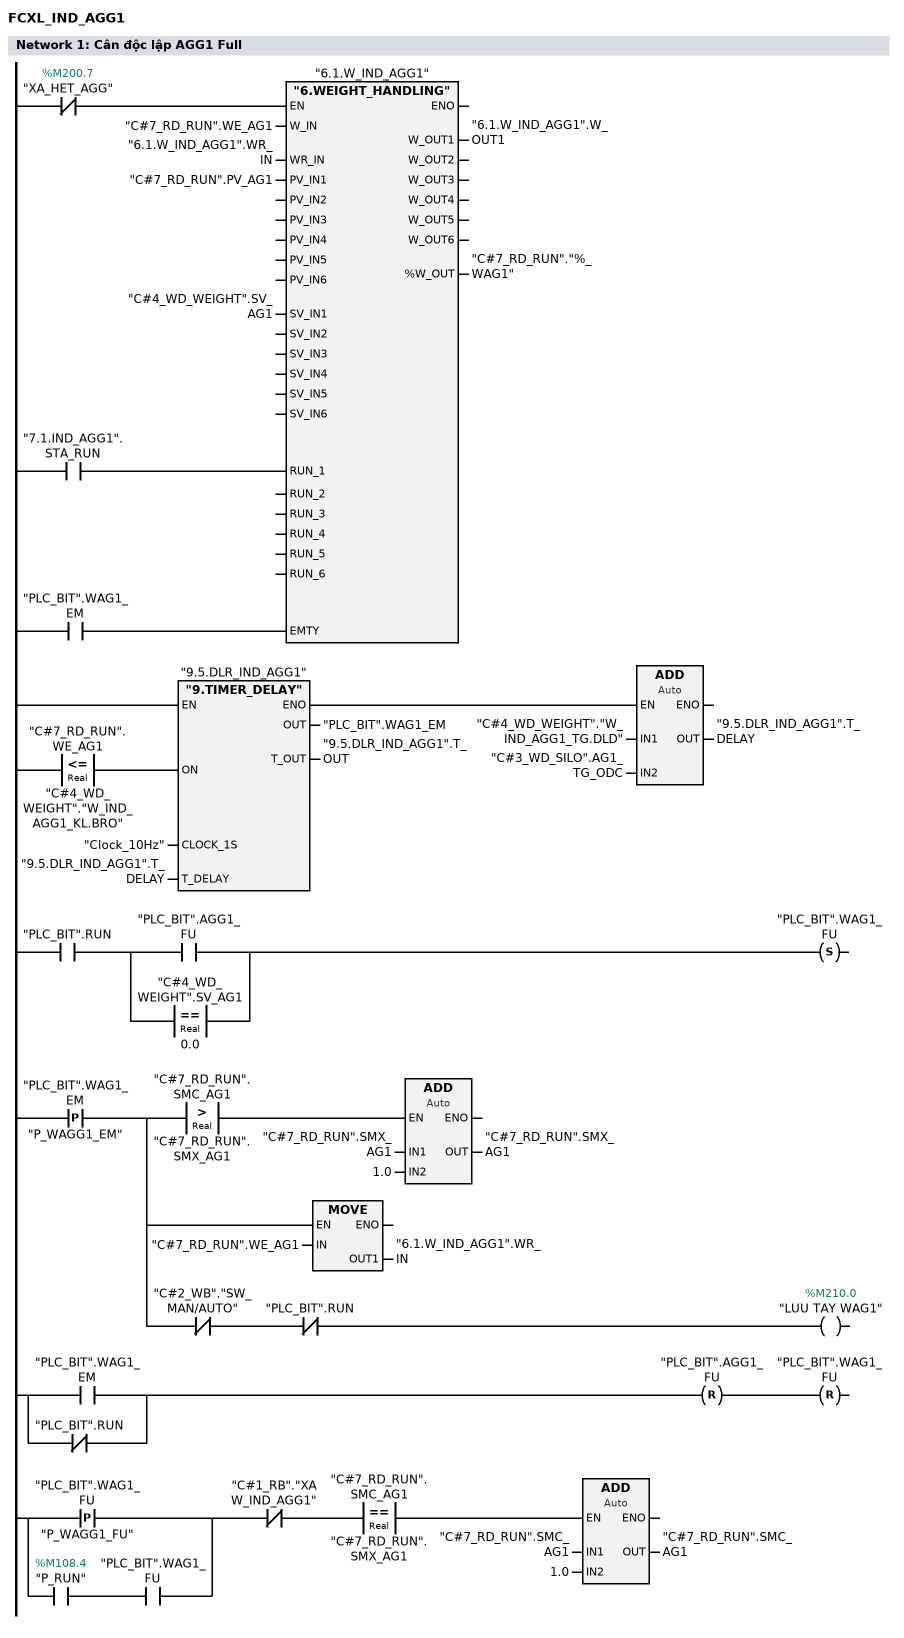
   RUNG wire#powerrail
      I_Contact( "XA_HET_AGG" )
      "6.1.W_IND_AGG1"(RUN_1 := wire#w1, EMTY := wire#w2, W_IN := "C#7_RD_RUN".WE_AG1, WR_IN := "6.1.W_IND_AGG1".WR_IN, PV_IN1 := "C#7_RD_RUN".PV_AG1, PV_IN2 :=, PV_IN3 :=, PV_IN4 :=, PV_IN5 :=, PV_IN6 :=, SV_IN1 := "C#4_WD_WEIGHT".SV_AG1, SV_IN2 :=, SV_IN3 :=, SV_IN4 :=, SV_IN5 :=, SV_IN6 :=, RUN_2 :=, RUN_3 :=, RUN_4 :=, RUN_5 :=, RUN_6 :=, W_OUT1 => "6.1.W_IND_AGG1".W_OUT1, W_OUT2 =>, W_OUT3 =>, W_OUT4 =>, W_OUT5 =>, W_OUT6 =>, "%W_OUT" => "C#7_RD_RUN"."%_WAG1")
   END_RUNG
   RUNG wire#powerrail
      Contact( "7.1.IND_AGG1".STA_RUN )
   END_RUNG wire#w1
   RUNG wire#powerrail
      Contact( "PLC_BIT".WAG1_EM )
   END_RUNG wire#w2
   RUNG wire#powerrail
      "9.5.DLR_IND_AGG1"(ON := wire#w3, CLOCK_1S := "Clock_10Hz", T_DELAY := "9.5.DLR_IND_AGG1".T_DELAY, OUT => "PLC_BIT".WAG1_EM, T_OUT => "9.5.DLR_IND_AGG1".T_OUT)
      Add(in1 := "C#4_WD_WEIGHT"."W_IND_AGG1_TG.DLD", in2 := "C#3_WD_SILO".AG1_TG_ODC, out => "9.5.DLR_IND_AGG1".T_DELAY)
   END_RUNG
   RUNG wire#powerrail
      { S7_Templates := "SrcType := Real" } LE_Contact(in1 := "C#7_RD_RUN".WE_AG1, in2 := "C#4_WD_WEIGHT"."W_IND_AGG1_KL.BRO")
   END_RUNG wire#w3
   RUNG wire#powerrail
      Contact( "PLC_BIT".RUN )
      wire#w4
      Contact( "PLC_BIT".AGG1_FU )
      wire#w5
      S_Coil( "PLC_BIT".WAG1_FU )
   END_RUNG
   RUNG wire#w4
      { S7_Templates := "SrcType := Real" } EQ_Contact(in1 := "C#4_WD_WEIGHT".SV_AG1, in2 := 0.0)
   END_RUNG wire#w5
   RUNG wire#powerrail
      P_Contact(operand := "PLC_BIT".WAG1_EM, bit := "P_WAGG1_EM")
      wire#w6
      { S7_Templates := "SrcType := Real" } GT_Contact(in1 := "C#7_RD_RUN".SMC_AG1, in2 := "C#7_RD_RUN".SMX_AG1)
      Add(in1 := "C#7_RD_RUN".SMX_AG1, in2 := 1.0, out => "C#7_RD_RUN".SMX_AG1)
   END_RUNG
   RUNG wire#w6
      Move(in := "C#7_RD_RUN".WE_AG1, out1 => "6.1.W_IND_AGG1".WR_IN)
   END_RUNG
   RUNG wire#w6
      I_Contact( "C#2_WB"."SW_MAN/AUTO" )
      I_Contact( "PLC_BIT".RUN )
      Coil( "LUU TAY WAG1" )
   END_RUNG
   RUNG wire#powerrail
      Contact( "PLC_BIT".WAG1_EM )
      wire#w7
      R_Coil( "PLC_BIT".AGG1_FU )
      R_Coil( "PLC_BIT".WAG1_FU )
   END_RUNG
   RUNG wire#powerrail
      I_Contact( "PLC_BIT".RUN )
   END_RUNG wire#w7
   RUNG wire#powerrail
      P_Contact(operand := "PLC_BIT".WAG1_FU, bit := "P_WAGG1_FU")
      wire#w8
      I_Contact( "C#1_RB"."XA W_IND_AGG1" )
      { S7_Templates := "SrcType := Real" } EQ_Contact(in1 := "C#7_RD_RUN".SMC_AG1, in2 := "C#7_RD_RUN".SMX_AG1)
      Add(in1 := "C#7_RD_RUN".SMC_AG1, in2 := 1.0, out => "C#7_RD_RUN".SMC_AG1)
   END_RUNG
   RUNG wire#powerrail
      Contact( "P_RUN" )
      Contact( "PLC_BIT".WAG1_FU )
   END_RUNG wire#w8
   // the same network as SCL:
   IF NOT "XA_HET_AGG" THEN
       "6.1.W_IND_AGG1"(W_IN := "C#7_RD_RUN".WE_AG1,   // "6.WEIGHT_HANDLING"
                        WR_IN := "6.1.W_IND_AGG1".WR_IN,
                        PV_IN1 := "C#7_RD_RUN".PV_AG1,
                        SV_IN1 := "C#4_WD_WEIGHT".SV_AG1,
                        RUN_1 := "7.1.IND_AGG1".STA_RUN,
                        EMTY := "PLC_BIT".WAG1_EM,
                        W_OUT1 => "6.1.W_IND_AGG1".W_OUT1,
                        "%W_OUT" => "C#7_RD_RUN"."%_WAG1");
   END_IF;
   "9.5.DLR_IND_AGG1"(ON := "C#7_RD_RUN".WE_AG1 <= "C#4_WD_WEIGHT"."W_IND_AGG1_KL.BRO",   // "9.TIMER_DELAY"
                      CLOCK_1S := "Clock_10Hz",
                      T_DELAY := "9.5.DLR_IND_AGG1".T_DELAY,
                      OUT => "PLC_BIT".WAG1_EM,
                      T_OUT => "9.5.DLR_IND_AGG1".T_OUT,
                      ENO => #_w1);
   IF #_w1 THEN
       "9.5.DLR_IND_AGG1".T_DELAY := "C#4_WD_WEIGHT"."W_IND_AGG1_TG.DLD" + "C#3_WD_SILO".AG1_TG_ODC;
   END_IF;
   IF "PLC_BIT".RUN AND ("PLC_BIT".AGG1_FU OR ("C#4_WD_WEIGHT".SV_AG1 = 0.0)) THEN
       "PLC_BIT".WAG1_FU := TRUE;
   END_IF;
   #_w2 := "PLC_BIT".WAG1_EM AND NOT "P_WAGG1_EM";   // rising edge of "PLC_BIT".WAG1_EM
   "P_WAGG1_EM" := "PLC_BIT".WAG1_EM;
   IF #_w2 AND ("C#7_RD_RUN".SMC_AG1 > "C#7_RD_RUN".SMX_AG1) THEN
       "C#7_RD_RUN".SMX_AG1 := "C#7_RD_RUN".SMX_AG1 + 1.0;
   END_IF;
   IF #_w2 THEN "6.1.W_IND_AGG1".WR_IN := "C#7_RD_RUN".WE_AG1; END_IF;
   "LUU TAY WAG1" := #_w2 AND NOT "C#2_WB"."SW_MAN/AUTO" AND NOT "PLC_BIT".RUN;
   IF "PLC_BIT".WAG1_EM OR NOT "PLC_BIT".RUN THEN
       "PLC_BIT".AGG1_FU := FALSE;
       "PLC_BIT".WAG1_FU := FALSE;
   END_IF;
   #_w3 := "PLC_BIT".WAG1_FU AND NOT "P_WAGG1_FU";   // rising edge of "PLC_BIT".WAG1_FU
   "P_WAGG1_FU" := "PLC_BIT".WAG1_FU;
   IF (#_w3 OR ("P_RUN" AND "PLC_BIT".WAG1_FU)) AND NOT "C#1_RB"."XA W_IND_AGG1" AND ("C#7_RD_RUN".SMC_AG1 = "C#7_RD_RUN".SMX_AG1) THEN
       "C#7_RD_RUN".SMC_AG1 := "C#7_RD_RUN".SMC_AG1 + 1.0;
   END_IF;
END_REGION
END_FUNCTION

FUNCTION "FCXL_IND_AGG2" : Void   // FC21, LAD
{ S7_Optimized_Access := 'TRUE' }
VERSION : 0.1
// stored: AutoNumber true, CodeModifiedDate 2026-01-15T16:25:53.7007107Z, CompileDate 2026-01-15T16:25:53.7394906Z, CreationDate 2026-01-15T16:24:02.4619467Z, HandleErrorsWithinBlock false, InterfaceModifiedDate 2026-01-11T04:47:47.7058671Z, IsConsistent true, IsIECCheckEnabled false, IsKnowHowProtected false, IsWriteProtected false, LibraryConformanceStatus Error: The block contains calls of single instances. Warning: The object contains access to global data blocks. Warning: The block contains direct access to inputs, outputs, bit memories, indirect access to the registry or indirect access to external memory areas that are unknown at the time of compilation., ModifiedDate 2026-01-15T16:25:53.7007107Z, ParameterModified 2026-01-11T04:47:47.7058671Z, PLCSimAdvancedSupport false, SetENOAutomatically False, StructureModified 2026-01-11T04:47:47.7058671Z, UDAEnableTagReadback false
   VAR_TEMP   // added for the SCL form of the ladder/FBD networks
      _w1 : Bool;
      _w2 : Bool;
      _w3 : Bool;
   END_VAR
BEGIN

REGION Network 1: Cân độc lập AGG2 Full
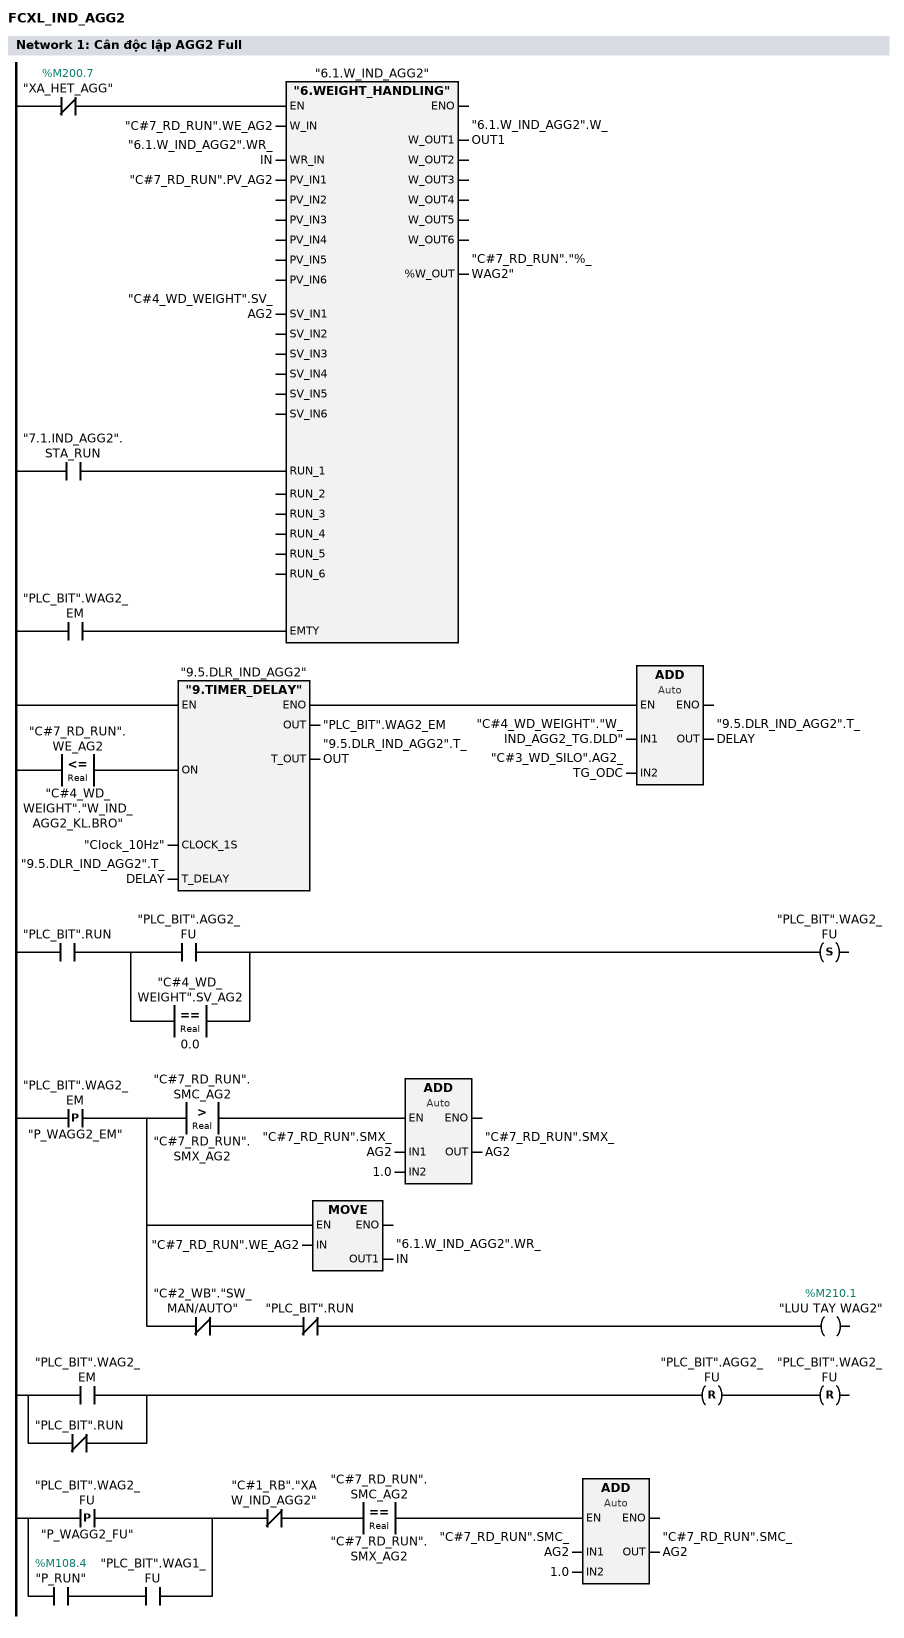
   RUNG wire#powerrail
      I_Contact( "XA_HET_AGG" )
      "6.1.W_IND_AGG2"(RUN_1 := wire#w1, EMTY := wire#w2, W_IN := "C#7_RD_RUN".WE_AG2, WR_IN := "6.1.W_IND_AGG2".WR_IN, PV_IN1 := "C#7_RD_RUN".PV_AG2, PV_IN2 :=, PV_IN3 :=, PV_IN4 :=, PV_IN5 :=, PV_IN6 :=, SV_IN1 := "C#4_WD_WEIGHT".SV_AG2, SV_IN2 :=, SV_IN3 :=, SV_IN4 :=, SV_IN5 :=, SV_IN6 :=, RUN_2 :=, RUN_3 :=, RUN_4 :=, RUN_5 :=, RUN_6 :=, W_OUT1 => "6.1.W_IND_AGG2".W_OUT1, W_OUT2 =>, W_OUT3 =>, W_OUT4 =>, W_OUT5 =>, W_OUT6 =>, "%W_OUT" => "C#7_RD_RUN"."%_WAG2")
   END_RUNG
   RUNG wire#powerrail
      Contact( "7.1.IND_AGG2".STA_RUN )
   END_RUNG wire#w1
   RUNG wire#powerrail
      Contact( "PLC_BIT".WAG2_EM )
   END_RUNG wire#w2
   RUNG wire#powerrail
      "9.5.DLR_IND_AGG2"(ON := wire#w3, CLOCK_1S := "Clock_10Hz", T_DELAY := "9.5.DLR_IND_AGG2".T_DELAY, OUT => "PLC_BIT".WAG2_EM, T_OUT => "9.5.DLR_IND_AGG2".T_OUT)
      Add(in1 := "C#4_WD_WEIGHT"."W_IND_AGG2_TG.DLD", in2 := "C#3_WD_SILO".AG2_TG_ODC, out => "9.5.DLR_IND_AGG2".T_DELAY)
   END_RUNG
   RUNG wire#powerrail
      { S7_Templates := "SrcType := Real" } LE_Contact(in1 := "C#7_RD_RUN".WE_AG2, in2 := "C#4_WD_WEIGHT"."W_IND_AGG2_KL.BRO")
   END_RUNG wire#w3
   RUNG wire#powerrail
      Contact( "PLC_BIT".RUN )
      wire#w4
      Contact( "PLC_BIT".AGG2_FU )
      wire#w5
      S_Coil( "PLC_BIT".WAG2_FU )
   END_RUNG
   RUNG wire#w4
      { S7_Templates := "SrcType := Real" } EQ_Contact(in1 := "C#4_WD_WEIGHT".SV_AG2, in2 := 0.0)
   END_RUNG wire#w5
   RUNG wire#powerrail
      P_Contact(operand := "PLC_BIT".WAG2_EM, bit := "P_WAGG2_EM")
      wire#w6
      { S7_Templates := "SrcType := Real" } GT_Contact(in1 := "C#7_RD_RUN".SMC_AG2, in2 := "C#7_RD_RUN".SMX_AG2)
      Add(in1 := "C#7_RD_RUN".SMX_AG2, in2 := 1.0, out => "C#7_RD_RUN".SMX_AG2)
   END_RUNG
   RUNG wire#w6
      Move(in := "C#7_RD_RUN".WE_AG2, out1 => "6.1.W_IND_AGG2".WR_IN)
   END_RUNG
   RUNG wire#w6
      I_Contact( "C#2_WB"."SW_MAN/AUTO" )
      I_Contact( "PLC_BIT".RUN )
      Coil( "LUU TAY WAG2" )
   END_RUNG
   RUNG wire#powerrail
      Contact( "PLC_BIT".WAG2_EM )
      wire#w7
      R_Coil( "PLC_BIT".AGG2_FU )
      R_Coil( "PLC_BIT".WAG2_FU )
   END_RUNG
   RUNG wire#powerrail
      I_Contact( "PLC_BIT".RUN )
   END_RUNG wire#w7
   RUNG wire#powerrail
      P_Contact(operand := "PLC_BIT".WAG2_FU, bit := "P_WAGG2_FU")
      wire#w8
      I_Contact( "C#1_RB"."XA W_IND_AGG2" )
      { S7_Templates := "SrcType := Real" } EQ_Contact(in1 := "C#7_RD_RUN".SMC_AG2, in2 := "C#7_RD_RUN".SMX_AG2)
      Add(in1 := "C#7_RD_RUN".SMC_AG2, in2 := 1.0, out => "C#7_RD_RUN".SMC_AG2)
   END_RUNG
   RUNG wire#powerrail
      Contact( "P_RUN" )
      Contact( "PLC_BIT".WAG1_FU )
   END_RUNG wire#w8
   // the same network as SCL:
   IF NOT "XA_HET_AGG" THEN
       "6.1.W_IND_AGG2"(W_IN := "C#7_RD_RUN".WE_AG2,   // "6.WEIGHT_HANDLING"
                        WR_IN := "6.1.W_IND_AGG2".WR_IN,
                        PV_IN1 := "C#7_RD_RUN".PV_AG2,
                        SV_IN1 := "C#4_WD_WEIGHT".SV_AG2,
                        RUN_1 := "7.1.IND_AGG2".STA_RUN,
                        EMTY := "PLC_BIT".WAG2_EM,
                        W_OUT1 => "6.1.W_IND_AGG2".W_OUT1,
                        "%W_OUT" => "C#7_RD_RUN"."%_WAG2");
   END_IF;
   "9.5.DLR_IND_AGG2"(ON := "C#7_RD_RUN".WE_AG2 <= "C#4_WD_WEIGHT"."W_IND_AGG2_KL.BRO",   // "9.TIMER_DELAY"
                      CLOCK_1S := "Clock_10Hz",
                      T_DELAY := "9.5.DLR_IND_AGG2".T_DELAY,
                      OUT => "PLC_BIT".WAG2_EM,
                      T_OUT => "9.5.DLR_IND_AGG2".T_OUT,
                      ENO => #_w1);
   IF #_w1 THEN
       "9.5.DLR_IND_AGG2".T_DELAY := "C#4_WD_WEIGHT"."W_IND_AGG2_TG.DLD" + "C#3_WD_SILO".AG2_TG_ODC;
   END_IF;
   IF "PLC_BIT".RUN AND ("PLC_BIT".AGG2_FU OR ("C#4_WD_WEIGHT".SV_AG2 = 0.0)) THEN
       "PLC_BIT".WAG2_FU := TRUE;
   END_IF;
   #_w2 := "PLC_BIT".WAG2_EM AND NOT "P_WAGG2_EM";   // rising edge of "PLC_BIT".WAG2_EM
   "P_WAGG2_EM" := "PLC_BIT".WAG2_EM;
   IF #_w2 AND ("C#7_RD_RUN".SMC_AG2 > "C#7_RD_RUN".SMX_AG2) THEN
       "C#7_RD_RUN".SMX_AG2 := "C#7_RD_RUN".SMX_AG2 + 1.0;
   END_IF;
   IF #_w2 THEN "6.1.W_IND_AGG2".WR_IN := "C#7_RD_RUN".WE_AG2; END_IF;
   "LUU TAY WAG2" := #_w2 AND NOT "C#2_WB"."SW_MAN/AUTO" AND NOT "PLC_BIT".RUN;
   IF "PLC_BIT".WAG2_EM OR NOT "PLC_BIT".RUN THEN
       "PLC_BIT".AGG2_FU := FALSE;
       "PLC_BIT".WAG2_FU := FALSE;
   END_IF;
   #_w3 := "PLC_BIT".WAG2_FU AND NOT "P_WAGG2_FU";   // rising edge of "PLC_BIT".WAG2_FU
   "P_WAGG2_FU" := "PLC_BIT".WAG2_FU;
   IF (#_w3 OR ("P_RUN" AND "PLC_BIT".WAG1_FU)) AND NOT "C#1_RB"."XA W_IND_AGG2" AND ("C#7_RD_RUN".SMC_AG2 = "C#7_RD_RUN".SMX_AG2) THEN
       "C#7_RD_RUN".SMC_AG2 := "C#7_RD_RUN".SMC_AG2 + 1.0;
   END_IF;
END_REGION
END_FUNCTION

FUNCTION "FCXL_IND_AGG3" : Void   // FC22, LAD
{ S7_Optimized_Access := 'TRUE' }
VERSION : 0.1
// stored: AutoNumber true, CodeModifiedDate 2026-01-15T16:25:53.6082795Z, CompileDate 2026-01-15T16:25:53.6491144Z, CreationDate 2026-01-15T16:24:02.4619467Z, HandleErrorsWithinBlock false, InterfaceModifiedDate 2026-01-11T04:48:05.8897553Z, IsConsistent true, IsIECCheckEnabled false, IsKnowHowProtected false, IsWriteProtected false, LibraryConformanceStatus Error: The block contains calls of single instances. Warning: The object contains access to global data blocks. Warning: The block contains direct access to inputs, outputs, bit memories, indirect access to the registry or indirect access to external memory areas that are unknown at the time of compilation., ModifiedDate 2026-01-15T16:25:53.6082795Z, ParameterModified 2026-01-11T04:48:05.8897553Z, PLCSimAdvancedSupport false, SetENOAutomatically False, StructureModified 2026-01-11T04:48:05.8897553Z, UDAEnableTagReadback false
   VAR_TEMP   // added for the SCL form of the ladder/FBD networks
      _w1 : Bool;
      _w2 : Bool;
      _w3 : Bool;
   END_VAR
BEGIN

REGION Network 1: Cân độc lập AGG3 Full
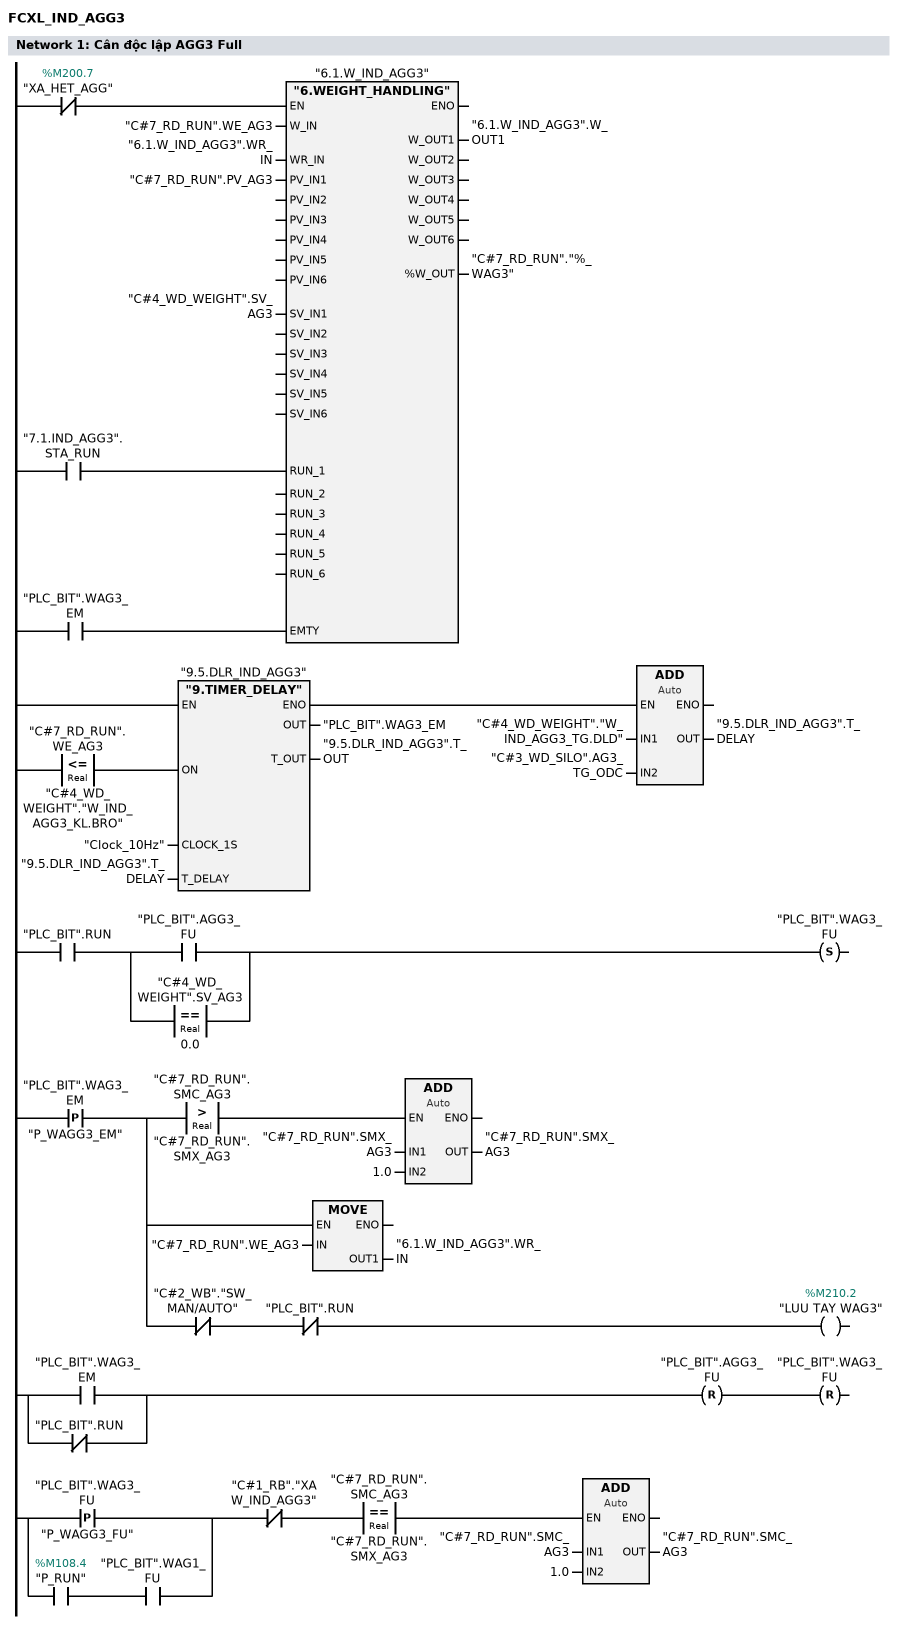
   RUNG wire#powerrail
      I_Contact( "XA_HET_AGG" )
      "6.1.W_IND_AGG3"(RUN_1 := wire#w1, EMTY := wire#w2, W_IN := "C#7_RD_RUN".WE_AG3, WR_IN := "6.1.W_IND_AGG3".WR_IN, PV_IN1 := "C#7_RD_RUN".PV_AG3, PV_IN2 :=, PV_IN3 :=, PV_IN4 :=, PV_IN5 :=, PV_IN6 :=, SV_IN1 := "C#4_WD_WEIGHT".SV_AG3, SV_IN2 :=, SV_IN3 :=, SV_IN4 :=, SV_IN5 :=, SV_IN6 :=, RUN_2 :=, RUN_3 :=, RUN_4 :=, RUN_5 :=, RUN_6 :=, W_OUT1 => "6.1.W_IND_AGG3".W_OUT1, W_OUT2 =>, W_OUT3 =>, W_OUT4 =>, W_OUT5 =>, W_OUT6 =>, "%W_OUT" => "C#7_RD_RUN"."%_WAG3")
   END_RUNG
   RUNG wire#powerrail
      Contact( "7.1.IND_AGG3".STA_RUN )
   END_RUNG wire#w1
   RUNG wire#powerrail
      Contact( "PLC_BIT".WAG3_EM )
   END_RUNG wire#w2
   RUNG wire#powerrail
      "9.5.DLR_IND_AGG3"(ON := wire#w3, CLOCK_1S := "Clock_10Hz", T_DELAY := "9.5.DLR_IND_AGG3".T_DELAY, OUT => "PLC_BIT".WAG3_EM, T_OUT => "9.5.DLR_IND_AGG3".T_OUT)
      Add(in1 := "C#4_WD_WEIGHT"."W_IND_AGG3_TG.DLD", in2 := "C#3_WD_SILO".AG3_TG_ODC, out => "9.5.DLR_IND_AGG3".T_DELAY)
   END_RUNG
   RUNG wire#powerrail
      { S7_Templates := "SrcType := Real" } LE_Contact(in1 := "C#7_RD_RUN".WE_AG3, in2 := "C#4_WD_WEIGHT"."W_IND_AGG3_KL.BRO")
   END_RUNG wire#w3
   RUNG wire#powerrail
      Contact( "PLC_BIT".RUN )
      wire#w4
      Contact( "PLC_BIT".AGG3_FU )
      wire#w5
      S_Coil( "PLC_BIT".WAG3_FU )
   END_RUNG
   RUNG wire#w4
      { S7_Templates := "SrcType := Real" } EQ_Contact(in1 := "C#4_WD_WEIGHT".SV_AG3, in2 := 0.0)
   END_RUNG wire#w5
   RUNG wire#powerrail
      P_Contact(operand := "PLC_BIT".WAG3_EM, bit := "P_WAGG3_EM")
      wire#w6
      { S7_Templates := "SrcType := Real" } GT_Contact(in1 := "C#7_RD_RUN".SMC_AG3, in2 := "C#7_RD_RUN".SMX_AG3)
      Add(in1 := "C#7_RD_RUN".SMX_AG3, in2 := 1.0, out => "C#7_RD_RUN".SMX_AG3)
   END_RUNG
   RUNG wire#w6
      Move(in := "C#7_RD_RUN".WE_AG3, out1 => "6.1.W_IND_AGG3".WR_IN)
   END_RUNG
   RUNG wire#w6
      I_Contact( "C#2_WB"."SW_MAN/AUTO" )
      I_Contact( "PLC_BIT".RUN )
      Coil( "LUU TAY WAG3" )
   END_RUNG
   RUNG wire#powerrail
      Contact( "PLC_BIT".WAG3_EM )
      wire#w7
      R_Coil( "PLC_BIT".AGG3_FU )
      R_Coil( "PLC_BIT".WAG3_FU )
   END_RUNG
   RUNG wire#powerrail
      I_Contact( "PLC_BIT".RUN )
   END_RUNG wire#w7
   RUNG wire#powerrail
      P_Contact(operand := "PLC_BIT".WAG3_FU, bit := "P_WAGG3_FU")
      wire#w8
      I_Contact( "C#1_RB"."XA W_IND_AGG3" )
      { S7_Templates := "SrcType := Real" } EQ_Contact(in1 := "C#7_RD_RUN".SMC_AG3, in2 := "C#7_RD_RUN".SMX_AG3)
      Add(in1 := "C#7_RD_RUN".SMC_AG3, in2 := 1.0, out => "C#7_RD_RUN".SMC_AG3)
   END_RUNG
   RUNG wire#powerrail
      Contact( "P_RUN" )
      Contact( "PLC_BIT".WAG1_FU )
   END_RUNG wire#w8
   // the same network as SCL:
   IF NOT "XA_HET_AGG" THEN
       "6.1.W_IND_AGG3"(W_IN := "C#7_RD_RUN".WE_AG3,   // "6.WEIGHT_HANDLING"
                        WR_IN := "6.1.W_IND_AGG3".WR_IN,
                        PV_IN1 := "C#7_RD_RUN".PV_AG3,
                        SV_IN1 := "C#4_WD_WEIGHT".SV_AG3,
                        RUN_1 := "7.1.IND_AGG3".STA_RUN,
                        EMTY := "PLC_BIT".WAG3_EM,
                        W_OUT1 => "6.1.W_IND_AGG3".W_OUT1,
                        "%W_OUT" => "C#7_RD_RUN"."%_WAG3");
   END_IF;
   "9.5.DLR_IND_AGG3"(ON := "C#7_RD_RUN".WE_AG3 <= "C#4_WD_WEIGHT"."W_IND_AGG3_KL.BRO",   // "9.TIMER_DELAY"
                      CLOCK_1S := "Clock_10Hz",
                      T_DELAY := "9.5.DLR_IND_AGG3".T_DELAY,
                      OUT => "PLC_BIT".WAG3_EM,
                      T_OUT => "9.5.DLR_IND_AGG3".T_OUT,
                      ENO => #_w1);
   IF #_w1 THEN
       "9.5.DLR_IND_AGG3".T_DELAY := "C#4_WD_WEIGHT"."W_IND_AGG3_TG.DLD" + "C#3_WD_SILO".AG3_TG_ODC;
   END_IF;
   IF "PLC_BIT".RUN AND ("PLC_BIT".AGG3_FU OR ("C#4_WD_WEIGHT".SV_AG3 = 0.0)) THEN
       "PLC_BIT".WAG3_FU := TRUE;
   END_IF;
   #_w2 := "PLC_BIT".WAG3_EM AND NOT "P_WAGG3_EM";   // rising edge of "PLC_BIT".WAG3_EM
   "P_WAGG3_EM" := "PLC_BIT".WAG3_EM;
   IF #_w2 AND ("C#7_RD_RUN".SMC_AG3 > "C#7_RD_RUN".SMX_AG3) THEN
       "C#7_RD_RUN".SMX_AG3 := "C#7_RD_RUN".SMX_AG3 + 1.0;
   END_IF;
   IF #_w2 THEN "6.1.W_IND_AGG3".WR_IN := "C#7_RD_RUN".WE_AG3; END_IF;
   "LUU TAY WAG3" := #_w2 AND NOT "C#2_WB"."SW_MAN/AUTO" AND NOT "PLC_BIT".RUN;
   IF "PLC_BIT".WAG3_EM OR NOT "PLC_BIT".RUN THEN
       "PLC_BIT".AGG3_FU := FALSE;
       "PLC_BIT".WAG3_FU := FALSE;
   END_IF;
   #_w3 := "PLC_BIT".WAG3_FU AND NOT "P_WAGG3_FU";   // rising edge of "PLC_BIT".WAG3_FU
   "P_WAGG3_FU" := "PLC_BIT".WAG3_FU;
   IF (#_w3 OR ("P_RUN" AND "PLC_BIT".WAG1_FU)) AND NOT "C#1_RB"."XA W_IND_AGG3" AND ("C#7_RD_RUN".SMC_AG3 = "C#7_RD_RUN".SMX_AG3) THEN
       "C#7_RD_RUN".SMC_AG3 := "C#7_RD_RUN".SMC_AG3 + 1.0;
   END_IF;
END_REGION
END_FUNCTION

